REGION Network 39: Step[802] :
   RUNG wire#powerrail
      { S7_Templates := "SrcType := DInt" } EQ_Contact(in1 := "Unit1.Em2.ControlNodes".semiAutoSplice.sequence.status.currentStep, in2 := #JOB_8_STEP_02)
      Contact( "Unit1.Em2.ControlNodes".semiAutoSplice.sequence.status.seqActive )
      wire#w1
      Coil( "Unit1.Em2.ControlNodes".semiAutoSplice."step".action1[802] )
   END_RUNG
   RUNG wire#w1
      Coil( "Unit1.Em2.ControlNodes".semiAutoSplice."step".transition1[802] )
   END_RUNG
   RUNG wire#w1
      Contact( "Unit1.Em2.ControlNodes".semiAutoSplice."step".transition1[802] )
      { S7_Templates := "time_type := Time" } #statTonTimer[802].TON(pt := #SeqDelayTime, et =>)
      Move(in := #JOB_8_STEP_03, out1 => "Unit1.Em2.ControlNodes".semiAutoSplice.sequence.status.nextStep)
   END_RUNG
   // the same network as SCL:
   "Unit1.Em2.ControlNodes".semiAutoSplice."step".action1[802] := ("Unit1.Em2.ControlNodes".semiAutoSplice.sequence.status.currentStep = #JOB_8_STEP_02) AND "Unit1.Em2.ControlNodes".semiAutoSplice.sequence.status.seqActive;
   "Unit1.Em2.ControlNodes".semiAutoSplice."step".transition1[802] := ("Unit1.Em2.ControlNodes".semiAutoSplice.sequence.status.currentStep = #JOB_8_STEP_02) AND "Unit1.Em2.ControlNodes".semiAutoSplice.sequence.status.seqActive;
   #statTonTimer[802].TON(IN := ("Unit1.Em2.ControlNodes".semiAutoSplice.sequence.status.currentStep = #JOB_8_STEP_02) AND "Unit1.Em2.ControlNodes".semiAutoSplice.sequence.status.seqActive AND "Unit1.Em2.ControlNodes".semiAutoSplice."step".transition1[802],
                          PT := #SeqDelayTime);
   IF #statTonTimer[802].Q THEN
       "Unit1.Em2.ControlNodes".semiAutoSplice.sequence.status.nextStep := #JOB_8_STEP_03;
   END_IF;
END_REGION

REGION Network 40: Step[803] : cutter Home (Down)
   RUNG wire#powerrail
      { S7_Templates := "SrcType := DInt" } EQ_Contact(in1 := "Unit1.Em2.ControlNodes".semiAutoSplice.sequence.status.currentStep, in2 := #JOB_8_STEP_03)
      Contact( "Unit1.Em2.ControlNodes".semiAutoSplice.sequence.status.seqActive )
      wire#w1
      I_Contact( "Unit1.Em2.ControlNodes".cmCutterUpDown.monitoring.inHomePos )
      Coil( "Unit1.Em2.ControlNodes".semiAutoSplice."step".action1[803] )
   END_RUNG
   RUNG wire#w1
      Contact( "Unit1.Em2.ControlNodes".cmCutterUpDown.monitoring.inHomePos )
      Coil( "Unit1.Em2.ControlNodes".semiAutoSplice."step".transition1[803] )
   END_RUNG
   RUNG wire#w1
      Contact( "Unit1.Em2.ControlNodes".semiAutoSplice."step".transition1[803] )
      { S7_Templates := "time_type := Time" } #statTonTimer[803].TON(pt := #SeqDelayTime, et =>)
      Move(in := #JOB_8_STEP_04, out1 => "Unit1.Em2.ControlNodes".semiAutoSplice.sequence.status.nextStep)
      Add(in1 := #RetryCnt[0], in2 := 1, out => #RetryCnt[0])
   END_RUNG
   // the same network as SCL:
   #_w1 := ("Unit1.Em2.ControlNodes".semiAutoSplice.sequence.status.currentStep = #JOB_8_STEP_03) AND "Unit1.Em2.ControlNodes".semiAutoSplice.sequence.status.seqActive;
   "Unit1.Em2.ControlNodes".semiAutoSplice."step".action1[803] := #_w1 AND NOT "Unit1.Em2.ControlNodes".cmCutterUpDown.monitoring.inHomePos;
   "Unit1.Em2.ControlNodes".semiAutoSplice."step".transition1[803] := #_w1 AND "Unit1.Em2.ControlNodes".cmCutterUpDown.monitoring.inHomePos;
   #statTonTimer[803].TON(IN := #_w1 AND "Unit1.Em2.ControlNodes".semiAutoSplice."step".transition1[803],
                          PT := #SeqDelayTime);
   IF #statTonTimer[803].Q THEN
       "Unit1.Em2.ControlNodes".semiAutoSplice.sequence.status.nextStep := #JOB_8_STEP_04;
       #RetryCnt[0] := #RetryCnt[0] + 1;
   END_IF;
END_REGION

REGION Network 41: Step[804] : retry
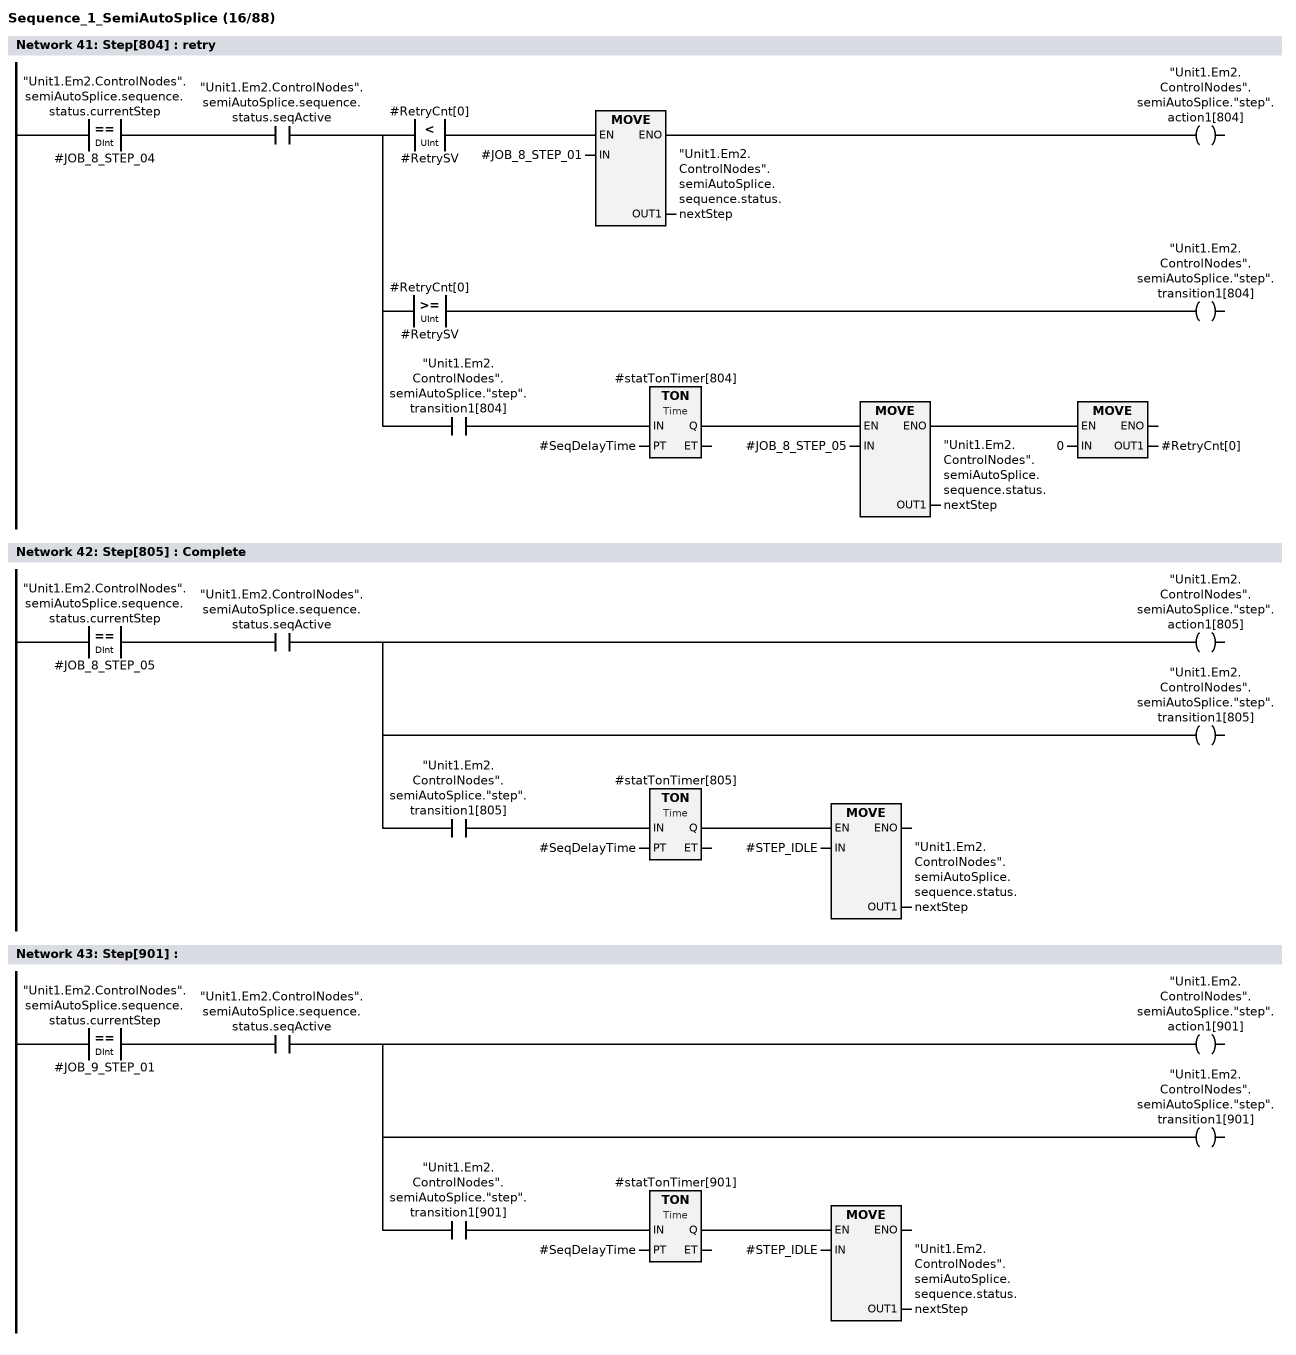
   RUNG wire#powerrail
      { S7_Templates := "SrcType := DInt" } EQ_Contact(in1 := "Unit1.Em2.ControlNodes".semiAutoSplice.sequence.status.currentStep, in2 := #JOB_8_STEP_04)
      Contact( "Unit1.Em2.ControlNodes".semiAutoSplice.sequence.status.seqActive )
      wire#w1
      { S7_Templates := "SrcType := UInt" } LT_Contact(in1 := #RetryCnt[0], in2 := #RetrySV)
      Move(in := #JOB_8_STEP_01, out1 => "Unit1.Em2.ControlNodes".semiAutoSplice.sequence.status.nextStep)
      Coil( "Unit1.Em2.ControlNodes".semiAutoSplice."step".action1[804] )
   END_RUNG
   RUNG wire#w1
      { S7_Templates := "SrcType := UInt" } GE_Contact(in1 := #RetryCnt[0], in2 := #RetrySV)
      Coil( "Unit1.Em2.ControlNodes".semiAutoSplice."step".transition1[804] )
   END_RUNG
   RUNG wire#w1
      Contact( "Unit1.Em2.ControlNodes".semiAutoSplice."step".transition1[804] )
      { S7_Templates := "time_type := Time" } #statTonTimer[804].TON(pt := #SeqDelayTime, et =>)
      Move(in := #JOB_8_STEP_05, out1 => "Unit1.Em2.ControlNodes".semiAutoSplice.sequence.status.nextStep)
      Move(in := 0, out1 => #RetryCnt[0])
   END_RUNG
   // the same network as SCL:
   #_w1 := ("Unit1.Em2.ControlNodes".semiAutoSplice.sequence.status.currentStep = #JOB_8_STEP_04) AND "Unit1.Em2.ControlNodes".semiAutoSplice.sequence.status.seqActive;
   #_w2 := #_w1 AND (#RetryCnt[0] < #RetrySV);
   IF #_w2 THEN "Unit1.Em2.ControlNodes".semiAutoSplice.sequence.status.nextStep := #JOB_8_STEP_01; END_IF;
   "Unit1.Em2.ControlNodes".semiAutoSplice."step".action1[804] := #_w2;
   "Unit1.Em2.ControlNodes".semiAutoSplice."step".transition1[804] := #_w1 AND (#RetryCnt[0] >= #RetrySV);
   #statTonTimer[804].TON(IN := #_w1 AND "Unit1.Em2.ControlNodes".semiAutoSplice."step".transition1[804],
                          PT := #SeqDelayTime);
   IF #statTonTimer[804].Q THEN
       "Unit1.Em2.ControlNodes".semiAutoSplice.sequence.status.nextStep := #JOB_8_STEP_05;
       #RetryCnt[0] := 0;
   END_IF;
END_REGION

REGION Network 42: Step[805] : Complete
   RUNG wire#powerrail
      { S7_Templates := "SrcType := DInt" } EQ_Contact(in1 := "Unit1.Em2.ControlNodes".semiAutoSplice.sequence.status.currentStep, in2 := #JOB_8_STEP_05)
      Contact( "Unit1.Em2.ControlNodes".semiAutoSplice.sequence.status.seqActive )
      wire#w1
      Coil( "Unit1.Em2.ControlNodes".semiAutoSplice."step".action1[805] )
   END_RUNG
   RUNG wire#w1
      Coil( "Unit1.Em2.ControlNodes".semiAutoSplice."step".transition1[805] )
   END_RUNG
   RUNG wire#w1
      Contact( "Unit1.Em2.ControlNodes".semiAutoSplice."step".transition1[805] )
      { S7_Templates := "time_type := Time" } #statTonTimer[805].TON(pt := #SeqDelayTime, et =>)
      Move(in := #STEP_IDLE, out1 => "Unit1.Em2.ControlNodes".semiAutoSplice.sequence.status.nextStep)
   END_RUNG
   // the same network as SCL:
   "Unit1.Em2.ControlNodes".semiAutoSplice."step".action1[805] := ("Unit1.Em2.ControlNodes".semiAutoSplice.sequence.status.currentStep = #JOB_8_STEP_05) AND "Unit1.Em2.ControlNodes".semiAutoSplice.sequence.status.seqActive;
   "Unit1.Em2.ControlNodes".semiAutoSplice."step".transition1[805] := ("Unit1.Em2.ControlNodes".semiAutoSplice.sequence.status.currentStep = #JOB_8_STEP_05) AND "Unit1.Em2.ControlNodes".semiAutoSplice.sequence.status.seqActive;
   #statTonTimer[805].TON(IN := ("Unit1.Em2.ControlNodes".semiAutoSplice.sequence.status.currentStep = #JOB_8_STEP_05) AND "Unit1.Em2.ControlNodes".semiAutoSplice.sequence.status.seqActive AND "Unit1.Em2.ControlNodes".semiAutoSplice."step".transition1[805],
                          PT := #SeqDelayTime);
   IF #statTonTimer[805].Q THEN
       "Unit1.Em2.ControlNodes".semiAutoSplice.sequence.status.nextStep := #STEP_IDLE;
   END_IF;
END_REGION

REGION Network 43: Step[901] :
   RUNG wire#powerrail
      { S7_Templates := "SrcType := DInt" } EQ_Contact(in1 := "Unit1.Em2.ControlNodes".semiAutoSplice.sequence.status.currentStep, in2 := #JOB_9_STEP_01)
      Contact( "Unit1.Em2.ControlNodes".semiAutoSplice.sequence.status.seqActive )
      wire#w1
      Coil( "Unit1.Em2.ControlNodes".semiAutoSplice."step".action1[901] )
   END_RUNG
   RUNG wire#w1
      Coil( "Unit1.Em2.ControlNodes".semiAutoSplice."step".transition1[901] )
   END_RUNG
   RUNG wire#w1
      Contact( "Unit1.Em2.ControlNodes".semiAutoSplice."step".transition1[901] )
      { S7_Templates := "time_type := Time" } #statTonTimer[901].TON(pt := #SeqDelayTime, et =>)
      Move(in := #STEP_IDLE, out1 => "Unit1.Em2.ControlNodes".semiAutoSplice.sequence.status.nextStep)
   END_RUNG
   // the same network as SCL:
   "Unit1.Em2.ControlNodes".semiAutoSplice."step".action1[901] := ("Unit1.Em2.ControlNodes".semiAutoSplice.sequence.status.currentStep = #JOB_9_STEP_01) AND "Unit1.Em2.ControlNodes".semiAutoSplice.sequence.status.seqActive;
   "Unit1.Em2.ControlNodes".semiAutoSplice."step".transition1[901] := ("Unit1.Em2.ControlNodes".semiAutoSplice.sequence.status.currentStep = #JOB_9_STEP_01) AND "Unit1.Em2.ControlNodes".semiAutoSplice.sequence.status.seqActive;
   #statTonTimer[901].TON(IN := ("Unit1.Em2.ControlNodes".semiAutoSplice.sequence.status.currentStep = #JOB_9_STEP_01) AND "Unit1.Em2.ControlNodes".semiAutoSplice.sequence.status.seqActive AND "Unit1.Em2.ControlNodes".semiAutoSplice."step".transition1[901],
                          PT := #SeqDelayTime);
   IF #statTonTimer[901].Q THEN
       "Unit1.Em2.ControlNodes".semiAutoSplice.sequence.status.nextStep := #STEP_IDLE;
   END_IF;
END_REGION

REGION Network 44: Step[1001] : Top Link Top Left/right Vacc Off (Btm Left/Right Vacc On)
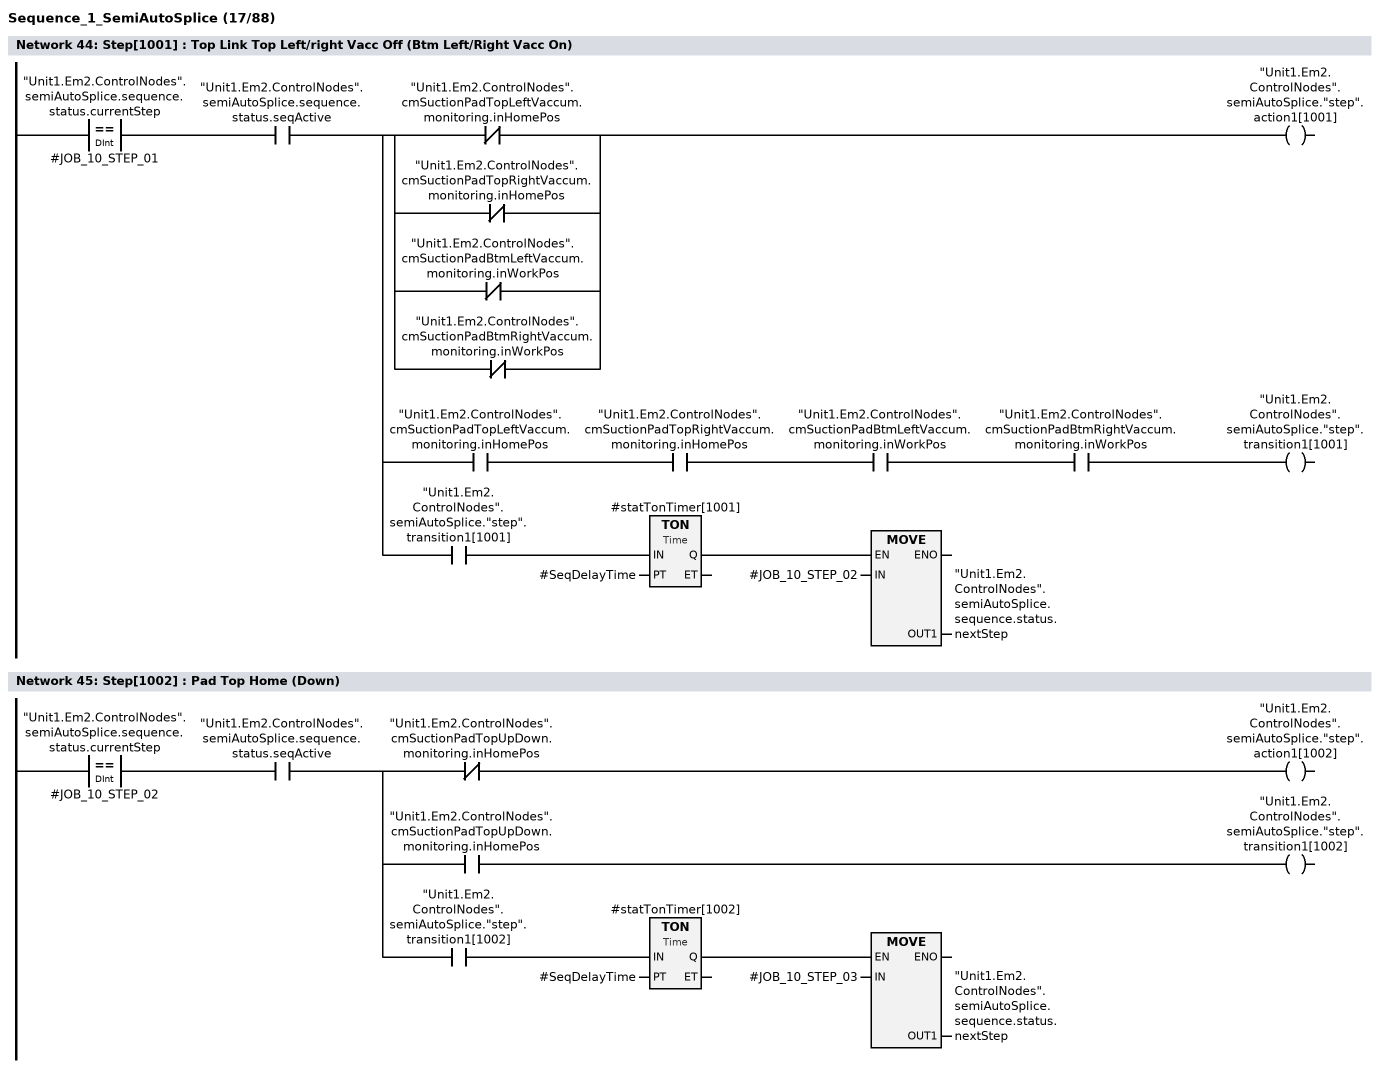
   RUNG wire#powerrail
      { S7_Templates := "SrcType := DInt" } EQ_Contact(in1 := "Unit1.Em2.ControlNodes".semiAutoSplice.sequence.status.currentStep, in2 := #JOB_10_STEP_01)
      Contact( "Unit1.Em2.ControlNodes".semiAutoSplice.sequence.status.seqActive )
      wire#w1
      I_Contact( "Unit1.Em2.ControlNodes".cmSuctionPadTopLeftVaccum.monitoring.inHomePos )
      wire#w2
      Coil( "Unit1.Em2.ControlNodes".semiAutoSplice."step".action1[1001] )
   END_RUNG
   RUNG wire#w1
      I_Contact( "Unit1.Em2.ControlNodes".cmSuctionPadTopRightVaccum.monitoring.inHomePos )
   END_RUNG wire#w2
   RUNG wire#w1
      I_Contact( "Unit1.Em2.ControlNodes".cmSuctionPadBtmLeftVaccum.monitoring.inWorkPos )
   END_RUNG wire#w2
   RUNG wire#w1
      I_Contact( "Unit1.Em2.ControlNodes".cmSuctionPadBtmRightVaccum.monitoring.inWorkPos )
   END_RUNG wire#w2
   RUNG wire#w1
      Contact( "Unit1.Em2.ControlNodes".cmSuctionPadTopLeftVaccum.monitoring.inHomePos )
      Contact( "Unit1.Em2.ControlNodes".cmSuctionPadTopRightVaccum.monitoring.inHomePos )
      Contact( "Unit1.Em2.ControlNodes".cmSuctionPadBtmLeftVaccum.monitoring.inWorkPos )
      Contact( "Unit1.Em2.ControlNodes".cmSuctionPadBtmRightVaccum.monitoring.inWorkPos )
      Coil( "Unit1.Em2.ControlNodes".semiAutoSplice."step".transition1[1001] )
   END_RUNG
   RUNG wire#w1
      Contact( "Unit1.Em2.ControlNodes".semiAutoSplice."step".transition1[1001] )
      { S7_Templates := "time_type := Time" } #statTonTimer[1001].TON(pt := #SeqDelayTime, et =>)
      Move(in := #JOB_10_STEP_02, out1 => "Unit1.Em2.ControlNodes".semiAutoSplice.sequence.status.nextStep)
   END_RUNG
   // the same network as SCL:
   #_w1 := ("Unit1.Em2.ControlNodes".semiAutoSplice.sequence.status.currentStep = #JOB_10_STEP_01) AND "Unit1.Em2.ControlNodes".semiAutoSplice.sequence.status.seqActive;
   "Unit1.Em2.ControlNodes".semiAutoSplice."step".action1[1001] := #_w1 AND (NOT "Unit1.Em2.ControlNodes".cmSuctionPadTopLeftVaccum.monitoring.inHomePos OR NOT "Unit1.Em2.ControlNodes".cmSuctionPadTopRightVaccum.monitoring.inHomePos OR NOT "Unit1.Em2.ControlNodes".cmSuctionPadBtmLeftVaccum.monitoring.inWorkPos OR NOT "Unit1.Em2.ControlNodes".cmSuctionPadBtmRightVaccum.monitoring.inWorkPos);
   "Unit1.Em2.ControlNodes".semiAutoSplice."step".transition1[1001] := #_w1 AND "Unit1.Em2.ControlNodes".cmSuctionPadTopLeftVaccum.monitoring.inHomePos AND "Unit1.Em2.ControlNodes".cmSuctionPadTopRightVaccum.monitoring.inHomePos AND "Unit1.Em2.ControlNodes".cmSuctionPadBtmLeftVaccum.monitoring.inWorkPos AND "Unit1.Em2.ControlNodes".cmSuctionPadBtmRightVaccum.monitoring.inWorkPos;
   #statTonTimer[1001].TON(IN := #_w1 AND "Unit1.Em2.ControlNodes".semiAutoSplice."step".transition1[1001],
                           PT := #SeqDelayTime);
   IF #statTonTimer[1001].Q THEN
       "Unit1.Em2.ControlNodes".semiAutoSplice.sequence.status.nextStep := #JOB_10_STEP_02;
   END_IF;
END_REGION

REGION Network 45: Step[1002] : Pad Top Home (Down)
   RUNG wire#powerrail
      { S7_Templates := "SrcType := DInt" } EQ_Contact(in1 := "Unit1.Em2.ControlNodes".semiAutoSplice.sequence.status.currentStep, in2 := #JOB_10_STEP_02)
      Contact( "Unit1.Em2.ControlNodes".semiAutoSplice.sequence.status.seqActive )
      wire#w1
      I_Contact( "Unit1.Em2.ControlNodes".cmSuctionPadTopUpDown.monitoring.inHomePos )
      Coil( "Unit1.Em2.ControlNodes".semiAutoSplice."step".action1[1002] )
   END_RUNG
   RUNG wire#w1
      Contact( "Unit1.Em2.ControlNodes".cmSuctionPadTopUpDown.monitoring.inHomePos )
      Coil( "Unit1.Em2.ControlNodes".semiAutoSplice."step".transition1[1002] )
   END_RUNG
   RUNG wire#w1
      Contact( "Unit1.Em2.ControlNodes".semiAutoSplice."step".transition1[1002] )
      { S7_Templates := "time_type := Time" } #statTonTimer[1002].TON(pt := #SeqDelayTime, et =>)
      Move(in := #JOB_10_STEP_03, out1 => "Unit1.Em2.ControlNodes".semiAutoSplice.sequence.status.nextStep)
   END_RUNG
   // the same network as SCL:
   #_w1 := ("Unit1.Em2.ControlNodes".semiAutoSplice.sequence.status.currentStep = #JOB_10_STEP_02) AND "Unit1.Em2.ControlNodes".semiAutoSplice.sequence.status.seqActive;
   "Unit1.Em2.ControlNodes".semiAutoSplice."step".action1[1002] := #_w1 AND NOT "Unit1.Em2.ControlNodes".cmSuctionPadTopUpDown.monitoring.inHomePos;
   "Unit1.Em2.ControlNodes".semiAutoSplice."step".transition1[1002] := #_w1 AND "Unit1.Em2.ControlNodes".cmSuctionPadTopUpDown.monitoring.inHomePos;
   #statTonTimer[1002].TON(IN := #_w1 AND "Unit1.Em2.ControlNodes".semiAutoSplice."step".transition1[1002],
                           PT := #SeqDelayTime);
   IF #statTonTimer[1002].Q THEN
       "Unit1.Em2.ControlNodes".semiAutoSplice.sequence.status.nextStep := #JOB_10_STEP_03;
   END_IF;
END_REGION

REGION Network 46: Step[1003] :
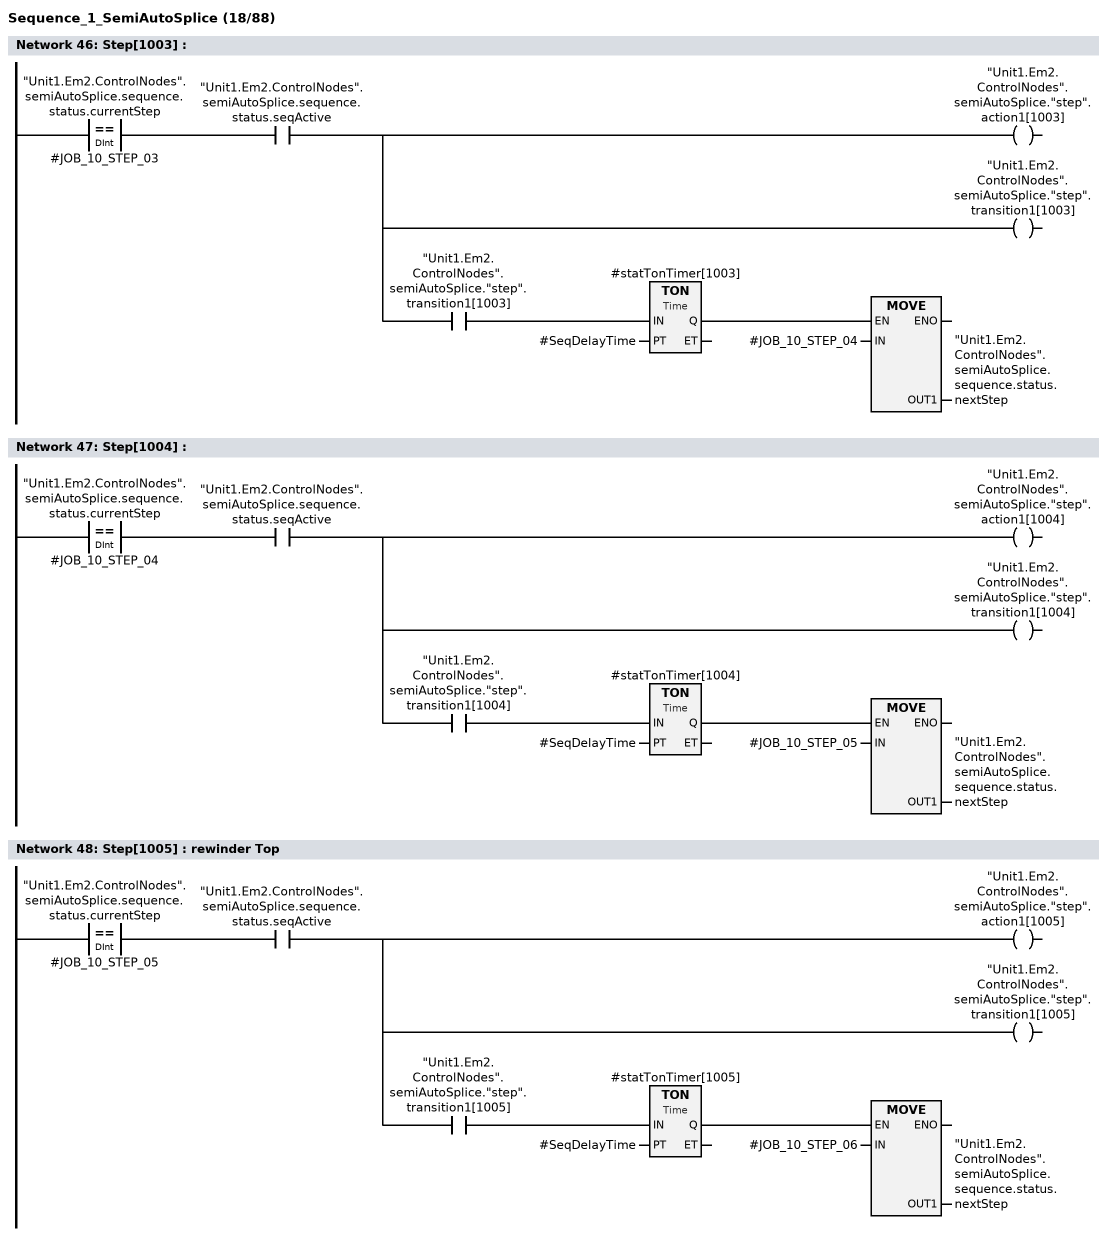
   RUNG wire#powerrail
      { S7_Templates := "SrcType := DInt" } EQ_Contact(in1 := "Unit1.Em2.ControlNodes".semiAutoSplice.sequence.status.currentStep, in2 := #JOB_10_STEP_03)
      Contact( "Unit1.Em2.ControlNodes".semiAutoSplice.sequence.status.seqActive )
      wire#w1
      Coil( "Unit1.Em2.ControlNodes".semiAutoSplice."step".action1[1003] )
   END_RUNG
   RUNG wire#w1
      Coil( "Unit1.Em2.ControlNodes".semiAutoSplice."step".transition1[1003] )
   END_RUNG
   RUNG wire#w1
      Contact( "Unit1.Em2.ControlNodes".semiAutoSplice."step".transition1[1003] )
      { S7_Templates := "time_type := Time" } #statTonTimer[1003].TON(pt := #SeqDelayTime, et =>)
      Move(in := #JOB_10_STEP_04, out1 => "Unit1.Em2.ControlNodes".semiAutoSplice.sequence.status.nextStep)
   END_RUNG
   // the same network as SCL:
   "Unit1.Em2.ControlNodes".semiAutoSplice."step".action1[1003] := ("Unit1.Em2.ControlNodes".semiAutoSplice.sequence.status.currentStep = #JOB_10_STEP_03) AND "Unit1.Em2.ControlNodes".semiAutoSplice.sequence.status.seqActive;
   "Unit1.Em2.ControlNodes".semiAutoSplice."step".transition1[1003] := ("Unit1.Em2.ControlNodes".semiAutoSplice.sequence.status.currentStep = #JOB_10_STEP_03) AND "Unit1.Em2.ControlNodes".semiAutoSplice.sequence.status.seqActive;
   #statTonTimer[1003].TON(IN := ("Unit1.Em2.ControlNodes".semiAutoSplice.sequence.status.currentStep = #JOB_10_STEP_03) AND "Unit1.Em2.ControlNodes".semiAutoSplice.sequence.status.seqActive AND "Unit1.Em2.ControlNodes".semiAutoSplice."step".transition1[1003],
                           PT := #SeqDelayTime);
   IF #statTonTimer[1003].Q THEN
       "Unit1.Em2.ControlNodes".semiAutoSplice.sequence.status.nextStep := #JOB_10_STEP_04;
   END_IF;
END_REGION

REGION Network 47: Step[1004] :
   RUNG wire#powerrail
      { S7_Templates := "SrcType := DInt" } EQ_Contact(in1 := "Unit1.Em2.ControlNodes".semiAutoSplice.sequence.status.currentStep, in2 := #JOB_10_STEP_04)
      Contact( "Unit1.Em2.ControlNodes".semiAutoSplice.sequence.status.seqActive )
      wire#w1
      Coil( "Unit1.Em2.ControlNodes".semiAutoSplice."step".action1[1004] )
   END_RUNG
   RUNG wire#w1
      Coil( "Unit1.Em2.ControlNodes".semiAutoSplice."step".transition1[1004] )
   END_RUNG
   RUNG wire#w1
      Contact( "Unit1.Em2.ControlNodes".semiAutoSplice."step".transition1[1004] )
      { S7_Templates := "time_type := Time" } #statTonTimer[1004].TON(pt := #SeqDelayTime, et =>)
      Move(in := #JOB_10_STEP_05, out1 => "Unit1.Em2.ControlNodes".semiAutoSplice.sequence.status.nextStep)
   END_RUNG
   // the same network as SCL:
   "Unit1.Em2.ControlNodes".semiAutoSplice."step".action1[1004] := ("Unit1.Em2.ControlNodes".semiAutoSplice.sequence.status.currentStep = #JOB_10_STEP_04) AND "Unit1.Em2.ControlNodes".semiAutoSplice.sequence.status.seqActive;
   "Unit1.Em2.ControlNodes".semiAutoSplice."step".transition1[1004] := ("Unit1.Em2.ControlNodes".semiAutoSplice.sequence.status.currentStep = #JOB_10_STEP_04) AND "Unit1.Em2.ControlNodes".semiAutoSplice.sequence.status.seqActive;
   #statTonTimer[1004].TON(IN := ("Unit1.Em2.ControlNodes".semiAutoSplice.sequence.status.currentStep = #JOB_10_STEP_04) AND "Unit1.Em2.ControlNodes".semiAutoSplice.sequence.status.seqActive AND "Unit1.Em2.ControlNodes".semiAutoSplice."step".transition1[1004],
                           PT := #SeqDelayTime);
   IF #statTonTimer[1004].Q THEN
       "Unit1.Em2.ControlNodes".semiAutoSplice.sequence.status.nextStep := #JOB_10_STEP_05;
   END_IF;
END_REGION

REGION Network 48: Step[1005] : rewinder Top
   RUNG wire#powerrail
      { S7_Templates := "SrcType := DInt" } EQ_Contact(in1 := "Unit1.Em2.ControlNodes".semiAutoSplice.sequence.status.currentStep, in2 := #JOB_10_STEP_05)
      Contact( "Unit1.Em2.ControlNodes".semiAutoSplice.sequence.status.seqActive )
      wire#w1
      Coil( "Unit1.Em2.ControlNodes".semiAutoSplice."step".action1[1005] )
   END_RUNG
   RUNG wire#w1
      Coil( "Unit1.Em2.ControlNodes".semiAutoSplice."step".transition1[1005] )
   END_RUNG
   RUNG wire#w1
      Contact( "Unit1.Em2.ControlNodes".semiAutoSplice."step".transition1[1005] )
      { S7_Templates := "time_type := Time" } #statTonTimer[1005].TON(pt := #SeqDelayTime, et =>)
      Move(in := #JOB_10_STEP_06, out1 => "Unit1.Em2.ControlNodes".semiAutoSplice.sequence.status.nextStep)
   END_RUNG
   // the same network as SCL:
   "Unit1.Em2.ControlNodes".semiAutoSplice."step".action1[1005] := ("Unit1.Em2.ControlNodes".semiAutoSplice.sequence.status.currentStep = #JOB_10_STEP_05) AND "Unit1.Em2.ControlNodes".semiAutoSplice.sequence.status.seqActive;
   "Unit1.Em2.ControlNodes".semiAutoSplice."step".transition1[1005] := ("Unit1.Em2.ControlNodes".semiAutoSplice.sequence.status.currentStep = #JOB_10_STEP_05) AND "Unit1.Em2.ControlNodes".semiAutoSplice.sequence.status.seqActive;
   #statTonTimer[1005].TON(IN := ("Unit1.Em2.ControlNodes".semiAutoSplice.sequence.status.currentStep = #JOB_10_STEP_05) AND "Unit1.Em2.ControlNodes".semiAutoSplice.sequence.status.seqActive AND "Unit1.Em2.ControlNodes".semiAutoSplice."step".transition1[1005],
                           PT := #SeqDelayTime);
   IF #statTonTimer[1005].Q THEN
       "Unit1.Em2.ControlNodes".semiAutoSplice.sequence.status.nextStep := #JOB_10_STEP_06;
   END_IF;
END_REGION

REGION Network 49: Step[1006] : Complete
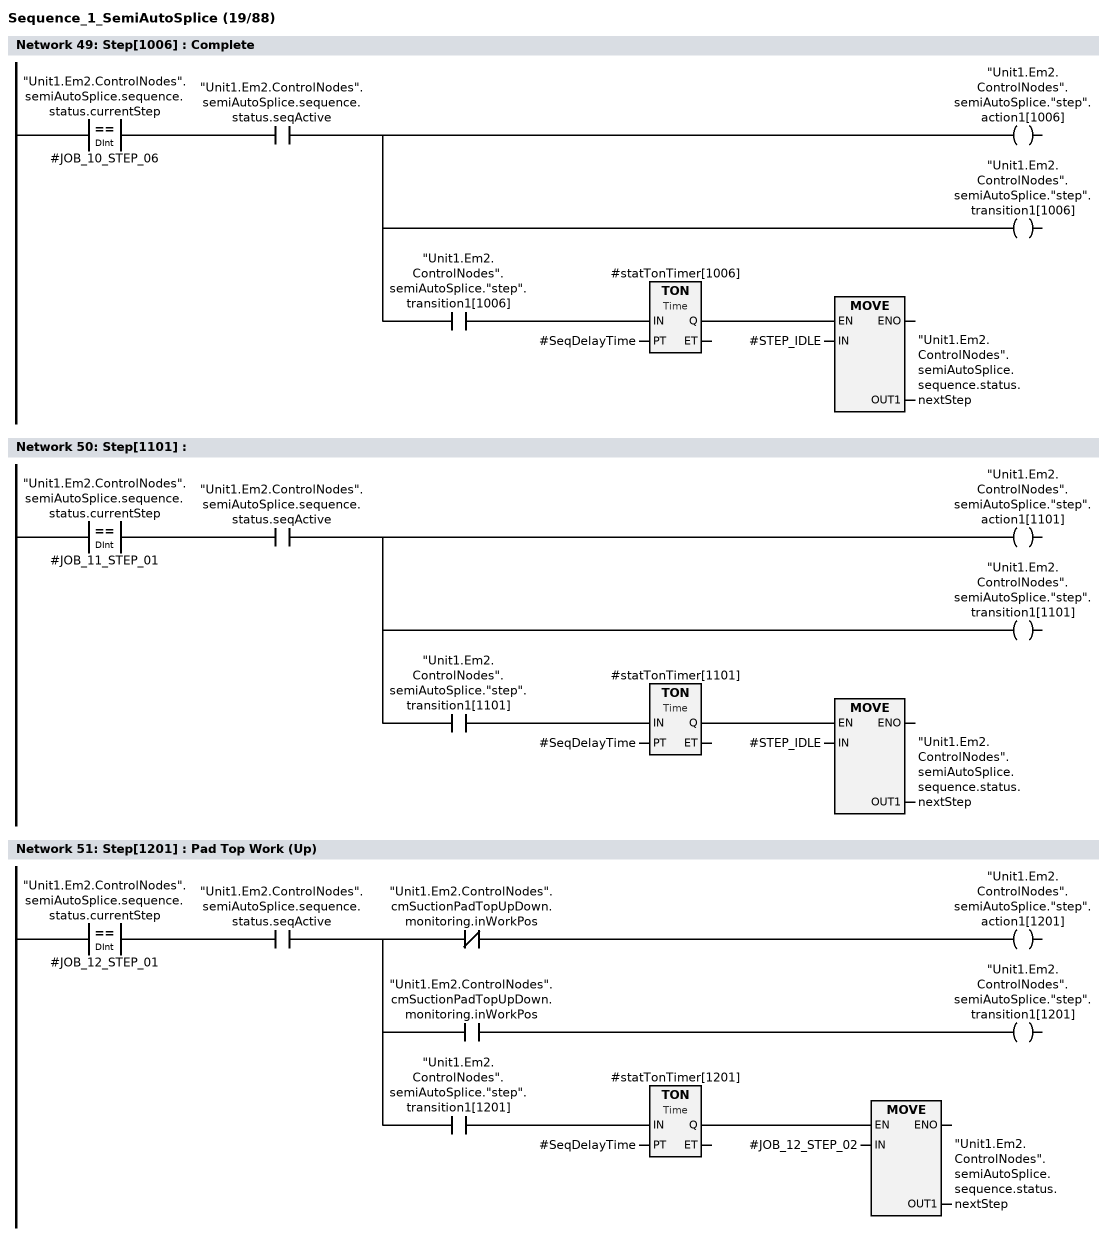
   RUNG wire#powerrail
      { S7_Templates := "SrcType := DInt" } EQ_Contact(in1 := "Unit1.Em2.ControlNodes".semiAutoSplice.sequence.status.currentStep, in2 := #JOB_10_STEP_06)
      Contact( "Unit1.Em2.ControlNodes".semiAutoSplice.sequence.status.seqActive )
      wire#w1
      Coil( "Unit1.Em2.ControlNodes".semiAutoSplice."step".action1[1006] )
   END_RUNG
   RUNG wire#w1
      Coil( "Unit1.Em2.ControlNodes".semiAutoSplice."step".transition1[1006] )
   END_RUNG
   RUNG wire#w1
      Contact( "Unit1.Em2.ControlNodes".semiAutoSplice."step".transition1[1006] )
      { S7_Templates := "time_type := Time" } #statTonTimer[1006].TON(pt := #SeqDelayTime, et =>)
      Move(in := #STEP_IDLE, out1 => "Unit1.Em2.ControlNodes".semiAutoSplice.sequence.status.nextStep)
   END_RUNG
   // the same network as SCL:
   "Unit1.Em2.ControlNodes".semiAutoSplice."step".action1[1006] := ("Unit1.Em2.ControlNodes".semiAutoSplice.sequence.status.currentStep = #JOB_10_STEP_06) AND "Unit1.Em2.ControlNodes".semiAutoSplice.sequence.status.seqActive;
   "Unit1.Em2.ControlNodes".semiAutoSplice."step".transition1[1006] := ("Unit1.Em2.ControlNodes".semiAutoSplice.sequence.status.currentStep = #JOB_10_STEP_06) AND "Unit1.Em2.ControlNodes".semiAutoSplice.sequence.status.seqActive;
   #statTonTimer[1006].TON(IN := ("Unit1.Em2.ControlNodes".semiAutoSplice.sequence.status.currentStep = #JOB_10_STEP_06) AND "Unit1.Em2.ControlNodes".semiAutoSplice.sequence.status.seqActive AND "Unit1.Em2.ControlNodes".semiAutoSplice."step".transition1[1006],
                           PT := #SeqDelayTime);
   IF #statTonTimer[1006].Q THEN
       "Unit1.Em2.ControlNodes".semiAutoSplice.sequence.status.nextStep := #STEP_IDLE;
   END_IF;
END_REGION

REGION Network 50: Step[1101] :
   RUNG wire#powerrail
      { S7_Templates := "SrcType := DInt" } EQ_Contact(in1 := "Unit1.Em2.ControlNodes".semiAutoSplice.sequence.status.currentStep, in2 := #JOB_11_STEP_01)
      Contact( "Unit1.Em2.ControlNodes".semiAutoSplice.sequence.status.seqActive )
      wire#w1
      Coil( "Unit1.Em2.ControlNodes".semiAutoSplice."step".action1[1101] )
   END_RUNG
   RUNG wire#w1
      Coil( "Unit1.Em2.ControlNodes".semiAutoSplice."step".transition1[1101] )
   END_RUNG
   RUNG wire#w1
      Contact( "Unit1.Em2.ControlNodes".semiAutoSplice."step".transition1[1101] )
      { S7_Templates := "time_type := Time" } #statTonTimer[1101].TON(pt := #SeqDelayTime, et =>)
      Move(in := #STEP_IDLE, out1 => "Unit1.Em2.ControlNodes".semiAutoSplice.sequence.status.nextStep)
   END_RUNG
   // the same network as SCL:
   "Unit1.Em2.ControlNodes".semiAutoSplice."step".action1[1101] := ("Unit1.Em2.ControlNodes".semiAutoSplice.sequence.status.currentStep = #JOB_11_STEP_01) AND "Unit1.Em2.ControlNodes".semiAutoSplice.sequence.status.seqActive;
   "Unit1.Em2.ControlNodes".semiAutoSplice."step".transition1[1101] := ("Unit1.Em2.ControlNodes".semiAutoSplice.sequence.status.currentStep = #JOB_11_STEP_01) AND "Unit1.Em2.ControlNodes".semiAutoSplice.sequence.status.seqActive;
   #statTonTimer[1101].TON(IN := ("Unit1.Em2.ControlNodes".semiAutoSplice.sequence.status.currentStep = #JOB_11_STEP_01) AND "Unit1.Em2.ControlNodes".semiAutoSplice.sequence.status.seqActive AND "Unit1.Em2.ControlNodes".semiAutoSplice."step".transition1[1101],
                           PT := #SeqDelayTime);
   IF #statTonTimer[1101].Q THEN
       "Unit1.Em2.ControlNodes".semiAutoSplice.sequence.status.nextStep := #STEP_IDLE;
   END_IF;
END_REGION

REGION Network 51: Step[1201] : Pad Top Work (Up)
   RUNG wire#powerrail
      { S7_Templates := "SrcType := DInt" } EQ_Contact(in1 := "Unit1.Em2.ControlNodes".semiAutoSplice.sequence.status.currentStep, in2 := #JOB_12_STEP_01)
      Contact( "Unit1.Em2.ControlNodes".semiAutoSplice.sequence.status.seqActive )
      wire#w1
      I_Contact( "Unit1.Em2.ControlNodes".cmSuctionPadTopUpDown.monitoring.inWorkPos )
      Coil( "Unit1.Em2.ControlNodes".semiAutoSplice."step".action1[1201] )
   END_RUNG
   RUNG wire#w1
      Contact( "Unit1.Em2.ControlNodes".cmSuctionPadTopUpDown.monitoring.inWorkPos )
      Coil( "Unit1.Em2.ControlNodes".semiAutoSplice."step".transition1[1201] )
   END_RUNG
   RUNG wire#w1
      Contact( "Unit1.Em2.ControlNodes".semiAutoSplice."step".transition1[1201] )
      { S7_Templates := "time_type := Time" } #statTonTimer[1201].TON(pt := #SeqDelayTime, et =>)
      Move(in := #JOB_12_STEP_02, out1 => "Unit1.Em2.ControlNodes".semiAutoSplice.sequence.status.nextStep)
   END_RUNG
   // the same network as SCL:
   #_w1 := ("Unit1.Em2.ControlNodes".semiAutoSplice.sequence.status.currentStep = #JOB_12_STEP_01) AND "Unit1.Em2.ControlNodes".semiAutoSplice.sequence.status.seqActive;
   "Unit1.Em2.ControlNodes".semiAutoSplice."step".action1[1201] := #_w1 AND NOT "Unit1.Em2.ControlNodes".cmSuctionPadTopUpDown.monitoring.inWorkPos;
   "Unit1.Em2.ControlNodes".semiAutoSplice."step".transition1[1201] := #_w1 AND "Unit1.Em2.ControlNodes".cmSuctionPadTopUpDown.monitoring.inWorkPos;
   #statTonTimer[1201].TON(IN := #_w1 AND "Unit1.Em2.ControlNodes".semiAutoSplice."step".transition1[1201],
                           PT := #SeqDelayTime);
   IF #statTonTimer[1201].Q THEN
       "Unit1.Em2.ControlNodes".semiAutoSplice.sequence.status.nextStep := #JOB_12_STEP_02;
   END_IF;
END_REGION

REGION Network 52: Step[1202] :
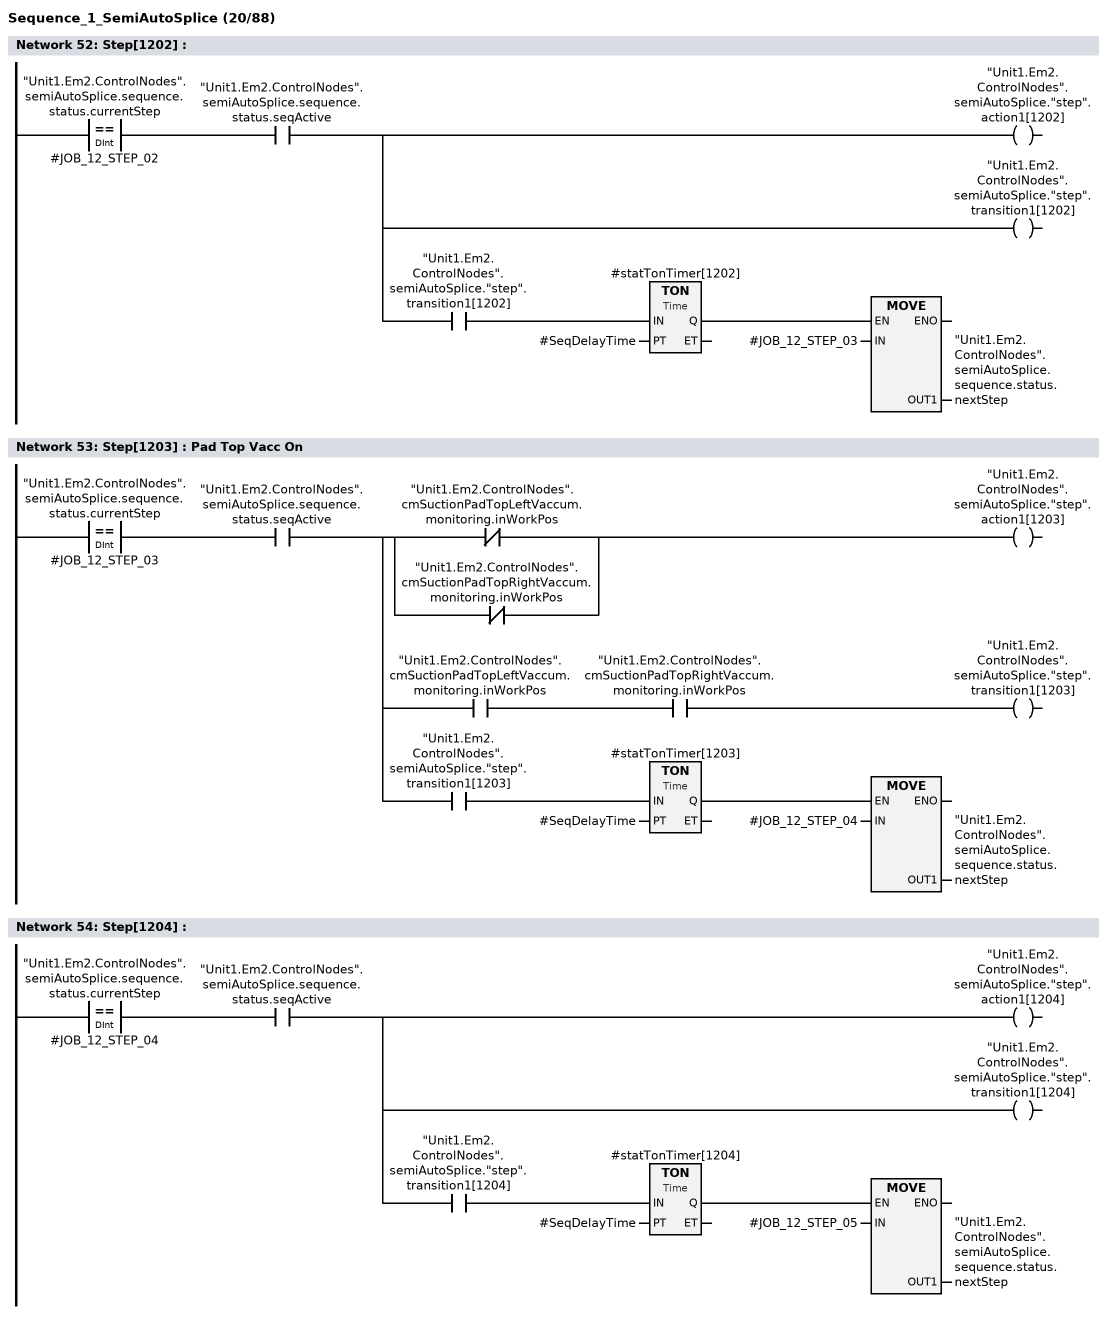
   RUNG wire#powerrail
      { S7_Templates := "SrcType := DInt" } EQ_Contact(in1 := "Unit1.Em2.ControlNodes".semiAutoSplice.sequence.status.currentStep, in2 := #JOB_12_STEP_02)
      Contact( "Unit1.Em2.ControlNodes".semiAutoSplice.sequence.status.seqActive )
      wire#w1
      Coil( "Unit1.Em2.ControlNodes".semiAutoSplice."step".action1[1202] )
   END_RUNG
   RUNG wire#w1
      Coil( "Unit1.Em2.ControlNodes".semiAutoSplice."step".transition1[1202] )
   END_RUNG
   RUNG wire#w1
      Contact( "Unit1.Em2.ControlNodes".semiAutoSplice."step".transition1[1202] )
      { S7_Templates := "time_type := Time" } #statTonTimer[1202].TON(pt := #SeqDelayTime, et =>)
      Move(in := #JOB_12_STEP_03, out1 => "Unit1.Em2.ControlNodes".semiAutoSplice.sequence.status.nextStep)
   END_RUNG
   // the same network as SCL:
   "Unit1.Em2.ControlNodes".semiAutoSplice."step".action1[1202] := ("Unit1.Em2.ControlNodes".semiAutoSplice.sequence.status.currentStep = #JOB_12_STEP_02) AND "Unit1.Em2.ControlNodes".semiAutoSplice.sequence.status.seqActive;
   "Unit1.Em2.ControlNodes".semiAutoSplice."step".transition1[1202] := ("Unit1.Em2.ControlNodes".semiAutoSplice.sequence.status.currentStep = #JOB_12_STEP_02) AND "Unit1.Em2.ControlNodes".semiAutoSplice.sequence.status.seqActive;
   #statTonTimer[1202].TON(IN := ("Unit1.Em2.ControlNodes".semiAutoSplice.sequence.status.currentStep = #JOB_12_STEP_02) AND "Unit1.Em2.ControlNodes".semiAutoSplice.sequence.status.seqActive AND "Unit1.Em2.ControlNodes".semiAutoSplice."step".transition1[1202],
                           PT := #SeqDelayTime);
   IF #statTonTimer[1202].Q THEN
       "Unit1.Em2.ControlNodes".semiAutoSplice.sequence.status.nextStep := #JOB_12_STEP_03;
   END_IF;
END_REGION

REGION Network 53: Step[1203] : Pad Top Vacc On
   RUNG wire#powerrail
      { S7_Templates := "SrcType := DInt" } EQ_Contact(in1 := "Unit1.Em2.ControlNodes".semiAutoSplice.sequence.status.currentStep, in2 := #JOB_12_STEP_03)
      Contact( "Unit1.Em2.ControlNodes".semiAutoSplice.sequence.status.seqActive )
      wire#w1
      I_Contact( "Unit1.Em2.ControlNodes".cmSuctionPadTopLeftVaccum.monitoring.inWorkPos )
      wire#w2
      Coil( "Unit1.Em2.ControlNodes".semiAutoSplice."step".action1[1203] )
   END_RUNG
   RUNG wire#w1
      I_Contact( "Unit1.Em2.ControlNodes".cmSuctionPadTopRightVaccum.monitoring.inWorkPos )
   END_RUNG wire#w2
   RUNG wire#w1
      Contact( "Unit1.Em2.ControlNodes".cmSuctionPadTopLeftVaccum.monitoring.inWorkPos )
      Contact( "Unit1.Em2.ControlNodes".cmSuctionPadTopRightVaccum.monitoring.inWorkPos )
      Coil( "Unit1.Em2.ControlNodes".semiAutoSplice."step".transition1[1203] )
   END_RUNG
   RUNG wire#w1
      Contact( "Unit1.Em2.ControlNodes".semiAutoSplice."step".transition1[1203] )
      { S7_Templates := "time_type := Time" } #statTonTimer[1203].TON(pt := #SeqDelayTime, et =>)
      Move(in := #JOB_12_STEP_04, out1 => "Unit1.Em2.ControlNodes".semiAutoSplice.sequence.status.nextStep)
   END_RUNG
   // the same network as SCL:
   #_w1 := ("Unit1.Em2.ControlNodes".semiAutoSplice.sequence.status.currentStep = #JOB_12_STEP_03) AND "Unit1.Em2.ControlNodes".semiAutoSplice.sequence.status.seqActive;
   "Unit1.Em2.ControlNodes".semiAutoSplice."step".action1[1203] := #_w1 AND (NOT "Unit1.Em2.ControlNodes".cmSuctionPadTopLeftVaccum.monitoring.inWorkPos OR NOT "Unit1.Em2.ControlNodes".cmSuctionPadTopRightVaccum.monitoring.inWorkPos);
   "Unit1.Em2.ControlNodes".semiAutoSplice."step".transition1[1203] := #_w1 AND "Unit1.Em2.ControlNodes".cmSuctionPadTopLeftVaccum.monitoring.inWorkPos AND "Unit1.Em2.ControlNodes".cmSuctionPadTopRightVaccum.monitoring.inWorkPos;
   #statTonTimer[1203].TON(IN := #_w1 AND "Unit1.Em2.ControlNodes".semiAutoSplice."step".transition1[1203],
                           PT := #SeqDelayTime);
   IF #statTonTimer[1203].Q THEN
       "Unit1.Em2.ControlNodes".semiAutoSplice.sequence.status.nextStep := #JOB_12_STEP_04;
   END_IF;
END_REGION

REGION Network 54: Step[1204] :
   RUNG wire#powerrail
      { S7_Templates := "SrcType := DInt" } EQ_Contact(in1 := "Unit1.Em2.ControlNodes".semiAutoSplice.sequence.status.currentStep, in2 := #JOB_12_STEP_04)
      Contact( "Unit1.Em2.ControlNodes".semiAutoSplice.sequence.status.seqActive )
      wire#w1
      Coil( "Unit1.Em2.ControlNodes".semiAutoSplice."step".action1[1204] )
   END_RUNG
   RUNG wire#w1
      Coil( "Unit1.Em2.ControlNodes".semiAutoSplice."step".transition1[1204] )
   END_RUNG
   RUNG wire#w1
      Contact( "Unit1.Em2.ControlNodes".semiAutoSplice."step".transition1[1204] )
      { S7_Templates := "time_type := Time" } #statTonTimer[1204].TON(pt := #SeqDelayTime, et =>)
      Move(in := #JOB_12_STEP_05, out1 => "Unit1.Em2.ControlNodes".semiAutoSplice.sequence.status.nextStep)
   END_RUNG
   // the same network as SCL:
   "Unit1.Em2.ControlNodes".semiAutoSplice."step".action1[1204] := ("Unit1.Em2.ControlNodes".semiAutoSplice.sequence.status.currentStep = #JOB_12_STEP_04) AND "Unit1.Em2.ControlNodes".semiAutoSplice.sequence.status.seqActive;
   "Unit1.Em2.ControlNodes".semiAutoSplice."step".transition1[1204] := ("Unit1.Em2.ControlNodes".semiAutoSplice.sequence.status.currentStep = #JOB_12_STEP_04) AND "Unit1.Em2.ControlNodes".semiAutoSplice.sequence.status.seqActive;
   #statTonTimer[1204].TON(IN := ("Unit1.Em2.ControlNodes".semiAutoSplice.sequence.status.currentStep = #JOB_12_STEP_04) AND "Unit1.Em2.ControlNodes".semiAutoSplice.sequence.status.seqActive AND "Unit1.Em2.ControlNodes".semiAutoSplice."step".transition1[1204],
                           PT := #SeqDelayTime);
   IF #statTonTimer[1204].Q THEN
       "Unit1.Em2.ControlNodes".semiAutoSplice.sequence.status.nextStep := #JOB_12_STEP_05;
   END_IF;
END_REGION

REGION Network 55: Step[1205] : Complete
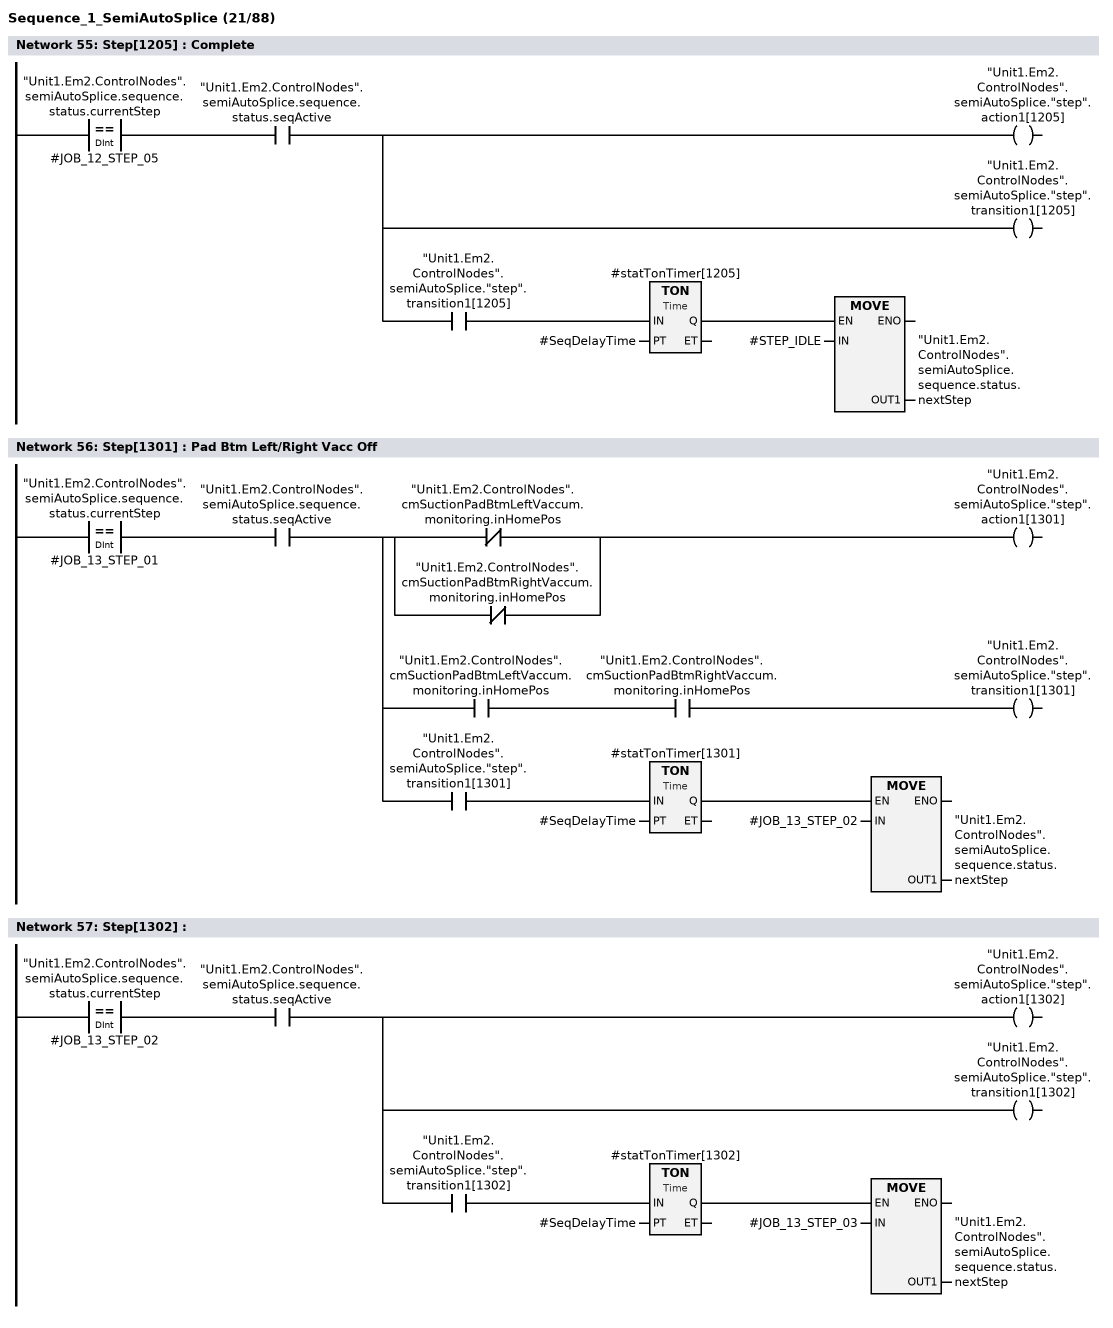
   RUNG wire#powerrail
      { S7_Templates := "SrcType := DInt" } EQ_Contact(in1 := "Unit1.Em2.ControlNodes".semiAutoSplice.sequence.status.currentStep, in2 := #JOB_12_STEP_05)
      Contact( "Unit1.Em2.ControlNodes".semiAutoSplice.sequence.status.seqActive )
      wire#w1
      Coil( "Unit1.Em2.ControlNodes".semiAutoSplice."step".action1[1205] )
   END_RUNG
   RUNG wire#w1
      Coil( "Unit1.Em2.ControlNodes".semiAutoSplice."step".transition1[1205] )
   END_RUNG
   RUNG wire#w1
      Contact( "Unit1.Em2.ControlNodes".semiAutoSplice."step".transition1[1205] )
      { S7_Templates := "time_type := Time" } #statTonTimer[1205].TON(pt := #SeqDelayTime, et =>)
      Move(in := #STEP_IDLE, out1 => "Unit1.Em2.ControlNodes".semiAutoSplice.sequence.status.nextStep)
   END_RUNG
   // the same network as SCL:
   "Unit1.Em2.ControlNodes".semiAutoSplice."step".action1[1205] := ("Unit1.Em2.ControlNodes".semiAutoSplice.sequence.status.currentStep = #JOB_12_STEP_05) AND "Unit1.Em2.ControlNodes".semiAutoSplice.sequence.status.seqActive;
   "Unit1.Em2.ControlNodes".semiAutoSplice."step".transition1[1205] := ("Unit1.Em2.ControlNodes".semiAutoSplice.sequence.status.currentStep = #JOB_12_STEP_05) AND "Unit1.Em2.ControlNodes".semiAutoSplice.sequence.status.seqActive;
   #statTonTimer[1205].TON(IN := ("Unit1.Em2.ControlNodes".semiAutoSplice.sequence.status.currentStep = #JOB_12_STEP_05) AND "Unit1.Em2.ControlNodes".semiAutoSplice.sequence.status.seqActive AND "Unit1.Em2.ControlNodes".semiAutoSplice."step".transition1[1205],
                           PT := #SeqDelayTime);
   IF #statTonTimer[1205].Q THEN
       "Unit1.Em2.ControlNodes".semiAutoSplice.sequence.status.nextStep := #STEP_IDLE;
   END_IF;
END_REGION

REGION Network 56: Step[1301] : Pad Btm Left/Right Vacc Off
   RUNG wire#powerrail
      { S7_Templates := "SrcType := DInt" } EQ_Contact(in1 := "Unit1.Em2.ControlNodes".semiAutoSplice.sequence.status.currentStep, in2 := #JOB_13_STEP_01)
      Contact( "Unit1.Em2.ControlNodes".semiAutoSplice.sequence.status.seqActive )
      wire#w1
      I_Contact( "Unit1.Em2.ControlNodes".cmSuctionPadBtmLeftVaccum.monitoring.inHomePos )
      wire#w2
      Coil( "Unit1.Em2.ControlNodes".semiAutoSplice."step".action1[1301] )
   END_RUNG
   RUNG wire#w1
      I_Contact( "Unit1.Em2.ControlNodes".cmSuctionPadBtmRightVaccum.monitoring.inHomePos )
   END_RUNG wire#w2
   RUNG wire#w1
      Contact( "Unit1.Em2.ControlNodes".cmSuctionPadBtmLeftVaccum.monitoring.inHomePos )
      Contact( "Unit1.Em2.ControlNodes".cmSuctionPadBtmRightVaccum.monitoring.inHomePos )
      Coil( "Unit1.Em2.ControlNodes".semiAutoSplice."step".transition1[1301] )
   END_RUNG
   RUNG wire#w1
      Contact( "Unit1.Em2.ControlNodes".semiAutoSplice."step".transition1[1301] )
      { S7_Templates := "time_type := Time" } #statTonTimer[1301].TON(pt := #SeqDelayTime, et =>)
      Move(in := #JOB_13_STEP_02, out1 => "Unit1.Em2.ControlNodes".semiAutoSplice.sequence.status.nextStep)
   END_RUNG
   // the same network as SCL:
   #_w1 := ("Unit1.Em2.ControlNodes".semiAutoSplice.sequence.status.currentStep = #JOB_13_STEP_01) AND "Unit1.Em2.ControlNodes".semiAutoSplice.sequence.status.seqActive;
   "Unit1.Em2.ControlNodes".semiAutoSplice."step".action1[1301] := #_w1 AND (NOT "Unit1.Em2.ControlNodes".cmSuctionPadBtmLeftVaccum.monitoring.inHomePos OR NOT "Unit1.Em2.ControlNodes".cmSuctionPadBtmRightVaccum.monitoring.inHomePos);
   "Unit1.Em2.ControlNodes".semiAutoSplice."step".transition1[1301] := #_w1 AND "Unit1.Em2.ControlNodes".cmSuctionPadBtmLeftVaccum.monitoring.inHomePos AND "Unit1.Em2.ControlNodes".cmSuctionPadBtmRightVaccum.monitoring.inHomePos;
   #statTonTimer[1301].TON(IN := #_w1 AND "Unit1.Em2.ControlNodes".semiAutoSplice."step".transition1[1301],
                           PT := #SeqDelayTime);
   IF #statTonTimer[1301].Q THEN
       "Unit1.Em2.ControlNodes".semiAutoSplice.sequence.status.nextStep := #JOB_13_STEP_02;
   END_IF;
END_REGION

REGION Network 57: Step[1302] :
   RUNG wire#powerrail
      { S7_Templates := "SrcType := DInt" } EQ_Contact(in1 := "Unit1.Em2.ControlNodes".semiAutoSplice.sequence.status.currentStep, in2 := #JOB_13_STEP_02)
      Contact( "Unit1.Em2.ControlNodes".semiAutoSplice.sequence.status.seqActive )
      wire#w1
      Coil( "Unit1.Em2.ControlNodes".semiAutoSplice."step".action1[1302] )
   END_RUNG
   RUNG wire#w1
      Coil( "Unit1.Em2.ControlNodes".semiAutoSplice."step".transition1[1302] )
   END_RUNG
   RUNG wire#w1
      Contact( "Unit1.Em2.ControlNodes".semiAutoSplice."step".transition1[1302] )
      { S7_Templates := "time_type := Time" } #statTonTimer[1302].TON(pt := #SeqDelayTime, et =>)
      Move(in := #JOB_13_STEP_03, out1 => "Unit1.Em2.ControlNodes".semiAutoSplice.sequence.status.nextStep)
   END_RUNG
   // the same network as SCL:
   "Unit1.Em2.ControlNodes".semiAutoSplice."step".action1[1302] := ("Unit1.Em2.ControlNodes".semiAutoSplice.sequence.status.currentStep = #JOB_13_STEP_02) AND "Unit1.Em2.ControlNodes".semiAutoSplice.sequence.status.seqActive;
   "Unit1.Em2.ControlNodes".semiAutoSplice."step".transition1[1302] := ("Unit1.Em2.ControlNodes".semiAutoSplice.sequence.status.currentStep = #JOB_13_STEP_02) AND "Unit1.Em2.ControlNodes".semiAutoSplice.sequence.status.seqActive;
   #statTonTimer[1302].TON(IN := ("Unit1.Em2.ControlNodes".semiAutoSplice.sequence.status.currentStep = #JOB_13_STEP_02) AND "Unit1.Em2.ControlNodes".semiAutoSplice.sequence.status.seqActive AND "Unit1.Em2.ControlNodes".semiAutoSplice."step".transition1[1302],
                           PT := #SeqDelayTime);
   IF #statTonTimer[1302].Q THEN
       "Unit1.Em2.ControlNodes".semiAutoSplice.sequence.status.nextStep := #JOB_13_STEP_03;
   END_IF;
END_REGION

REGION Network 58: Step[1303] : Pad Btm Home (Down)
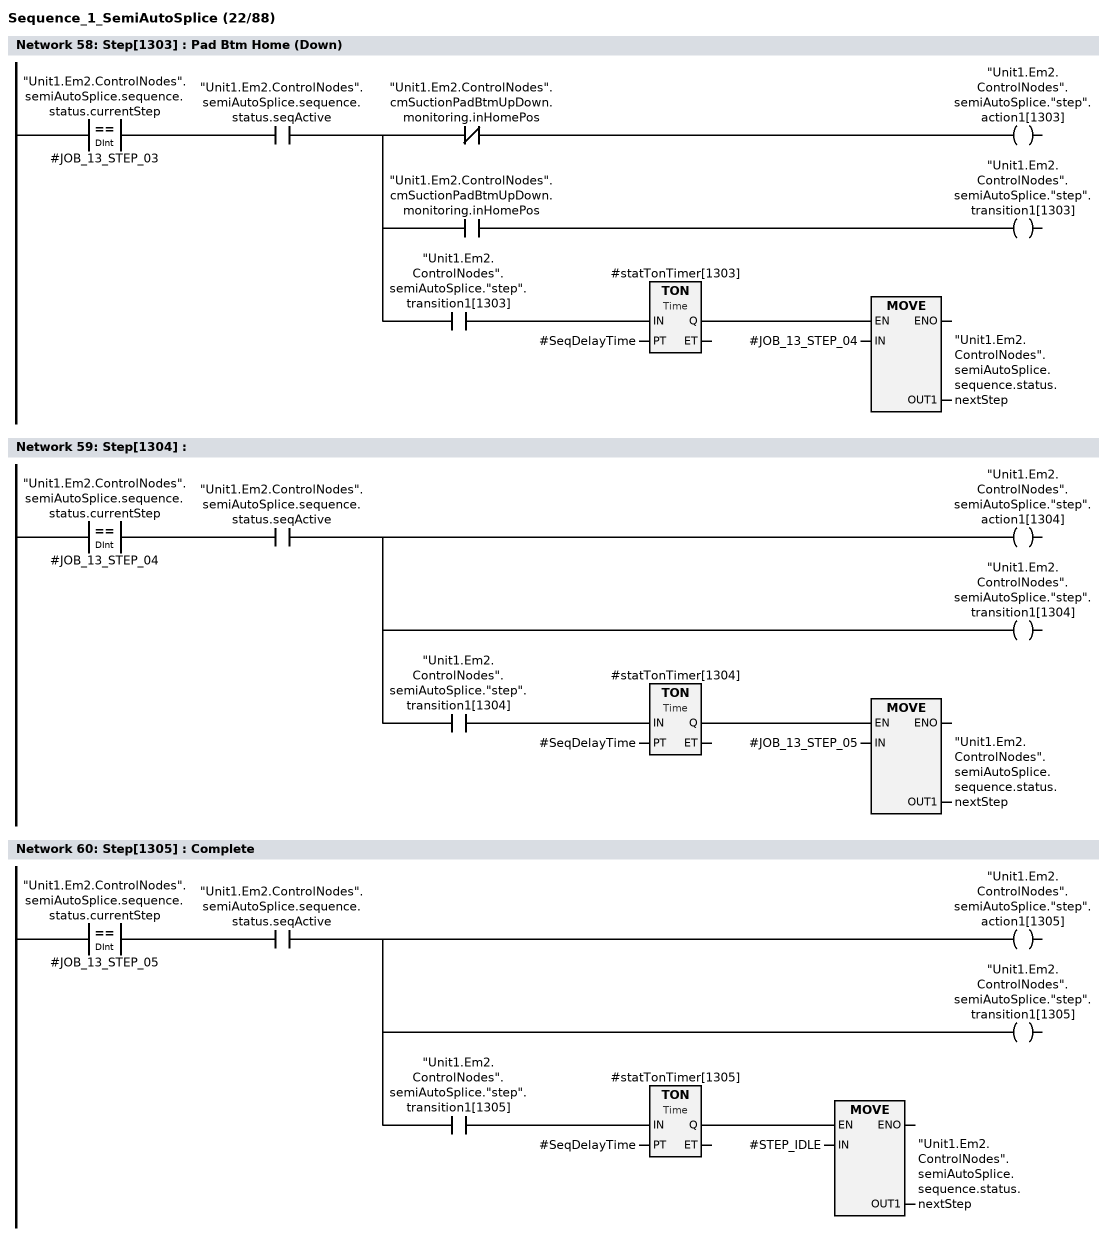
   RUNG wire#powerrail
      { S7_Templates := "SrcType := DInt" } EQ_Contact(in1 := "Unit1.Em2.ControlNodes".semiAutoSplice.sequence.status.currentStep, in2 := #JOB_13_STEP_03)
      Contact( "Unit1.Em2.ControlNodes".semiAutoSplice.sequence.status.seqActive )
      wire#w1
      I_Contact( "Unit1.Em2.ControlNodes".cmSuctionPadBtmUpDown.monitoring.inHomePos )
      Coil( "Unit1.Em2.ControlNodes".semiAutoSplice."step".action1[1303] )
   END_RUNG
   RUNG wire#w1
      Contact( "Unit1.Em2.ControlNodes".cmSuctionPadBtmUpDown.monitoring.inHomePos )
      Coil( "Unit1.Em2.ControlNodes".semiAutoSplice."step".transition1[1303] )
   END_RUNG
   RUNG wire#w1
      Contact( "Unit1.Em2.ControlNodes".semiAutoSplice."step".transition1[1303] )
      { S7_Templates := "time_type := Time" } #statTonTimer[1303].TON(pt := #SeqDelayTime, et =>)
      Move(in := #JOB_13_STEP_04, out1 => "Unit1.Em2.ControlNodes".semiAutoSplice.sequence.status.nextStep)
   END_RUNG
   // the same network as SCL:
   #_w1 := ("Unit1.Em2.ControlNodes".semiAutoSplice.sequence.status.currentStep = #JOB_13_STEP_03) AND "Unit1.Em2.ControlNodes".semiAutoSplice.sequence.status.seqActive;
   "Unit1.Em2.ControlNodes".semiAutoSplice."step".action1[1303] := #_w1 AND NOT "Unit1.Em2.ControlNodes".cmSuctionPadBtmUpDown.monitoring.inHomePos;
   "Unit1.Em2.ControlNodes".semiAutoSplice."step".transition1[1303] := #_w1 AND "Unit1.Em2.ControlNodes".cmSuctionPadBtmUpDown.monitoring.inHomePos;
   #statTonTimer[1303].TON(IN := #_w1 AND "Unit1.Em2.ControlNodes".semiAutoSplice."step".transition1[1303],
                           PT := #SeqDelayTime);
   IF #statTonTimer[1303].Q THEN
       "Unit1.Em2.ControlNodes".semiAutoSplice.sequence.status.nextStep := #JOB_13_STEP_04;
   END_IF;
END_REGION

REGION Network 59: Step[1304] :
   RUNG wire#powerrail
      { S7_Templates := "SrcType := DInt" } EQ_Contact(in1 := "Unit1.Em2.ControlNodes".semiAutoSplice.sequence.status.currentStep, in2 := #JOB_13_STEP_04)
      Contact( "Unit1.Em2.ControlNodes".semiAutoSplice.sequence.status.seqActive )
      wire#w1
      Coil( "Unit1.Em2.ControlNodes".semiAutoSplice."step".action1[1304] )
   END_RUNG
   RUNG wire#w1
      Coil( "Unit1.Em2.ControlNodes".semiAutoSplice."step".transition1[1304] )
   END_RUNG
   RUNG wire#w1
      Contact( "Unit1.Em2.ControlNodes".semiAutoSplice."step".transition1[1304] )
      { S7_Templates := "time_type := Time" } #statTonTimer[1304].TON(pt := #SeqDelayTime, et =>)
      Move(in := #JOB_13_STEP_05, out1 => "Unit1.Em2.ControlNodes".semiAutoSplice.sequence.status.nextStep)
   END_RUNG
   // the same network as SCL:
   "Unit1.Em2.ControlNodes".semiAutoSplice."step".action1[1304] := ("Unit1.Em2.ControlNodes".semiAutoSplice.sequence.status.currentStep = #JOB_13_STEP_04) AND "Unit1.Em2.ControlNodes".semiAutoSplice.sequence.status.seqActive;
   "Unit1.Em2.ControlNodes".semiAutoSplice."step".transition1[1304] := ("Unit1.Em2.ControlNodes".semiAutoSplice.sequence.status.currentStep = #JOB_13_STEP_04) AND "Unit1.Em2.ControlNodes".semiAutoSplice.sequence.status.seqActive;
   #statTonTimer[1304].TON(IN := ("Unit1.Em2.ControlNodes".semiAutoSplice.sequence.status.currentStep = #JOB_13_STEP_04) AND "Unit1.Em2.ControlNodes".semiAutoSplice.sequence.status.seqActive AND "Unit1.Em2.ControlNodes".semiAutoSplice."step".transition1[1304],
                           PT := #SeqDelayTime);
   IF #statTonTimer[1304].Q THEN
       "Unit1.Em2.ControlNodes".semiAutoSplice.sequence.status.nextStep := #JOB_13_STEP_05;
   END_IF;
END_REGION

REGION Network 60: Step[1305] : Complete
   RUNG wire#powerrail
      { S7_Templates := "SrcType := DInt" } EQ_Contact(in1 := "Unit1.Em2.ControlNodes".semiAutoSplice.sequence.status.currentStep, in2 := #JOB_13_STEP_05)
      Contact( "Unit1.Em2.ControlNodes".semiAutoSplice.sequence.status.seqActive )
      wire#w1
      Coil( "Unit1.Em2.ControlNodes".semiAutoSplice."step".action1[1305] )
   END_RUNG
   RUNG wire#w1
      Coil( "Unit1.Em2.ControlNodes".semiAutoSplice."step".transition1[1305] )
   END_RUNG
   RUNG wire#w1
      Contact( "Unit1.Em2.ControlNodes".semiAutoSplice."step".transition1[1305] )
      { S7_Templates := "time_type := Time" } #statTonTimer[1305].TON(pt := #SeqDelayTime, et =>)
      Move(in := #STEP_IDLE, out1 => "Unit1.Em2.ControlNodes".semiAutoSplice.sequence.status.nextStep)
   END_RUNG
   // the same network as SCL:
   "Unit1.Em2.ControlNodes".semiAutoSplice."step".action1[1305] := ("Unit1.Em2.ControlNodes".semiAutoSplice.sequence.status.currentStep = #JOB_13_STEP_05) AND "Unit1.Em2.ControlNodes".semiAutoSplice.sequence.status.seqActive;
   "Unit1.Em2.ControlNodes".semiAutoSplice."step".transition1[1305] := ("Unit1.Em2.ControlNodes".semiAutoSplice.sequence.status.currentStep = #JOB_13_STEP_05) AND "Unit1.Em2.ControlNodes".semiAutoSplice.sequence.status.seqActive;
   #statTonTimer[1305].TON(IN := ("Unit1.Em2.ControlNodes".semiAutoSplice.sequence.status.currentStep = #JOB_13_STEP_05) AND "Unit1.Em2.ControlNodes".semiAutoSplice.sequence.status.seqActive AND "Unit1.Em2.ControlNodes".semiAutoSplice."step".transition1[1305],
                           PT := #SeqDelayTime);
   IF #statTonTimer[1305].Q THEN
       "Unit1.Em2.ControlNodes".semiAutoSplice.sequence.status.nextStep := #STEP_IDLE;
   END_IF;
END_REGION

REGION Network 61: Step[1401] : Head rotate Btm work (FWD)
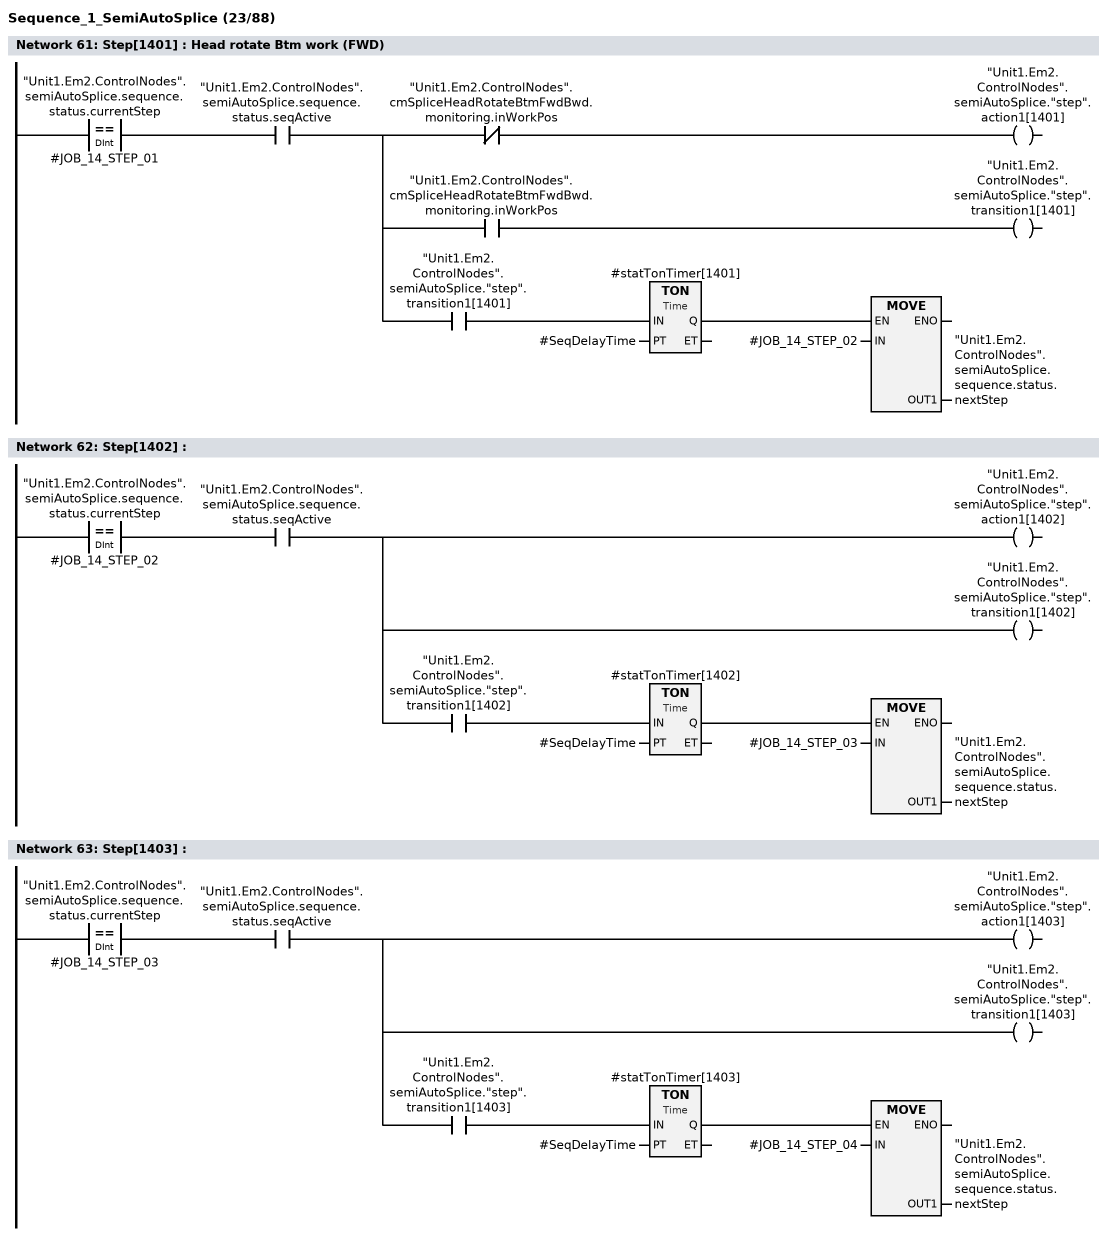
   RUNG wire#powerrail
      { S7_Templates := "SrcType := DInt" } EQ_Contact(in1 := "Unit1.Em2.ControlNodes".semiAutoSplice.sequence.status.currentStep, in2 := #JOB_14_STEP_01)
      Contact( "Unit1.Em2.ControlNodes".semiAutoSplice.sequence.status.seqActive )
      wire#w1
      I_Contact( "Unit1.Em2.ControlNodes".cmSpliceHeadRotateBtmFwdBwd.monitoring.inWorkPos )
      Coil( "Unit1.Em2.ControlNodes".semiAutoSplice."step".action1[1401] )
   END_RUNG
   RUNG wire#w1
      Contact( "Unit1.Em2.ControlNodes".cmSpliceHeadRotateBtmFwdBwd.monitoring.inWorkPos )
      Coil( "Unit1.Em2.ControlNodes".semiAutoSplice."step".transition1[1401] )
   END_RUNG
   RUNG wire#w1
      Contact( "Unit1.Em2.ControlNodes".semiAutoSplice."step".transition1[1401] )
      { S7_Templates := "time_type := Time" } #statTonTimer[1401].TON(pt := #SeqDelayTime, et =>)
      Move(in := #JOB_14_STEP_02, out1 => "Unit1.Em2.ControlNodes".semiAutoSplice.sequence.status.nextStep)
   END_RUNG
   // the same network as SCL:
   #_w1 := ("Unit1.Em2.ControlNodes".semiAutoSplice.sequence.status.currentStep = #JOB_14_STEP_01) AND "Unit1.Em2.ControlNodes".semiAutoSplice.sequence.status.seqActive;
   "Unit1.Em2.ControlNodes".semiAutoSplice."step".action1[1401] := #_w1 AND NOT "Unit1.Em2.ControlNodes".cmSpliceHeadRotateBtmFwdBwd.monitoring.inWorkPos;
   "Unit1.Em2.ControlNodes".semiAutoSplice."step".transition1[1401] := #_w1 AND "Unit1.Em2.ControlNodes".cmSpliceHeadRotateBtmFwdBwd.monitoring.inWorkPos;
   #statTonTimer[1401].TON(IN := #_w1 AND "Unit1.Em2.ControlNodes".semiAutoSplice."step".transition1[1401],
                           PT := #SeqDelayTime);
   IF #statTonTimer[1401].Q THEN
       "Unit1.Em2.ControlNodes".semiAutoSplice.sequence.status.nextStep := #JOB_14_STEP_02;
   END_IF;
END_REGION

REGION Network 62: Step[1402] :
   RUNG wire#powerrail
      { S7_Templates := "SrcType := DInt" } EQ_Contact(in1 := "Unit1.Em2.ControlNodes".semiAutoSplice.sequence.status.currentStep, in2 := #JOB_14_STEP_02)
      Contact( "Unit1.Em2.ControlNodes".semiAutoSplice.sequence.status.seqActive )
      wire#w1
      Coil( "Unit1.Em2.ControlNodes".semiAutoSplice."step".action1[1402] )
   END_RUNG
   RUNG wire#w1
      Coil( "Unit1.Em2.ControlNodes".semiAutoSplice."step".transition1[1402] )
   END_RUNG
   RUNG wire#w1
      Contact( "Unit1.Em2.ControlNodes".semiAutoSplice."step".transition1[1402] )
      { S7_Templates := "time_type := Time" } #statTonTimer[1402].TON(pt := #SeqDelayTime, et =>)
      Move(in := #JOB_14_STEP_03, out1 => "Unit1.Em2.ControlNodes".semiAutoSplice.sequence.status.nextStep)
   END_RUNG
   // the same network as SCL:
   "Unit1.Em2.ControlNodes".semiAutoSplice."step".action1[1402] := ("Unit1.Em2.ControlNodes".semiAutoSplice.sequence.status.currentStep = #JOB_14_STEP_02) AND "Unit1.Em2.ControlNodes".semiAutoSplice.sequence.status.seqActive;
   "Unit1.Em2.ControlNodes".semiAutoSplice."step".transition1[1402] := ("Unit1.Em2.ControlNodes".semiAutoSplice.sequence.status.currentStep = #JOB_14_STEP_02) AND "Unit1.Em2.ControlNodes".semiAutoSplice.sequence.status.seqActive;
   #statTonTimer[1402].TON(IN := ("Unit1.Em2.ControlNodes".semiAutoSplice.sequence.status.currentStep = #JOB_14_STEP_02) AND "Unit1.Em2.ControlNodes".semiAutoSplice.sequence.status.seqActive AND "Unit1.Em2.ControlNodes".semiAutoSplice."step".transition1[1402],
                           PT := #SeqDelayTime);
   IF #statTonTimer[1402].Q THEN
       "Unit1.Em2.ControlNodes".semiAutoSplice.sequence.status.nextStep := #JOB_14_STEP_03;
   END_IF;
END_REGION

REGION Network 63: Step[1403] :
   RUNG wire#powerrail
      { S7_Templates := "SrcType := DInt" } EQ_Contact(in1 := "Unit1.Em2.ControlNodes".semiAutoSplice.sequence.status.currentStep, in2 := #JOB_14_STEP_03)
      Contact( "Unit1.Em2.ControlNodes".semiAutoSplice.sequence.status.seqActive )
      wire#w1
      Coil( "Unit1.Em2.ControlNodes".semiAutoSplice."step".action1[1403] )
   END_RUNG
   RUNG wire#w1
      Coil( "Unit1.Em2.ControlNodes".semiAutoSplice."step".transition1[1403] )
   END_RUNG
   RUNG wire#w1
      Contact( "Unit1.Em2.ControlNodes".semiAutoSplice."step".transition1[1403] )
      { S7_Templates := "time_type := Time" } #statTonTimer[1403].TON(pt := #SeqDelayTime, et =>)
      Move(in := #JOB_14_STEP_04, out1 => "Unit1.Em2.ControlNodes".semiAutoSplice.sequence.status.nextStep)
   END_RUNG
   // the same network as SCL:
   "Unit1.Em2.ControlNodes".semiAutoSplice."step".action1[1403] := ("Unit1.Em2.ControlNodes".semiAutoSplice.sequence.status.currentStep = #JOB_14_STEP_03) AND "Unit1.Em2.ControlNodes".semiAutoSplice.sequence.status.seqActive;
   "Unit1.Em2.ControlNodes".semiAutoSplice."step".transition1[1403] := ("Unit1.Em2.ControlNodes".semiAutoSplice.sequence.status.currentStep = #JOB_14_STEP_03) AND "Unit1.Em2.ControlNodes".semiAutoSplice.sequence.status.seqActive;
   #statTonTimer[1403].TON(IN := ("Unit1.Em2.ControlNodes".semiAutoSplice.sequence.status.currentStep = #JOB_14_STEP_03) AND "Unit1.Em2.ControlNodes".semiAutoSplice.sequence.status.seqActive AND "Unit1.Em2.ControlNodes".semiAutoSplice."step".transition1[1403],
                           PT := #SeqDelayTime);
   IF #statTonTimer[1403].Q THEN
       "Unit1.Em2.ControlNodes".semiAutoSplice.sequence.status.nextStep := #JOB_14_STEP_04;
   END_IF;
END_REGION

REGION Network 64: Step[1404] :
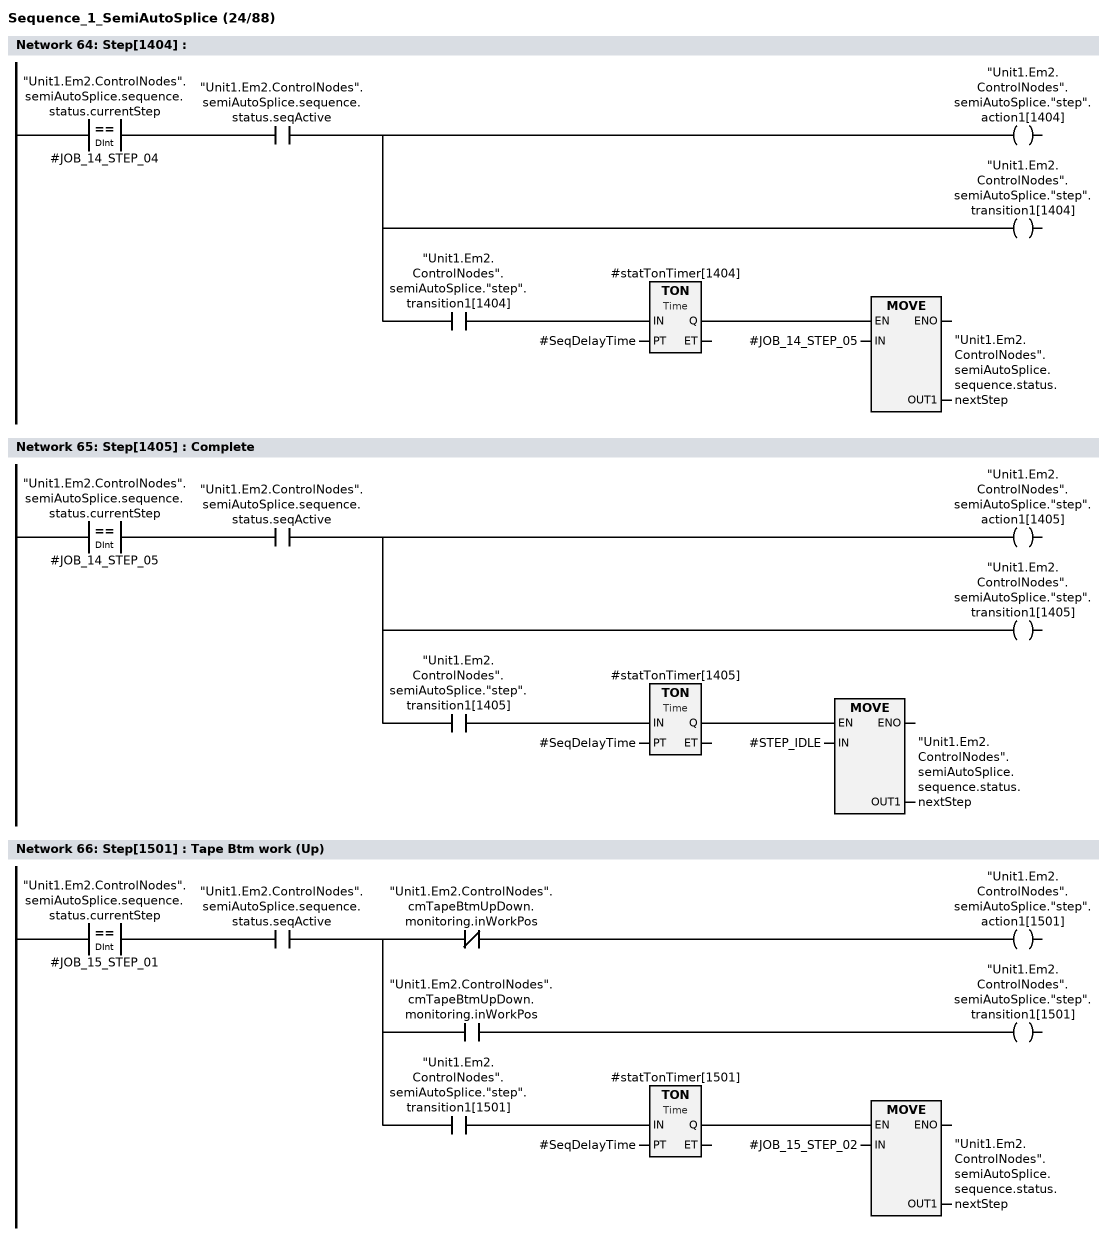
   RUNG wire#powerrail
      { S7_Templates := "SrcType := DInt" } EQ_Contact(in1 := "Unit1.Em2.ControlNodes".semiAutoSplice.sequence.status.currentStep, in2 := #JOB_14_STEP_04)
      Contact( "Unit1.Em2.ControlNodes".semiAutoSplice.sequence.status.seqActive )
      wire#w1
      Coil( "Unit1.Em2.ControlNodes".semiAutoSplice."step".action1[1404] )
   END_RUNG
   RUNG wire#w1
      Coil( "Unit1.Em2.ControlNodes".semiAutoSplice."step".transition1[1404] )
   END_RUNG
   RUNG wire#w1
      Contact( "Unit1.Em2.ControlNodes".semiAutoSplice."step".transition1[1404] )
      { S7_Templates := "time_type := Time" } #statTonTimer[1404].TON(pt := #SeqDelayTime, et =>)
      Move(in := #JOB_14_STEP_05, out1 => "Unit1.Em2.ControlNodes".semiAutoSplice.sequence.status.nextStep)
   END_RUNG
   // the same network as SCL:
   "Unit1.Em2.ControlNodes".semiAutoSplice."step".action1[1404] := ("Unit1.Em2.ControlNodes".semiAutoSplice.sequence.status.currentStep = #JOB_14_STEP_04) AND "Unit1.Em2.ControlNodes".semiAutoSplice.sequence.status.seqActive;
   "Unit1.Em2.ControlNodes".semiAutoSplice."step".transition1[1404] := ("Unit1.Em2.ControlNodes".semiAutoSplice.sequence.status.currentStep = #JOB_14_STEP_04) AND "Unit1.Em2.ControlNodes".semiAutoSplice.sequence.status.seqActive;
   #statTonTimer[1404].TON(IN := ("Unit1.Em2.ControlNodes".semiAutoSplice.sequence.status.currentStep = #JOB_14_STEP_04) AND "Unit1.Em2.ControlNodes".semiAutoSplice.sequence.status.seqActive AND "Unit1.Em2.ControlNodes".semiAutoSplice."step".transition1[1404],
                           PT := #SeqDelayTime);
   IF #statTonTimer[1404].Q THEN
       "Unit1.Em2.ControlNodes".semiAutoSplice.sequence.status.nextStep := #JOB_14_STEP_05;
   END_IF;
END_REGION

REGION Network 65: Step[1405] : Complete
   RUNG wire#powerrail
      { S7_Templates := "SrcType := DInt" } EQ_Contact(in1 := "Unit1.Em2.ControlNodes".semiAutoSplice.sequence.status.currentStep, in2 := #JOB_14_STEP_05)
      Contact( "Unit1.Em2.ControlNodes".semiAutoSplice.sequence.status.seqActive )
      wire#w1
      Coil( "Unit1.Em2.ControlNodes".semiAutoSplice."step".action1[1405] )
   END_RUNG
   RUNG wire#w1
      Coil( "Unit1.Em2.ControlNodes".semiAutoSplice."step".transition1[1405] )
   END_RUNG
   RUNG wire#w1
      Contact( "Unit1.Em2.ControlNodes".semiAutoSplice."step".transition1[1405] )
      { S7_Templates := "time_type := Time" } #statTonTimer[1405].TON(pt := #SeqDelayTime, et =>)
      Move(in := #STEP_IDLE, out1 => "Unit1.Em2.ControlNodes".semiAutoSplice.sequence.status.nextStep)
   END_RUNG
   // the same network as SCL:
   "Unit1.Em2.ControlNodes".semiAutoSplice."step".action1[1405] := ("Unit1.Em2.ControlNodes".semiAutoSplice.sequence.status.currentStep = #JOB_14_STEP_05) AND "Unit1.Em2.ControlNodes".semiAutoSplice.sequence.status.seqActive;
   "Unit1.Em2.ControlNodes".semiAutoSplice."step".transition1[1405] := ("Unit1.Em2.ControlNodes".semiAutoSplice.sequence.status.currentStep = #JOB_14_STEP_05) AND "Unit1.Em2.ControlNodes".semiAutoSplice.sequence.status.seqActive;
   #statTonTimer[1405].TON(IN := ("Unit1.Em2.ControlNodes".semiAutoSplice.sequence.status.currentStep = #JOB_14_STEP_05) AND "Unit1.Em2.ControlNodes".semiAutoSplice.sequence.status.seqActive AND "Unit1.Em2.ControlNodes".semiAutoSplice."step".transition1[1405],
                           PT := #SeqDelayTime);
   IF #statTonTimer[1405].Q THEN
       "Unit1.Em2.ControlNodes".semiAutoSplice.sequence.status.nextStep := #STEP_IDLE;
   END_IF;
END_REGION

REGION Network 66: Step[1501] : Tape Btm work (Up)
   RUNG wire#powerrail
      { S7_Templates := "SrcType := DInt" } EQ_Contact(in1 := "Unit1.Em2.ControlNodes".semiAutoSplice.sequence.status.currentStep, in2 := #JOB_15_STEP_01)
      Contact( "Unit1.Em2.ControlNodes".semiAutoSplice.sequence.status.seqActive )
      wire#w1
      I_Contact( "Unit1.Em2.ControlNodes".cmTapeBtmUpDown.monitoring.inWorkPos )
      Coil( "Unit1.Em2.ControlNodes".semiAutoSplice."step".action1[1501] )
   END_RUNG
   RUNG wire#w1
      Contact( "Unit1.Em2.ControlNodes".cmTapeBtmUpDown.monitoring.inWorkPos )
      Coil( "Unit1.Em2.ControlNodes".semiAutoSplice."step".transition1[1501] )
   END_RUNG
   RUNG wire#w1
      Contact( "Unit1.Em2.ControlNodes".semiAutoSplice."step".transition1[1501] )
      { S7_Templates := "time_type := Time" } #statTonTimer[1501].TON(pt := #SeqDelayTime, et =>)
      Move(in := #JOB_15_STEP_02, out1 => "Unit1.Em2.ControlNodes".semiAutoSplice.sequence.status.nextStep)
   END_RUNG
   // the same network as SCL:
   #_w1 := ("Unit1.Em2.ControlNodes".semiAutoSplice.sequence.status.currentStep = #JOB_15_STEP_01) AND "Unit1.Em2.ControlNodes".semiAutoSplice.sequence.status.seqActive;
   "Unit1.Em2.ControlNodes".semiAutoSplice."step".action1[1501] := #_w1 AND NOT "Unit1.Em2.ControlNodes".cmTapeBtmUpDown.monitoring.inWorkPos;
   "Unit1.Em2.ControlNodes".semiAutoSplice."step".transition1[1501] := #_w1 AND "Unit1.Em2.ControlNodes".cmTapeBtmUpDown.monitoring.inWorkPos;
   #statTonTimer[1501].TON(IN := #_w1 AND "Unit1.Em2.ControlNodes".semiAutoSplice."step".transition1[1501],
                           PT := #SeqDelayTime);
   IF #statTonTimer[1501].Q THEN
       "Unit1.Em2.ControlNodes".semiAutoSplice.sequence.status.nextStep := #JOB_15_STEP_02;
   END_IF;
END_REGION

REGION Network 67: Step[1502] :
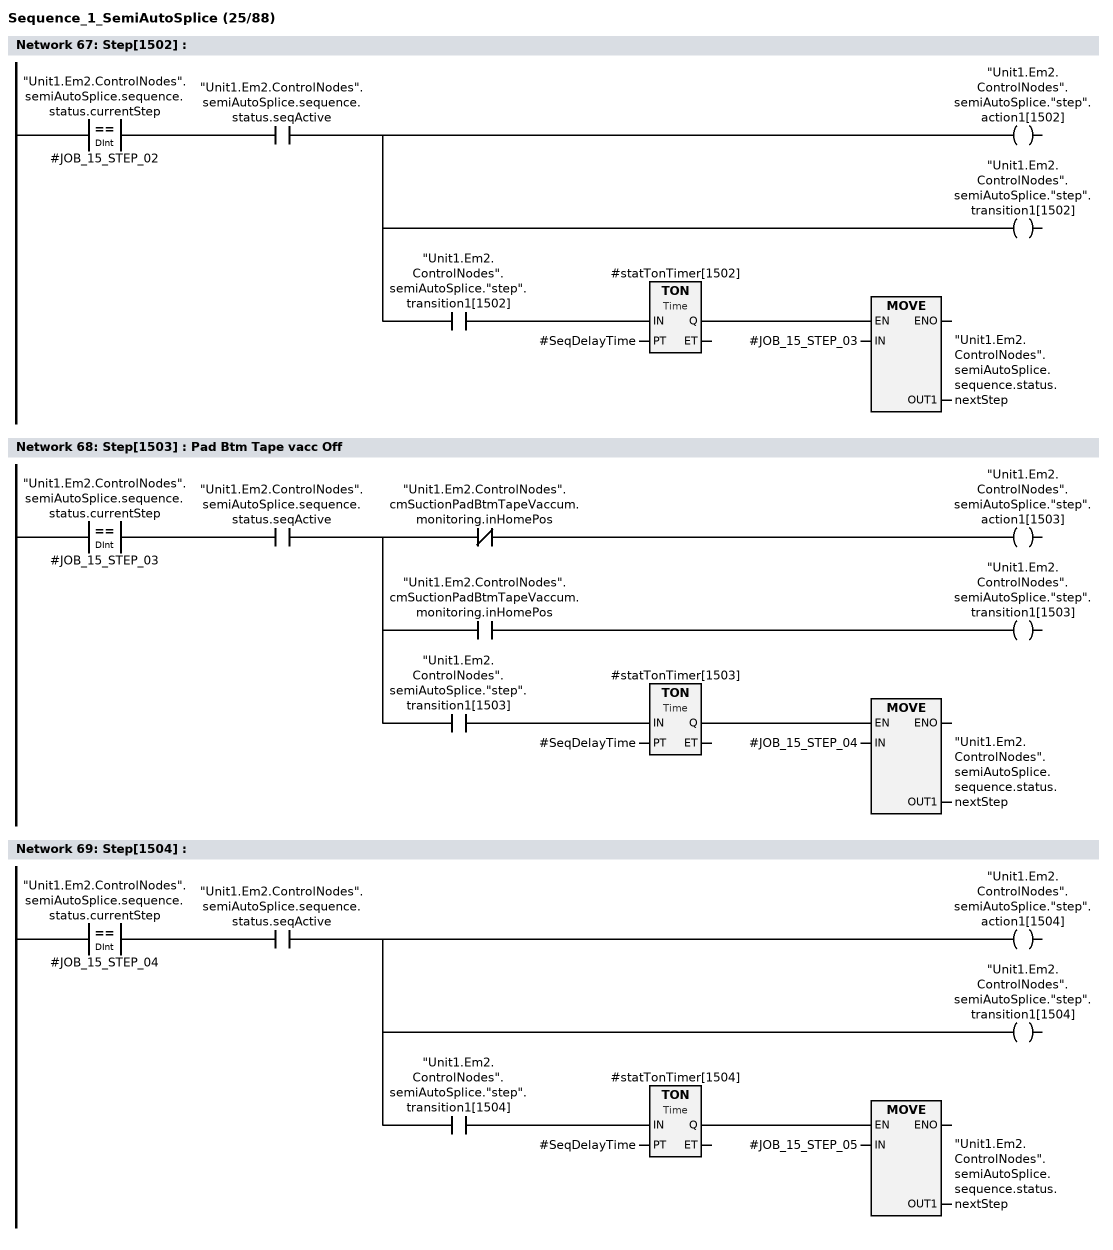
   RUNG wire#powerrail
      { S7_Templates := "SrcType := DInt" } EQ_Contact(in1 := "Unit1.Em2.ControlNodes".semiAutoSplice.sequence.status.currentStep, in2 := #JOB_15_STEP_02)
      Contact( "Unit1.Em2.ControlNodes".semiAutoSplice.sequence.status.seqActive )
      wire#w1
      Coil( "Unit1.Em2.ControlNodes".semiAutoSplice."step".action1[1502] )
   END_RUNG
   RUNG wire#w1
      Coil( "Unit1.Em2.ControlNodes".semiAutoSplice."step".transition1[1502] )
   END_RUNG
   RUNG wire#w1
      Contact( "Unit1.Em2.ControlNodes".semiAutoSplice."step".transition1[1502] )
      { S7_Templates := "time_type := Time" } #statTonTimer[1502].TON(pt := #SeqDelayTime, et =>)
      Move(in := #JOB_15_STEP_03, out1 => "Unit1.Em2.ControlNodes".semiAutoSplice.sequence.status.nextStep)
   END_RUNG
   // the same network as SCL:
   "Unit1.Em2.ControlNodes".semiAutoSplice."step".action1[1502] := ("Unit1.Em2.ControlNodes".semiAutoSplice.sequence.status.currentStep = #JOB_15_STEP_02) AND "Unit1.Em2.ControlNodes".semiAutoSplice.sequence.status.seqActive;
   "Unit1.Em2.ControlNodes".semiAutoSplice."step".transition1[1502] := ("Unit1.Em2.ControlNodes".semiAutoSplice.sequence.status.currentStep = #JOB_15_STEP_02) AND "Unit1.Em2.ControlNodes".semiAutoSplice.sequence.status.seqActive;
   #statTonTimer[1502].TON(IN := ("Unit1.Em2.ControlNodes".semiAutoSplice.sequence.status.currentStep = #JOB_15_STEP_02) AND "Unit1.Em2.ControlNodes".semiAutoSplice.sequence.status.seqActive AND "Unit1.Em2.ControlNodes".semiAutoSplice."step".transition1[1502],
                           PT := #SeqDelayTime);
   IF #statTonTimer[1502].Q THEN
       "Unit1.Em2.ControlNodes".semiAutoSplice.sequence.status.nextStep := #JOB_15_STEP_03;
   END_IF;
END_REGION

REGION Network 68: Step[1503] : Pad Btm Tape vacc Off
   RUNG wire#powerrail
      { S7_Templates := "SrcType := DInt" } EQ_Contact(in1 := "Unit1.Em2.ControlNodes".semiAutoSplice.sequence.status.currentStep, in2 := #JOB_15_STEP_03)
      Contact( "Unit1.Em2.ControlNodes".semiAutoSplice.sequence.status.seqActive )
      wire#w1
      I_Contact( "Unit1.Em2.ControlNodes".cmSuctionPadBtmTapeVaccum.monitoring.inHomePos )
      Coil( "Unit1.Em2.ControlNodes".semiAutoSplice."step".action1[1503] )
   END_RUNG
   RUNG wire#w1
      Contact( "Unit1.Em2.ControlNodes".cmSuctionPadBtmTapeVaccum.monitoring.inHomePos )
      Coil( "Unit1.Em2.ControlNodes".semiAutoSplice."step".transition1[1503] )
   END_RUNG
   RUNG wire#w1
      Contact( "Unit1.Em2.ControlNodes".semiAutoSplice."step".transition1[1503] )
      { S7_Templates := "time_type := Time" } #statTonTimer[1503].TON(pt := #SeqDelayTime, et =>)
      Move(in := #JOB_15_STEP_04, out1 => "Unit1.Em2.ControlNodes".semiAutoSplice.sequence.status.nextStep)
   END_RUNG
   // the same network as SCL:
   #_w1 := ("Unit1.Em2.ControlNodes".semiAutoSplice.sequence.status.currentStep = #JOB_15_STEP_03) AND "Unit1.Em2.ControlNodes".semiAutoSplice.sequence.status.seqActive;
   "Unit1.Em2.ControlNodes".semiAutoSplice."step".action1[1503] := #_w1 AND NOT "Unit1.Em2.ControlNodes".cmSuctionPadBtmTapeVaccum.monitoring.inHomePos;
   "Unit1.Em2.ControlNodes".semiAutoSplice."step".transition1[1503] := #_w1 AND "Unit1.Em2.ControlNodes".cmSuctionPadBtmTapeVaccum.monitoring.inHomePos;
   #statTonTimer[1503].TON(IN := #_w1 AND "Unit1.Em2.ControlNodes".semiAutoSplice."step".transition1[1503],
                           PT := #SeqDelayTime);
   IF #statTonTimer[1503].Q THEN
       "Unit1.Em2.ControlNodes".semiAutoSplice.sequence.status.nextStep := #JOB_15_STEP_04;
   END_IF;
END_REGION

REGION Network 69: Step[1504] :
   RUNG wire#powerrail
      { S7_Templates := "SrcType := DInt" } EQ_Contact(in1 := "Unit1.Em2.ControlNodes".semiAutoSplice.sequence.status.currentStep, in2 := #JOB_15_STEP_04)
      Contact( "Unit1.Em2.ControlNodes".semiAutoSplice.sequence.status.seqActive )
      wire#w1
      Coil( "Unit1.Em2.ControlNodes".semiAutoSplice."step".action1[1504] )
   END_RUNG
   RUNG wire#w1
      Coil( "Unit1.Em2.ControlNodes".semiAutoSplice."step".transition1[1504] )
   END_RUNG
   RUNG wire#w1
      Contact( "Unit1.Em2.ControlNodes".semiAutoSplice."step".transition1[1504] )
      { S7_Templates := "time_type := Time" } #statTonTimer[1504].TON(pt := #SeqDelayTime, et =>)
      Move(in := #JOB_15_STEP_05, out1 => "Unit1.Em2.ControlNodes".semiAutoSplice.sequence.status.nextStep)
   END_RUNG
   // the same network as SCL:
   "Unit1.Em2.ControlNodes".semiAutoSplice."step".action1[1504] := ("Unit1.Em2.ControlNodes".semiAutoSplice.sequence.status.currentStep = #JOB_15_STEP_04) AND "Unit1.Em2.ControlNodes".semiAutoSplice.sequence.status.seqActive;
   "Unit1.Em2.ControlNodes".semiAutoSplice."step".transition1[1504] := ("Unit1.Em2.ControlNodes".semiAutoSplice.sequence.status.currentStep = #JOB_15_STEP_04) AND "Unit1.Em2.ControlNodes".semiAutoSplice.sequence.status.seqActive;
   #statTonTimer[1504].TON(IN := ("Unit1.Em2.ControlNodes".semiAutoSplice.sequence.status.currentStep = #JOB_15_STEP_04) AND "Unit1.Em2.ControlNodes".semiAutoSplice.sequence.status.seqActive AND "Unit1.Em2.ControlNodes".semiAutoSplice."step".transition1[1504],
                           PT := #SeqDelayTime);
   IF #statTonTimer[1504].Q THEN
       "Unit1.Em2.ControlNodes".semiAutoSplice.sequence.status.nextStep := #JOB_15_STEP_05;
   END_IF;
END_REGION

REGION Network 70: Step[1505] : Tape Btm home (Down)
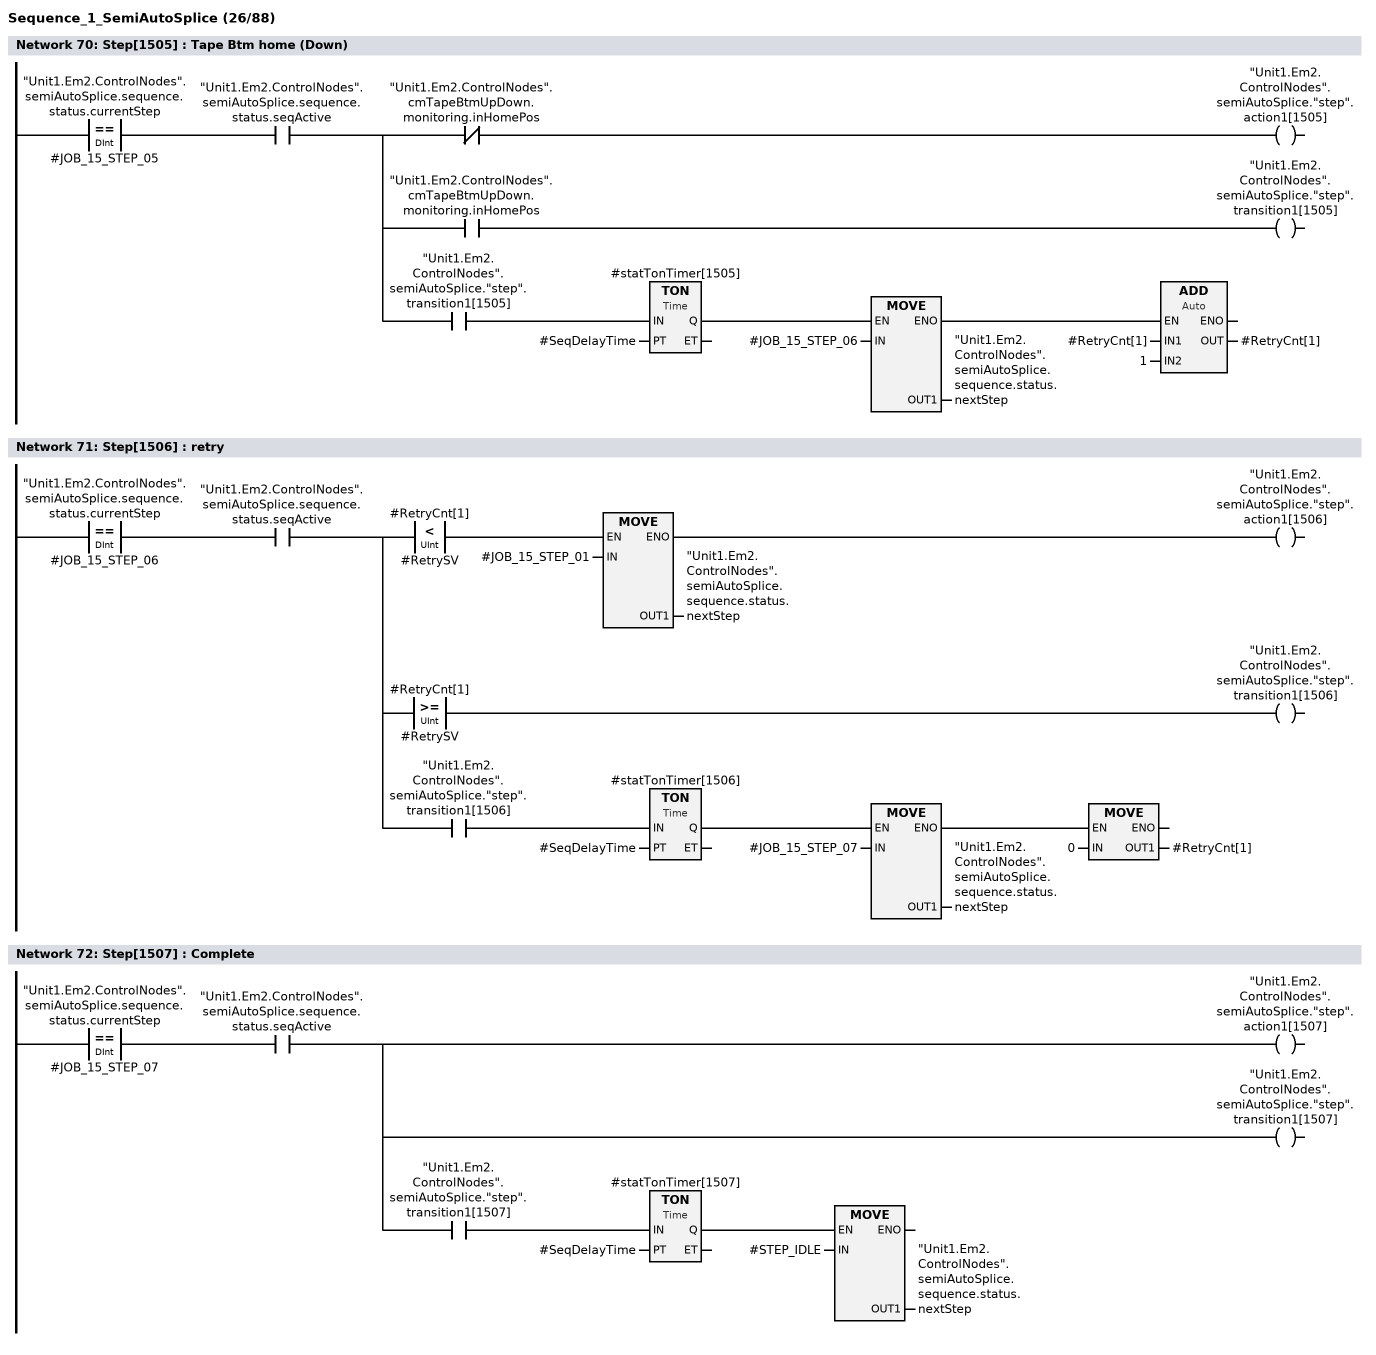
   RUNG wire#powerrail
      { S7_Templates := "SrcType := DInt" } EQ_Contact(in1 := "Unit1.Em2.ControlNodes".semiAutoSplice.sequence.status.currentStep, in2 := #JOB_15_STEP_05)
      Contact( "Unit1.Em2.ControlNodes".semiAutoSplice.sequence.status.seqActive )
      wire#w1
      I_Contact( "Unit1.Em2.ControlNodes".cmTapeBtmUpDown.monitoring.inHomePos )
      Coil( "Unit1.Em2.ControlNodes".semiAutoSplice."step".action1[1505] )
   END_RUNG
   RUNG wire#w1
      Contact( "Unit1.Em2.ControlNodes".cmTapeBtmUpDown.monitoring.inHomePos )
      Coil( "Unit1.Em2.ControlNodes".semiAutoSplice."step".transition1[1505] )
   END_RUNG
   RUNG wire#w1
      Contact( "Unit1.Em2.ControlNodes".semiAutoSplice."step".transition1[1505] )
      { S7_Templates := "time_type := Time" } #statTonTimer[1505].TON(pt := #SeqDelayTime, et =>)
      Move(in := #JOB_15_STEP_06, out1 => "Unit1.Em2.ControlNodes".semiAutoSplice.sequence.status.nextStep)
      Add(in1 := #RetryCnt[1], in2 := 1, out => #RetryCnt[1])
   END_RUNG
   // the same network as SCL:
   #_w1 := ("Unit1.Em2.ControlNodes".semiAutoSplice.sequence.status.currentStep = #JOB_15_STEP_05) AND "Unit1.Em2.ControlNodes".semiAutoSplice.sequence.status.seqActive;
   "Unit1.Em2.ControlNodes".semiAutoSplice."step".action1[1505] := #_w1 AND NOT "Unit1.Em2.ControlNodes".cmTapeBtmUpDown.monitoring.inHomePos;
   "Unit1.Em2.ControlNodes".semiAutoSplice."step".transition1[1505] := #_w1 AND "Unit1.Em2.ControlNodes".cmTapeBtmUpDown.monitoring.inHomePos;
   #statTonTimer[1505].TON(IN := #_w1 AND "Unit1.Em2.ControlNodes".semiAutoSplice."step".transition1[1505],
                           PT := #SeqDelayTime);
   IF #statTonTimer[1505].Q THEN
       "Unit1.Em2.ControlNodes".semiAutoSplice.sequence.status.nextStep := #JOB_15_STEP_06;
       #RetryCnt[1] := #RetryCnt[1] + 1;
   END_IF;
END_REGION

REGION Network 71: Step[1506] : retry
   RUNG wire#powerrail
      { S7_Templates := "SrcType := DInt" } EQ_Contact(in1 := "Unit1.Em2.ControlNodes".semiAutoSplice.sequence.status.currentStep, in2 := #JOB_15_STEP_06)
      Contact( "Unit1.Em2.ControlNodes".semiAutoSplice.sequence.status.seqActive )
      wire#w1
      { S7_Templates := "SrcType := UInt" } LT_Contact(in1 := #RetryCnt[1], in2 := #RetrySV)
      Move(in := #JOB_15_STEP_01, out1 => "Unit1.Em2.ControlNodes".semiAutoSplice.sequence.status.nextStep)
      Coil( "Unit1.Em2.ControlNodes".semiAutoSplice."step".action1[1506] )
   END_RUNG
   RUNG wire#w1
      { S7_Templates := "SrcType := UInt" } GE_Contact(in1 := #RetryCnt[1], in2 := #RetrySV)
      Coil( "Unit1.Em2.ControlNodes".semiAutoSplice."step".transition1[1506] )
   END_RUNG
   RUNG wire#w1
      Contact( "Unit1.Em2.ControlNodes".semiAutoSplice."step".transition1[1506] )
      { S7_Templates := "time_type := Time" } #statTonTimer[1506].TON(pt := #SeqDelayTime, et =>)
      Move(in := #JOB_15_STEP_07, out1 => "Unit1.Em2.ControlNodes".semiAutoSplice.sequence.status.nextStep)
      Move(in := 0, out1 => #RetryCnt[1])
   END_RUNG
   // the same network as SCL:
   #_w1 := ("Unit1.Em2.ControlNodes".semiAutoSplice.sequence.status.currentStep = #JOB_15_STEP_06) AND "Unit1.Em2.ControlNodes".semiAutoSplice.sequence.status.seqActive;
   #_w2 := #_w1 AND (#RetryCnt[1] < #RetrySV);
   IF #_w2 THEN "Unit1.Em2.ControlNodes".semiAutoSplice.sequence.status.nextStep := #JOB_15_STEP_01; END_IF;
   "Unit1.Em2.ControlNodes".semiAutoSplice."step".action1[1506] := #_w2;
   "Unit1.Em2.ControlNodes".semiAutoSplice."step".transition1[1506] := #_w1 AND (#RetryCnt[1] >= #RetrySV);
   #statTonTimer[1506].TON(IN := #_w1 AND "Unit1.Em2.ControlNodes".semiAutoSplice."step".transition1[1506],
                           PT := #SeqDelayTime);
   IF #statTonTimer[1506].Q THEN
       "Unit1.Em2.ControlNodes".semiAutoSplice.sequence.status.nextStep := #JOB_15_STEP_07;
       #RetryCnt[1] := 0;
   END_IF;
END_REGION

REGION Network 72: Step[1507] : Complete
   RUNG wire#powerrail
      { S7_Templates := "SrcType := DInt" } EQ_Contact(in1 := "Unit1.Em2.ControlNodes".semiAutoSplice.sequence.status.currentStep, in2 := #JOB_15_STEP_07)
      Contact( "Unit1.Em2.ControlNodes".semiAutoSplice.sequence.status.seqActive )
      wire#w1
      Coil( "Unit1.Em2.ControlNodes".semiAutoSplice."step".action1[1507] )
   END_RUNG
   RUNG wire#w1
      Coil( "Unit1.Em2.ControlNodes".semiAutoSplice."step".transition1[1507] )
   END_RUNG
   RUNG wire#w1
      Contact( "Unit1.Em2.ControlNodes".semiAutoSplice."step".transition1[1507] )
      { S7_Templates := "time_type := Time" } #statTonTimer[1507].TON(pt := #SeqDelayTime, et =>)
      Move(in := #STEP_IDLE, out1 => "Unit1.Em2.ControlNodes".semiAutoSplice.sequence.status.nextStep)
   END_RUNG
   // the same network as SCL:
   "Unit1.Em2.ControlNodes".semiAutoSplice."step".action1[1507] := ("Unit1.Em2.ControlNodes".semiAutoSplice.sequence.status.currentStep = #JOB_15_STEP_07) AND "Unit1.Em2.ControlNodes".semiAutoSplice.sequence.status.seqActive;
   "Unit1.Em2.ControlNodes".semiAutoSplice."step".transition1[1507] := ("Unit1.Em2.ControlNodes".semiAutoSplice.sequence.status.currentStep = #JOB_15_STEP_07) AND "Unit1.Em2.ControlNodes".semiAutoSplice.sequence.status.seqActive;
   #statTonTimer[1507].TON(IN := ("Unit1.Em2.ControlNodes".semiAutoSplice.sequence.status.currentStep = #JOB_15_STEP_07) AND "Unit1.Em2.ControlNodes".semiAutoSplice.sequence.status.seqActive AND "Unit1.Em2.ControlNodes".semiAutoSplice."step".transition1[1507],
                           PT := #SeqDelayTime);
   IF #statTonTimer[1507].Q THEN
       "Unit1.Em2.ControlNodes".semiAutoSplice.sequence.status.nextStep := #STEP_IDLE;
   END_IF;
END_REGION

REGION Network 73: Step[1601] : Head rotate Btm home (BWD)
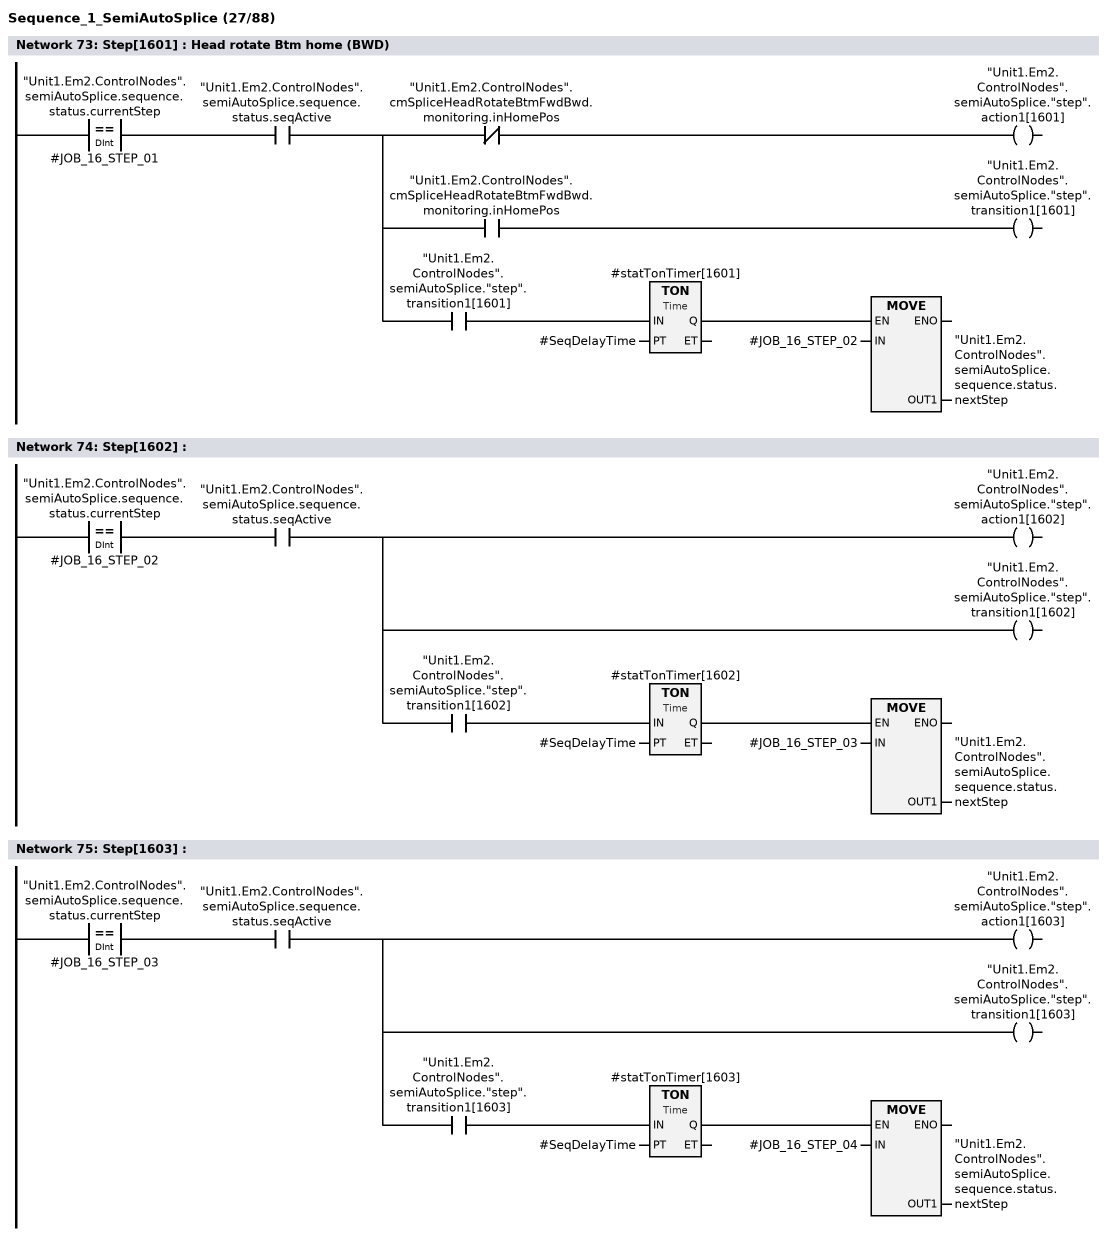
   RUNG wire#powerrail
      { S7_Templates := "SrcType := DInt" } EQ_Contact(in1 := "Unit1.Em2.ControlNodes".semiAutoSplice.sequence.status.currentStep, in2 := #JOB_16_STEP_01)
      Contact( "Unit1.Em2.ControlNodes".semiAutoSplice.sequence.status.seqActive )
      wire#w1
      I_Contact( "Unit1.Em2.ControlNodes".cmSpliceHeadRotateBtmFwdBwd.monitoring.inHomePos )
      Coil( "Unit1.Em2.ControlNodes".semiAutoSplice."step".action1[1601] )
   END_RUNG
   RUNG wire#w1
      Contact( "Unit1.Em2.ControlNodes".cmSpliceHeadRotateBtmFwdBwd.monitoring.inHomePos )
      Coil( "Unit1.Em2.ControlNodes".semiAutoSplice."step".transition1[1601] )
   END_RUNG
   RUNG wire#w1
      Contact( "Unit1.Em2.ControlNodes".semiAutoSplice."step".transition1[1601] )
      { S7_Templates := "time_type := Time" } #statTonTimer[1601].TON(pt := #SeqDelayTime, et =>)
      Move(in := #JOB_16_STEP_02, out1 => "Unit1.Em2.ControlNodes".semiAutoSplice.sequence.status.nextStep)
   END_RUNG
   // the same network as SCL:
   #_w1 := ("Unit1.Em2.ControlNodes".semiAutoSplice.sequence.status.currentStep = #JOB_16_STEP_01) AND "Unit1.Em2.ControlNodes".semiAutoSplice.sequence.status.seqActive;
   "Unit1.Em2.ControlNodes".semiAutoSplice."step".action1[1601] := #_w1 AND NOT "Unit1.Em2.ControlNodes".cmSpliceHeadRotateBtmFwdBwd.monitoring.inHomePos;
   "Unit1.Em2.ControlNodes".semiAutoSplice."step".transition1[1601] := #_w1 AND "Unit1.Em2.ControlNodes".cmSpliceHeadRotateBtmFwdBwd.monitoring.inHomePos;
   #statTonTimer[1601].TON(IN := #_w1 AND "Unit1.Em2.ControlNodes".semiAutoSplice."step".transition1[1601],
                           PT := #SeqDelayTime);
   IF #statTonTimer[1601].Q THEN
       "Unit1.Em2.ControlNodes".semiAutoSplice.sequence.status.nextStep := #JOB_16_STEP_02;
   END_IF;
END_REGION

REGION Network 74: Step[1602] :
   RUNG wire#powerrail
      { S7_Templates := "SrcType := DInt" } EQ_Contact(in1 := "Unit1.Em2.ControlNodes".semiAutoSplice.sequence.status.currentStep, in2 := #JOB_16_STEP_02)
      Contact( "Unit1.Em2.ControlNodes".semiAutoSplice.sequence.status.seqActive )
      wire#w1
      Coil( "Unit1.Em2.ControlNodes".semiAutoSplice."step".action1[1602] )
   END_RUNG
   RUNG wire#w1
      Coil( "Unit1.Em2.ControlNodes".semiAutoSplice."step".transition1[1602] )
   END_RUNG
   RUNG wire#w1
      Contact( "Unit1.Em2.ControlNodes".semiAutoSplice."step".transition1[1602] )
      { S7_Templates := "time_type := Time" } #statTonTimer[1602].TON(pt := #SeqDelayTime, et =>)
      Move(in := #JOB_16_STEP_03, out1 => "Unit1.Em2.ControlNodes".semiAutoSplice.sequence.status.nextStep)
   END_RUNG
   // the same network as SCL:
   "Unit1.Em2.ControlNodes".semiAutoSplice."step".action1[1602] := ("Unit1.Em2.ControlNodes".semiAutoSplice.sequence.status.currentStep = #JOB_16_STEP_02) AND "Unit1.Em2.ControlNodes".semiAutoSplice.sequence.status.seqActive;
   "Unit1.Em2.ControlNodes".semiAutoSplice."step".transition1[1602] := ("Unit1.Em2.ControlNodes".semiAutoSplice.sequence.status.currentStep = #JOB_16_STEP_02) AND "Unit1.Em2.ControlNodes".semiAutoSplice.sequence.status.seqActive;
   #statTonTimer[1602].TON(IN := ("Unit1.Em2.ControlNodes".semiAutoSplice.sequence.status.currentStep = #JOB_16_STEP_02) AND "Unit1.Em2.ControlNodes".semiAutoSplice.sequence.status.seqActive AND "Unit1.Em2.ControlNodes".semiAutoSplice."step".transition1[1602],
                           PT := #SeqDelayTime);
   IF #statTonTimer[1602].Q THEN
       "Unit1.Em2.ControlNodes".semiAutoSplice.sequence.status.nextStep := #JOB_16_STEP_03;
   END_IF;
END_REGION

REGION Network 75: Step[1603] :
   RUNG wire#powerrail
      { S7_Templates := "SrcType := DInt" } EQ_Contact(in1 := "Unit1.Em2.ControlNodes".semiAutoSplice.sequence.status.currentStep, in2 := #JOB_16_STEP_03)
      Contact( "Unit1.Em2.ControlNodes".semiAutoSplice.sequence.status.seqActive )
      wire#w1
      Coil( "Unit1.Em2.ControlNodes".semiAutoSplice."step".action1[1603] )
   END_RUNG
   RUNG wire#w1
      Coil( "Unit1.Em2.ControlNodes".semiAutoSplice."step".transition1[1603] )
   END_RUNG
   RUNG wire#w1
      Contact( "Unit1.Em2.ControlNodes".semiAutoSplice."step".transition1[1603] )
      { S7_Templates := "time_type := Time" } #statTonTimer[1603].TON(pt := #SeqDelayTime, et =>)
      Move(in := #JOB_16_STEP_04, out1 => "Unit1.Em2.ControlNodes".semiAutoSplice.sequence.status.nextStep)
   END_RUNG
   // the same network as SCL:
   "Unit1.Em2.ControlNodes".semiAutoSplice."step".action1[1603] := ("Unit1.Em2.ControlNodes".semiAutoSplice.sequence.status.currentStep = #JOB_16_STEP_03) AND "Unit1.Em2.ControlNodes".semiAutoSplice.sequence.status.seqActive;
   "Unit1.Em2.ControlNodes".semiAutoSplice."step".transition1[1603] := ("Unit1.Em2.ControlNodes".semiAutoSplice.sequence.status.currentStep = #JOB_16_STEP_03) AND "Unit1.Em2.ControlNodes".semiAutoSplice.sequence.status.seqActive;
   #statTonTimer[1603].TON(IN := ("Unit1.Em2.ControlNodes".semiAutoSplice.sequence.status.currentStep = #JOB_16_STEP_03) AND "Unit1.Em2.ControlNodes".semiAutoSplice.sequence.status.seqActive AND "Unit1.Em2.ControlNodes".semiAutoSplice."step".transition1[1603],
                           PT := #SeqDelayTime);
   IF #statTonTimer[1603].Q THEN
       "Unit1.Em2.ControlNodes".semiAutoSplice.sequence.status.nextStep := #JOB_16_STEP_04;
   END_IF;
END_REGION

REGION Network 76: Step[1604] :
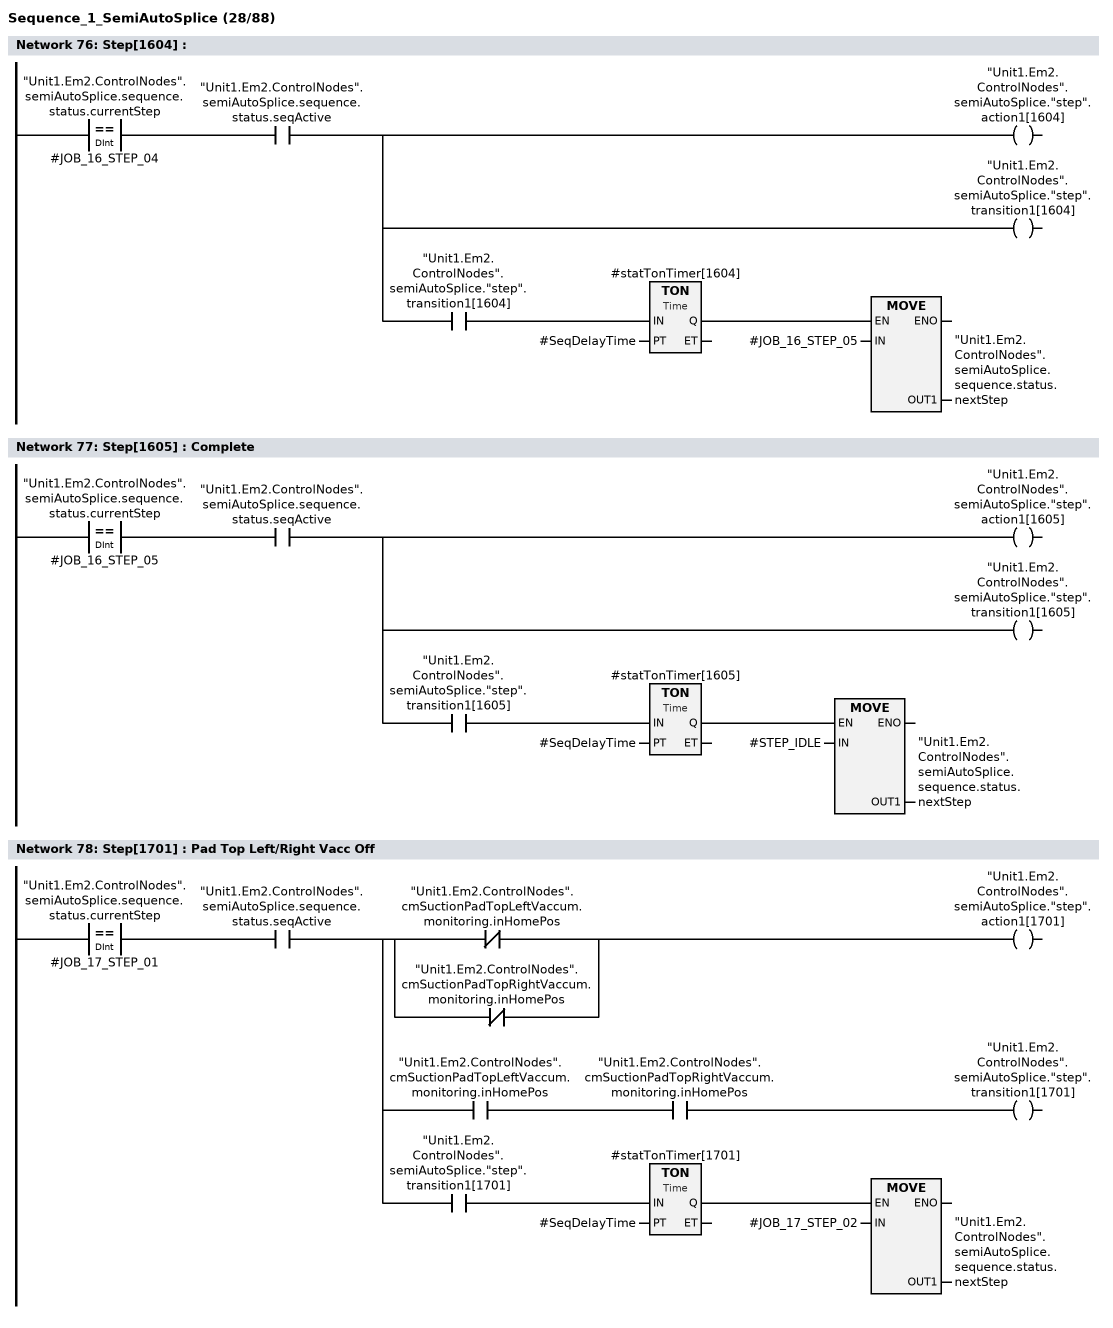
   RUNG wire#powerrail
      { S7_Templates := "SrcType := DInt" } EQ_Contact(in1 := "Unit1.Em2.ControlNodes".semiAutoSplice.sequence.status.currentStep, in2 := #JOB_16_STEP_04)
      Contact( "Unit1.Em2.ControlNodes".semiAutoSplice.sequence.status.seqActive )
      wire#w1
      Coil( "Unit1.Em2.ControlNodes".semiAutoSplice."step".action1[1604] )
   END_RUNG
   RUNG wire#w1
      Coil( "Unit1.Em2.ControlNodes".semiAutoSplice."step".transition1[1604] )
   END_RUNG
   RUNG wire#w1
      Contact( "Unit1.Em2.ControlNodes".semiAutoSplice."step".transition1[1604] )
      { S7_Templates := "time_type := Time" } #statTonTimer[1604].TON(pt := #SeqDelayTime, et =>)
      Move(in := #JOB_16_STEP_05, out1 => "Unit1.Em2.ControlNodes".semiAutoSplice.sequence.status.nextStep)
   END_RUNG
   // the same network as SCL:
   "Unit1.Em2.ControlNodes".semiAutoSplice."step".action1[1604] := ("Unit1.Em2.ControlNodes".semiAutoSplice.sequence.status.currentStep = #JOB_16_STEP_04) AND "Unit1.Em2.ControlNodes".semiAutoSplice.sequence.status.seqActive;
   "Unit1.Em2.ControlNodes".semiAutoSplice."step".transition1[1604] := ("Unit1.Em2.ControlNodes".semiAutoSplice.sequence.status.currentStep = #JOB_16_STEP_04) AND "Unit1.Em2.ControlNodes".semiAutoSplice.sequence.status.seqActive;
   #statTonTimer[1604].TON(IN := ("Unit1.Em2.ControlNodes".semiAutoSplice.sequence.status.currentStep = #JOB_16_STEP_04) AND "Unit1.Em2.ControlNodes".semiAutoSplice.sequence.status.seqActive AND "Unit1.Em2.ControlNodes".semiAutoSplice."step".transition1[1604],
                           PT := #SeqDelayTime);
   IF #statTonTimer[1604].Q THEN
       "Unit1.Em2.ControlNodes".semiAutoSplice.sequence.status.nextStep := #JOB_16_STEP_05;
   END_IF;
END_REGION

REGION Network 77: Step[1605] : Complete
   RUNG wire#powerrail
      { S7_Templates := "SrcType := DInt" } EQ_Contact(in1 := "Unit1.Em2.ControlNodes".semiAutoSplice.sequence.status.currentStep, in2 := #JOB_16_STEP_05)
      Contact( "Unit1.Em2.ControlNodes".semiAutoSplice.sequence.status.seqActive )
      wire#w1
      Coil( "Unit1.Em2.ControlNodes".semiAutoSplice."step".action1[1605] )
   END_RUNG
   RUNG wire#w1
      Coil( "Unit1.Em2.ControlNodes".semiAutoSplice."step".transition1[1605] )
   END_RUNG
   RUNG wire#w1
      Contact( "Unit1.Em2.ControlNodes".semiAutoSplice."step".transition1[1605] )
      { S7_Templates := "time_type := Time" } #statTonTimer[1605].TON(pt := #SeqDelayTime, et =>)
      Move(in := #STEP_IDLE, out1 => "Unit1.Em2.ControlNodes".semiAutoSplice.sequence.status.nextStep)
   END_RUNG
   // the same network as SCL:
   "Unit1.Em2.ControlNodes".semiAutoSplice."step".action1[1605] := ("Unit1.Em2.ControlNodes".semiAutoSplice.sequence.status.currentStep = #JOB_16_STEP_05) AND "Unit1.Em2.ControlNodes".semiAutoSplice.sequence.status.seqActive;
   "Unit1.Em2.ControlNodes".semiAutoSplice."step".transition1[1605] := ("Unit1.Em2.ControlNodes".semiAutoSplice.sequence.status.currentStep = #JOB_16_STEP_05) AND "Unit1.Em2.ControlNodes".semiAutoSplice.sequence.status.seqActive;
   #statTonTimer[1605].TON(IN := ("Unit1.Em2.ControlNodes".semiAutoSplice.sequence.status.currentStep = #JOB_16_STEP_05) AND "Unit1.Em2.ControlNodes".semiAutoSplice.sequence.status.seqActive AND "Unit1.Em2.ControlNodes".semiAutoSplice."step".transition1[1605],
                           PT := #SeqDelayTime);
   IF #statTonTimer[1605].Q THEN
       "Unit1.Em2.ControlNodes".semiAutoSplice.sequence.status.nextStep := #STEP_IDLE;
   END_IF;
END_REGION

REGION Network 78: Step[1701] : Pad Top Left/Right Vacc Off
   RUNG wire#powerrail
      { S7_Templates := "SrcType := DInt" } EQ_Contact(in1 := "Unit1.Em2.ControlNodes".semiAutoSplice.sequence.status.currentStep, in2 := #JOB_17_STEP_01)
      Contact( "Unit1.Em2.ControlNodes".semiAutoSplice.sequence.status.seqActive )
      wire#w1
      I_Contact( "Unit1.Em2.ControlNodes".cmSuctionPadTopLeftVaccum.monitoring.inHomePos )
      wire#w2
      Coil( "Unit1.Em2.ControlNodes".semiAutoSplice."step".action1[1701] )
   END_RUNG
   RUNG wire#w1
      I_Contact( "Unit1.Em2.ControlNodes".cmSuctionPadTopRightVaccum.monitoring.inHomePos )
   END_RUNG wire#w2
   RUNG wire#w1
      Contact( "Unit1.Em2.ControlNodes".cmSuctionPadTopLeftVaccum.monitoring.inHomePos )
      Contact( "Unit1.Em2.ControlNodes".cmSuctionPadTopRightVaccum.monitoring.inHomePos )
      Coil( "Unit1.Em2.ControlNodes".semiAutoSplice."step".transition1[1701] )
   END_RUNG
   RUNG wire#w1
      Contact( "Unit1.Em2.ControlNodes".semiAutoSplice."step".transition1[1701] )
      { S7_Templates := "time_type := Time" } #statTonTimer[1701].TON(pt := #SeqDelayTime, et =>)
      Move(in := #JOB_17_STEP_02, out1 => "Unit1.Em2.ControlNodes".semiAutoSplice.sequence.status.nextStep)
   END_RUNG
   // the same network as SCL:
   #_w1 := ("Unit1.Em2.ControlNodes".semiAutoSplice.sequence.status.currentStep = #JOB_17_STEP_01) AND "Unit1.Em2.ControlNodes".semiAutoSplice.sequence.status.seqActive;
   "Unit1.Em2.ControlNodes".semiAutoSplice."step".action1[1701] := #_w1 AND (NOT "Unit1.Em2.ControlNodes".cmSuctionPadTopLeftVaccum.monitoring.inHomePos OR NOT "Unit1.Em2.ControlNodes".cmSuctionPadTopRightVaccum.monitoring.inHomePos);
   "Unit1.Em2.ControlNodes".semiAutoSplice."step".transition1[1701] := #_w1 AND "Unit1.Em2.ControlNodes".cmSuctionPadTopLeftVaccum.monitoring.inHomePos AND "Unit1.Em2.ControlNodes".cmSuctionPadTopRightVaccum.monitoring.inHomePos;
   #statTonTimer[1701].TON(IN := #_w1 AND "Unit1.Em2.ControlNodes".semiAutoSplice."step".transition1[1701],
                           PT := #SeqDelayTime);
   IF #statTonTimer[1701].Q THEN
       "Unit1.Em2.ControlNodes".semiAutoSplice.sequence.status.nextStep := #JOB_17_STEP_02;
   END_IF;
END_REGION

REGION Network 79: Step[1702] :
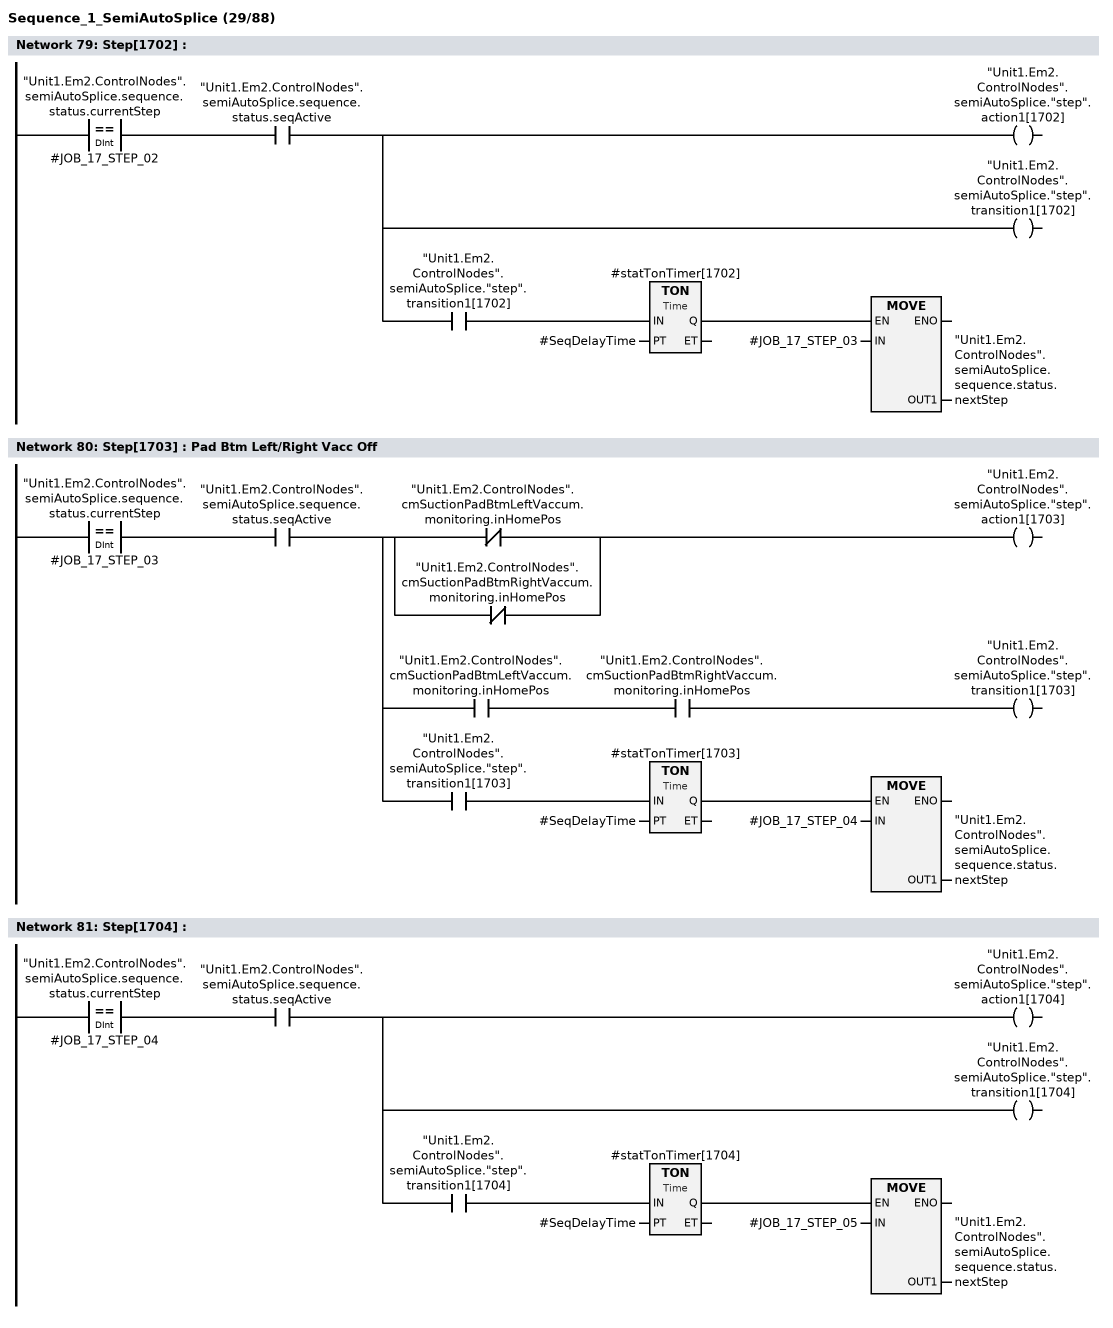
   RUNG wire#powerrail
      { S7_Templates := "SrcType := DInt" } EQ_Contact(in1 := "Unit1.Em2.ControlNodes".semiAutoSplice.sequence.status.currentStep, in2 := #JOB_17_STEP_02)
      Contact( "Unit1.Em2.ControlNodes".semiAutoSplice.sequence.status.seqActive )
      wire#w1
      Coil( "Unit1.Em2.ControlNodes".semiAutoSplice."step".action1[1702] )
   END_RUNG
   RUNG wire#w1
      Coil( "Unit1.Em2.ControlNodes".semiAutoSplice."step".transition1[1702] )
   END_RUNG
   RUNG wire#w1
      Contact( "Unit1.Em2.ControlNodes".semiAutoSplice."step".transition1[1702] )
      { S7_Templates := "time_type := Time" } #statTonTimer[1702].TON(pt := #SeqDelayTime, et =>)
      Move(in := #JOB_17_STEP_03, out1 => "Unit1.Em2.ControlNodes".semiAutoSplice.sequence.status.nextStep)
   END_RUNG
   // the same network as SCL:
   "Unit1.Em2.ControlNodes".semiAutoSplice."step".action1[1702] := ("Unit1.Em2.ControlNodes".semiAutoSplice.sequence.status.currentStep = #JOB_17_STEP_02) AND "Unit1.Em2.ControlNodes".semiAutoSplice.sequence.status.seqActive;
   "Unit1.Em2.ControlNodes".semiAutoSplice."step".transition1[1702] := ("Unit1.Em2.ControlNodes".semiAutoSplice.sequence.status.currentStep = #JOB_17_STEP_02) AND "Unit1.Em2.ControlNodes".semiAutoSplice.sequence.status.seqActive;
   #statTonTimer[1702].TON(IN := ("Unit1.Em2.ControlNodes".semiAutoSplice.sequence.status.currentStep = #JOB_17_STEP_02) AND "Unit1.Em2.ControlNodes".semiAutoSplice.sequence.status.seqActive AND "Unit1.Em2.ControlNodes".semiAutoSplice."step".transition1[1702],
                           PT := #SeqDelayTime);
   IF #statTonTimer[1702].Q THEN
       "Unit1.Em2.ControlNodes".semiAutoSplice.sequence.status.nextStep := #JOB_17_STEP_03;
   END_IF;
END_REGION

REGION Network 80: Step[1703] : Pad Btm Left/Right Vacc Off
   RUNG wire#powerrail
      { S7_Templates := "SrcType := DInt" } EQ_Contact(in1 := "Unit1.Em2.ControlNodes".semiAutoSplice.sequence.status.currentStep, in2 := #JOB_17_STEP_03)
      Contact( "Unit1.Em2.ControlNodes".semiAutoSplice.sequence.status.seqActive )
      wire#w1
      I_Contact( "Unit1.Em2.ControlNodes".cmSuctionPadBtmLeftVaccum.monitoring.inHomePos )
      wire#w2
      Coil( "Unit1.Em2.ControlNodes".semiAutoSplice."step".action1[1703] )
   END_RUNG
   RUNG wire#w1
      I_Contact( "Unit1.Em2.ControlNodes".cmSuctionPadBtmRightVaccum.monitoring.inHomePos )
   END_RUNG wire#w2
   RUNG wire#w1
      Contact( "Unit1.Em2.ControlNodes".cmSuctionPadBtmLeftVaccum.monitoring.inHomePos )
      Contact( "Unit1.Em2.ControlNodes".cmSuctionPadBtmRightVaccum.monitoring.inHomePos )
      Coil( "Unit1.Em2.ControlNodes".semiAutoSplice."step".transition1[1703] )
   END_RUNG
   RUNG wire#w1
      Contact( "Unit1.Em2.ControlNodes".semiAutoSplice."step".transition1[1703] )
      { S7_Templates := "time_type := Time" } #statTonTimer[1703].TON(pt := #SeqDelayTime, et =>)
      Move(in := #JOB_17_STEP_04, out1 => "Unit1.Em2.ControlNodes".semiAutoSplice.sequence.status.nextStep)
   END_RUNG
   // the same network as SCL:
   #_w1 := ("Unit1.Em2.ControlNodes".semiAutoSplice.sequence.status.currentStep = #JOB_17_STEP_03) AND "Unit1.Em2.ControlNodes".semiAutoSplice.sequence.status.seqActive;
   "Unit1.Em2.ControlNodes".semiAutoSplice."step".action1[1703] := #_w1 AND (NOT "Unit1.Em2.ControlNodes".cmSuctionPadBtmLeftVaccum.monitoring.inHomePos OR NOT "Unit1.Em2.ControlNodes".cmSuctionPadBtmRightVaccum.monitoring.inHomePos);
   "Unit1.Em2.ControlNodes".semiAutoSplice."step".transition1[1703] := #_w1 AND "Unit1.Em2.ControlNodes".cmSuctionPadBtmLeftVaccum.monitoring.inHomePos AND "Unit1.Em2.ControlNodes".cmSuctionPadBtmRightVaccum.monitoring.inHomePos;
   #statTonTimer[1703].TON(IN := #_w1 AND "Unit1.Em2.ControlNodes".semiAutoSplice."step".transition1[1703],
                           PT := #SeqDelayTime);
   IF #statTonTimer[1703].Q THEN
       "Unit1.Em2.ControlNodes".semiAutoSplice.sequence.status.nextStep := #JOB_17_STEP_04;
   END_IF;
END_REGION

REGION Network 81: Step[1704] :
   RUNG wire#powerrail
      { S7_Templates := "SrcType := DInt" } EQ_Contact(in1 := "Unit1.Em2.ControlNodes".semiAutoSplice.sequence.status.currentStep, in2 := #JOB_17_STEP_04)
      Contact( "Unit1.Em2.ControlNodes".semiAutoSplice.sequence.status.seqActive )
      wire#w1
      Coil( "Unit1.Em2.ControlNodes".semiAutoSplice."step".action1[1704] )
   END_RUNG
   RUNG wire#w1
      Coil( "Unit1.Em2.ControlNodes".semiAutoSplice."step".transition1[1704] )
   END_RUNG
   RUNG wire#w1
      Contact( "Unit1.Em2.ControlNodes".semiAutoSplice."step".transition1[1704] )
      { S7_Templates := "time_type := Time" } #statTonTimer[1704].TON(pt := #SeqDelayTime, et =>)
      Move(in := #JOB_17_STEP_05, out1 => "Unit1.Em2.ControlNodes".semiAutoSplice.sequence.status.nextStep)
   END_RUNG
   // the same network as SCL:
   "Unit1.Em2.ControlNodes".semiAutoSplice."step".action1[1704] := ("Unit1.Em2.ControlNodes".semiAutoSplice.sequence.status.currentStep = #JOB_17_STEP_04) AND "Unit1.Em2.ControlNodes".semiAutoSplice.sequence.status.seqActive;
   "Unit1.Em2.ControlNodes".semiAutoSplice."step".transition1[1704] := ("Unit1.Em2.ControlNodes".semiAutoSplice.sequence.status.currentStep = #JOB_17_STEP_04) AND "Unit1.Em2.ControlNodes".semiAutoSplice.sequence.status.seqActive;
   #statTonTimer[1704].TON(IN := ("Unit1.Em2.ControlNodes".semiAutoSplice.sequence.status.currentStep = #JOB_17_STEP_04) AND "Unit1.Em2.ControlNodes".semiAutoSplice.sequence.status.seqActive AND "Unit1.Em2.ControlNodes".semiAutoSplice."step".transition1[1704],
                           PT := #SeqDelayTime);
   IF #statTonTimer[1704].Q THEN
       "Unit1.Em2.ControlNodes".semiAutoSplice.sequence.status.nextStep := #JOB_17_STEP_05;
   END_IF;
END_REGION

REGION Network 82: Step[1705] :
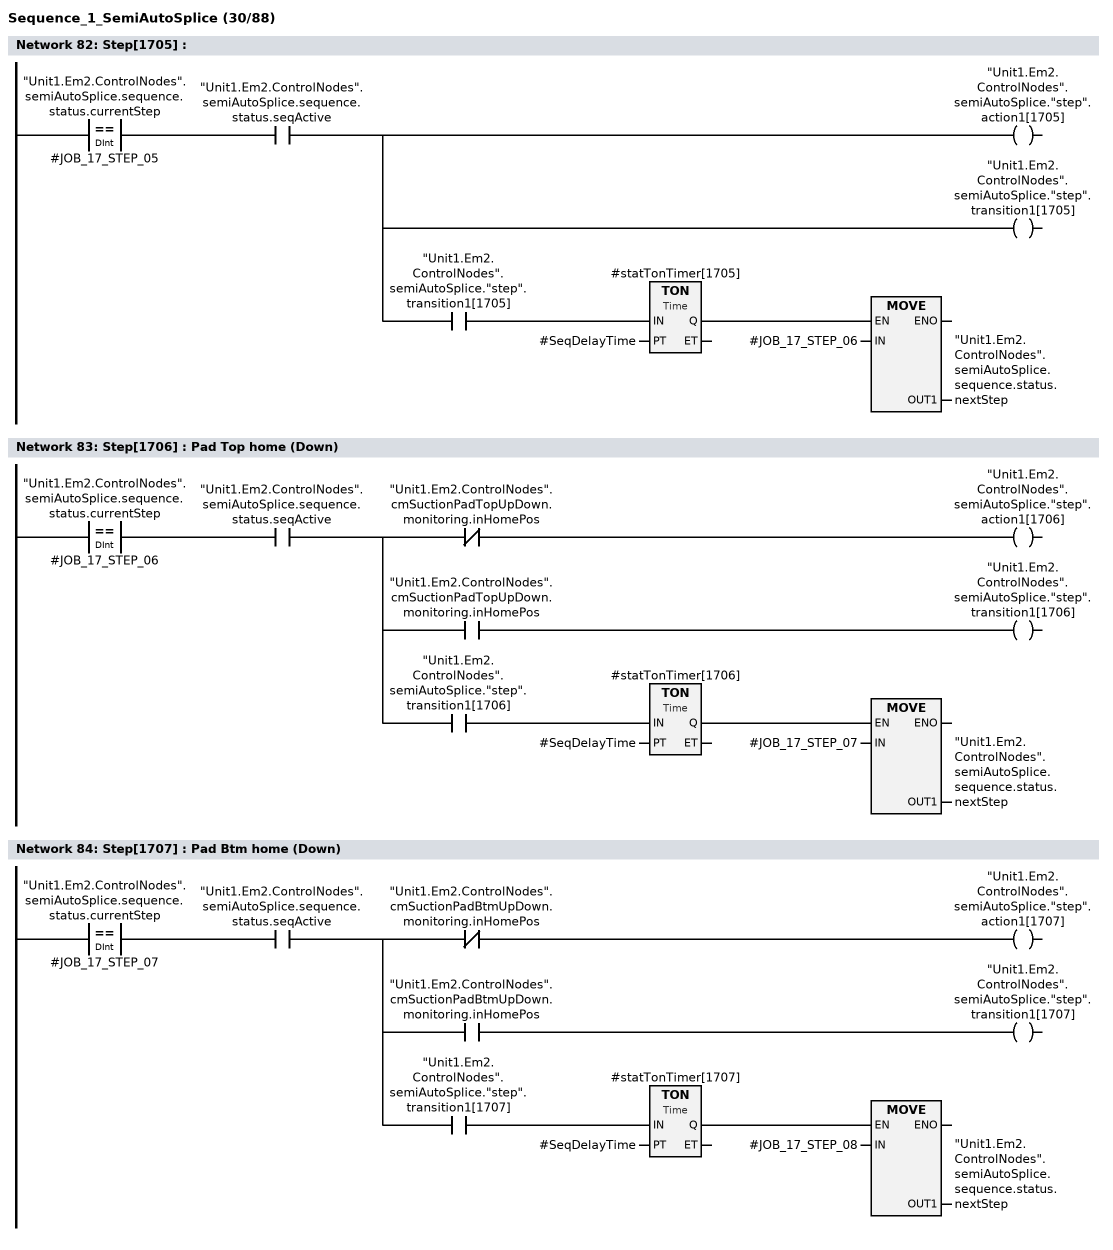
   RUNG wire#powerrail
      { S7_Templates := "SrcType := DInt" } EQ_Contact(in1 := "Unit1.Em2.ControlNodes".semiAutoSplice.sequence.status.currentStep, in2 := #JOB_17_STEP_05)
      Contact( "Unit1.Em2.ControlNodes".semiAutoSplice.sequence.status.seqActive )
      wire#w1
      Coil( "Unit1.Em2.ControlNodes".semiAutoSplice."step".action1[1705] )
   END_RUNG
   RUNG wire#w1
      Coil( "Unit1.Em2.ControlNodes".semiAutoSplice."step".transition1[1705] )
   END_RUNG
   RUNG wire#w1
      Contact( "Unit1.Em2.ControlNodes".semiAutoSplice."step".transition1[1705] )
      { S7_Templates := "time_type := Time" } #statTonTimer[1705].TON(pt := #SeqDelayTime, et =>)
      Move(in := #JOB_17_STEP_06, out1 => "Unit1.Em2.ControlNodes".semiAutoSplice.sequence.status.nextStep)
   END_RUNG
   // the same network as SCL:
   "Unit1.Em2.ControlNodes".semiAutoSplice."step".action1[1705] := ("Unit1.Em2.ControlNodes".semiAutoSplice.sequence.status.currentStep = #JOB_17_STEP_05) AND "Unit1.Em2.ControlNodes".semiAutoSplice.sequence.status.seqActive;
   "Unit1.Em2.ControlNodes".semiAutoSplice."step".transition1[1705] := ("Unit1.Em2.ControlNodes".semiAutoSplice.sequence.status.currentStep = #JOB_17_STEP_05) AND "Unit1.Em2.ControlNodes".semiAutoSplice.sequence.status.seqActive;
   #statTonTimer[1705].TON(IN := ("Unit1.Em2.ControlNodes".semiAutoSplice.sequence.status.currentStep = #JOB_17_STEP_05) AND "Unit1.Em2.ControlNodes".semiAutoSplice.sequence.status.seqActive AND "Unit1.Em2.ControlNodes".semiAutoSplice."step".transition1[1705],
                           PT := #SeqDelayTime);
   IF #statTonTimer[1705].Q THEN
       "Unit1.Em2.ControlNodes".semiAutoSplice.sequence.status.nextStep := #JOB_17_STEP_06;
   END_IF;
END_REGION

REGION Network 83: Step[1706] : Pad Top home (Down)
   RUNG wire#powerrail
      { S7_Templates := "SrcType := DInt" } EQ_Contact(in1 := "Unit1.Em2.ControlNodes".semiAutoSplice.sequence.status.currentStep, in2 := #JOB_17_STEP_06)
      Contact( "Unit1.Em2.ControlNodes".semiAutoSplice.sequence.status.seqActive )
      wire#w1
      I_Contact( "Unit1.Em2.ControlNodes".cmSuctionPadTopUpDown.monitoring.inHomePos )
      Coil( "Unit1.Em2.ControlNodes".semiAutoSplice."step".action1[1706] )
   END_RUNG
   RUNG wire#w1
      Contact( "Unit1.Em2.ControlNodes".cmSuctionPadTopUpDown.monitoring.inHomePos )
      Coil( "Unit1.Em2.ControlNodes".semiAutoSplice."step".transition1[1706] )
   END_RUNG
   RUNG wire#w1
      Contact( "Unit1.Em2.ControlNodes".semiAutoSplice."step".transition1[1706] )
      { S7_Templates := "time_type := Time" } #statTonTimer[1706].TON(pt := #SeqDelayTime, et =>)
      Move(in := #JOB_17_STEP_07, out1 => "Unit1.Em2.ControlNodes".semiAutoSplice.sequence.status.nextStep)
   END_RUNG
   // the same network as SCL:
   #_w1 := ("Unit1.Em2.ControlNodes".semiAutoSplice.sequence.status.currentStep = #JOB_17_STEP_06) AND "Unit1.Em2.ControlNodes".semiAutoSplice.sequence.status.seqActive;
   "Unit1.Em2.ControlNodes".semiAutoSplice."step".action1[1706] := #_w1 AND NOT "Unit1.Em2.ControlNodes".cmSuctionPadTopUpDown.monitoring.inHomePos;
   "Unit1.Em2.ControlNodes".semiAutoSplice."step".transition1[1706] := #_w1 AND "Unit1.Em2.ControlNodes".cmSuctionPadTopUpDown.monitoring.inHomePos;
   #statTonTimer[1706].TON(IN := #_w1 AND "Unit1.Em2.ControlNodes".semiAutoSplice."step".transition1[1706],
                           PT := #SeqDelayTime);
   IF #statTonTimer[1706].Q THEN
       "Unit1.Em2.ControlNodes".semiAutoSplice.sequence.status.nextStep := #JOB_17_STEP_07;
   END_IF;
END_REGION

REGION Network 84: Step[1707] : Pad Btm home (Down)
   RUNG wire#powerrail
      { S7_Templates := "SrcType := DInt" } EQ_Contact(in1 := "Unit1.Em2.ControlNodes".semiAutoSplice.sequence.status.currentStep, in2 := #JOB_17_STEP_07)
      Contact( "Unit1.Em2.ControlNodes".semiAutoSplice.sequence.status.seqActive )
      wire#w1
      I_Contact( "Unit1.Em2.ControlNodes".cmSuctionPadBtmUpDown.monitoring.inHomePos )
      Coil( "Unit1.Em2.ControlNodes".semiAutoSplice."step".action1[1707] )
   END_RUNG
   RUNG wire#w1
      Contact( "Unit1.Em2.ControlNodes".cmSuctionPadBtmUpDown.monitoring.inHomePos )
      Coil( "Unit1.Em2.ControlNodes".semiAutoSplice."step".transition1[1707] )
   END_RUNG
   RUNG wire#w1
      Contact( "Unit1.Em2.ControlNodes".semiAutoSplice."step".transition1[1707] )
      { S7_Templates := "time_type := Time" } #statTonTimer[1707].TON(pt := #SeqDelayTime, et =>)
      Move(in := #JOB_17_STEP_08, out1 => "Unit1.Em2.ControlNodes".semiAutoSplice.sequence.status.nextStep)
   END_RUNG
   // the same network as SCL:
   #_w1 := ("Unit1.Em2.ControlNodes".semiAutoSplice.sequence.status.currentStep = #JOB_17_STEP_07) AND "Unit1.Em2.ControlNodes".semiAutoSplice.sequence.status.seqActive;
   "Unit1.Em2.ControlNodes".semiAutoSplice."step".action1[1707] := #_w1 AND NOT "Unit1.Em2.ControlNodes".cmSuctionPadBtmUpDown.monitoring.inHomePos;
   "Unit1.Em2.ControlNodes".semiAutoSplice."step".transition1[1707] := #_w1 AND "Unit1.Em2.ControlNodes".cmSuctionPadBtmUpDown.monitoring.inHomePos;
   #statTonTimer[1707].TON(IN := #_w1 AND "Unit1.Em2.ControlNodes".semiAutoSplice."step".transition1[1707],
                           PT := #SeqDelayTime);
   IF #statTonTimer[1707].Q THEN
       "Unit1.Em2.ControlNodes".semiAutoSplice.sequence.status.nextStep := #JOB_17_STEP_08;
   END_IF;
END_REGION

REGION Network 85: Step[1708] : Complete
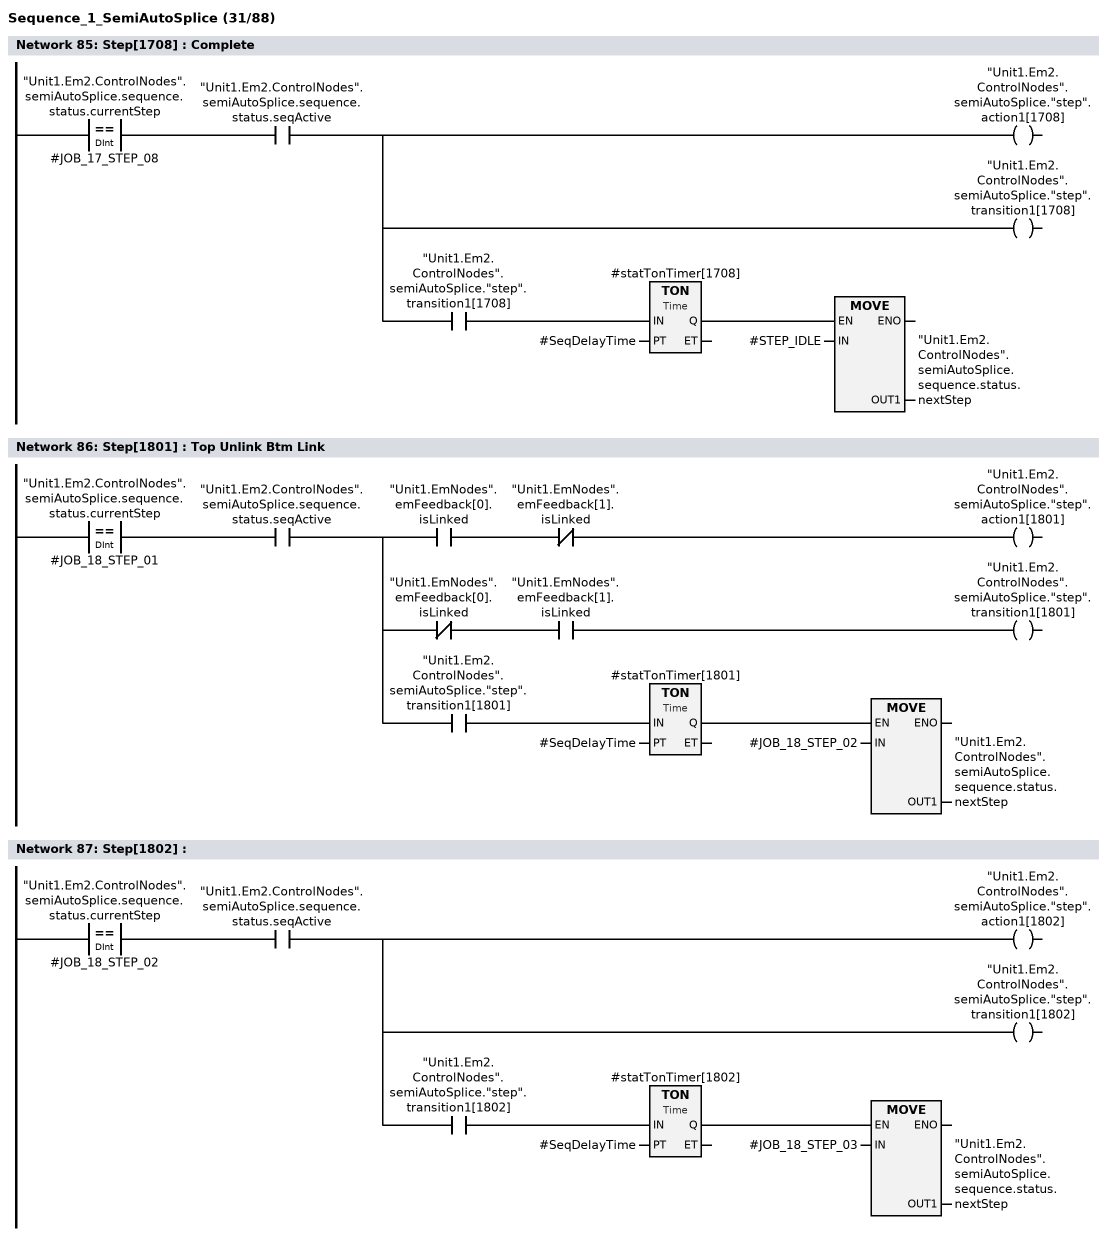
   RUNG wire#powerrail
      { S7_Templates := "SrcType := DInt" } EQ_Contact(in1 := "Unit1.Em2.ControlNodes".semiAutoSplice.sequence.status.currentStep, in2 := #JOB_17_STEP_08)
      Contact( "Unit1.Em2.ControlNodes".semiAutoSplice.sequence.status.seqActive )
      wire#w1
      Coil( "Unit1.Em2.ControlNodes".semiAutoSplice."step".action1[1708] )
   END_RUNG
   RUNG wire#w1
      Coil( "Unit1.Em2.ControlNodes".semiAutoSplice."step".transition1[1708] )
   END_RUNG
   RUNG wire#w1
      Contact( "Unit1.Em2.ControlNodes".semiAutoSplice."step".transition1[1708] )
      { S7_Templates := "time_type := Time" } #statTonTimer[1708].TON(pt := #SeqDelayTime, et =>)
      Move(in := #STEP_IDLE, out1 => "Unit1.Em2.ControlNodes".semiAutoSplice.sequence.status.nextStep)
   END_RUNG
   // the same network as SCL:
   "Unit1.Em2.ControlNodes".semiAutoSplice."step".action1[1708] := ("Unit1.Em2.ControlNodes".semiAutoSplice.sequence.status.currentStep = #JOB_17_STEP_08) AND "Unit1.Em2.ControlNodes".semiAutoSplice.sequence.status.seqActive;
   "Unit1.Em2.ControlNodes".semiAutoSplice."step".transition1[1708] := ("Unit1.Em2.ControlNodes".semiAutoSplice.sequence.status.currentStep = #JOB_17_STEP_08) AND "Unit1.Em2.ControlNodes".semiAutoSplice.sequence.status.seqActive;
   #statTonTimer[1708].TON(IN := ("Unit1.Em2.ControlNodes".semiAutoSplice.sequence.status.currentStep = #JOB_17_STEP_08) AND "Unit1.Em2.ControlNodes".semiAutoSplice.sequence.status.seqActive AND "Unit1.Em2.ControlNodes".semiAutoSplice."step".transition1[1708],
                           PT := #SeqDelayTime);
   IF #statTonTimer[1708].Q THEN
       "Unit1.Em2.ControlNodes".semiAutoSplice.sequence.status.nextStep := #STEP_IDLE;
   END_IF;
END_REGION

REGION Network 86: Step[1801] : Top Unlink Btm Link
   RUNG wire#powerrail
      { S7_Templates := "SrcType := DInt" } EQ_Contact(in1 := "Unit1.Em2.ControlNodes".semiAutoSplice.sequence.status.currentStep, in2 := #JOB_18_STEP_01)
      Contact( "Unit1.Em2.ControlNodes".semiAutoSplice.sequence.status.seqActive )
      wire#w1
      Contact( "Unit1.EmNodes".emFeedback[0].isLinked )
      I_Contact( "Unit1.EmNodes".emFeedback[1].isLinked )
      Coil( "Unit1.Em2.ControlNodes".semiAutoSplice."step".action1[1801] )
   END_RUNG
   RUNG wire#w1
      I_Contact( "Unit1.EmNodes".emFeedback[0].isLinked )
      Contact( "Unit1.EmNodes".emFeedback[1].isLinked )
      Coil( "Unit1.Em2.ControlNodes".semiAutoSplice."step".transition1[1801] )
   END_RUNG
   RUNG wire#w1
      Contact( "Unit1.Em2.ControlNodes".semiAutoSplice."step".transition1[1801] )
      { S7_Templates := "time_type := Time" } #statTonTimer[1801].TON(pt := #SeqDelayTime, et =>)
      Move(in := #JOB_18_STEP_02, out1 => "Unit1.Em2.ControlNodes".semiAutoSplice.sequence.status.nextStep)
   END_RUNG
   // the same network as SCL:
   #_w1 := ("Unit1.Em2.ControlNodes".semiAutoSplice.sequence.status.currentStep = #JOB_18_STEP_01) AND "Unit1.Em2.ControlNodes".semiAutoSplice.sequence.status.seqActive;
   "Unit1.Em2.ControlNodes".semiAutoSplice."step".action1[1801] := #_w1 AND "Unit1.EmNodes".emFeedback[0].isLinked AND NOT "Unit1.EmNodes".emFeedback[1].isLinked;
   "Unit1.Em2.ControlNodes".semiAutoSplice."step".transition1[1801] := #_w1 AND NOT "Unit1.EmNodes".emFeedback[0].isLinked AND "Unit1.EmNodes".emFeedback[1].isLinked;
   #statTonTimer[1801].TON(IN := #_w1 AND "Unit1.Em2.ControlNodes".semiAutoSplice."step".transition1[1801],
                           PT := #SeqDelayTime);
   IF #statTonTimer[1801].Q THEN
       "Unit1.Em2.ControlNodes".semiAutoSplice.sequence.status.nextStep := #JOB_18_STEP_02;
   END_IF;
END_REGION

REGION Network 87: Step[1802] :
   RUNG wire#powerrail
      { S7_Templates := "SrcType := DInt" } EQ_Contact(in1 := "Unit1.Em2.ControlNodes".semiAutoSplice.sequence.status.currentStep, in2 := #JOB_18_STEP_02)
      Contact( "Unit1.Em2.ControlNodes".semiAutoSplice.sequence.status.seqActive )
      wire#w1
      Coil( "Unit1.Em2.ControlNodes".semiAutoSplice."step".action1[1802] )
   END_RUNG
   RUNG wire#w1
      Coil( "Unit1.Em2.ControlNodes".semiAutoSplice."step".transition1[1802] )
   END_RUNG
   RUNG wire#w1
      Contact( "Unit1.Em2.ControlNodes".semiAutoSplice."step".transition1[1802] )
      { S7_Templates := "time_type := Time" } #statTonTimer[1802].TON(pt := #SeqDelayTime, et =>)
      Move(in := #JOB_18_STEP_03, out1 => "Unit1.Em2.ControlNodes".semiAutoSplice.sequence.status.nextStep)
   END_RUNG
   // the same network as SCL:
   "Unit1.Em2.ControlNodes".semiAutoSplice."step".action1[1802] := ("Unit1.Em2.ControlNodes".semiAutoSplice.sequence.status.currentStep = #JOB_18_STEP_02) AND "Unit1.Em2.ControlNodes".semiAutoSplice.sequence.status.seqActive;
   "Unit1.Em2.ControlNodes".semiAutoSplice."step".transition1[1802] := ("Unit1.Em2.ControlNodes".semiAutoSplice.sequence.status.currentStep = #JOB_18_STEP_02) AND "Unit1.Em2.ControlNodes".semiAutoSplice.sequence.status.seqActive;
   #statTonTimer[1802].TON(IN := ("Unit1.Em2.ControlNodes".semiAutoSplice.sequence.status.currentStep = #JOB_18_STEP_02) AND "Unit1.Em2.ControlNodes".semiAutoSplice.sequence.status.seqActive AND "Unit1.Em2.ControlNodes".semiAutoSplice."step".transition1[1802],
                           PT := #SeqDelayTime);
   IF #statTonTimer[1802].Q THEN
       "Unit1.Em2.ControlNodes".semiAutoSplice.sequence.status.nextStep := #JOB_18_STEP_03;
   END_IF;
END_REGION

REGION Network 88: Step[1803] :
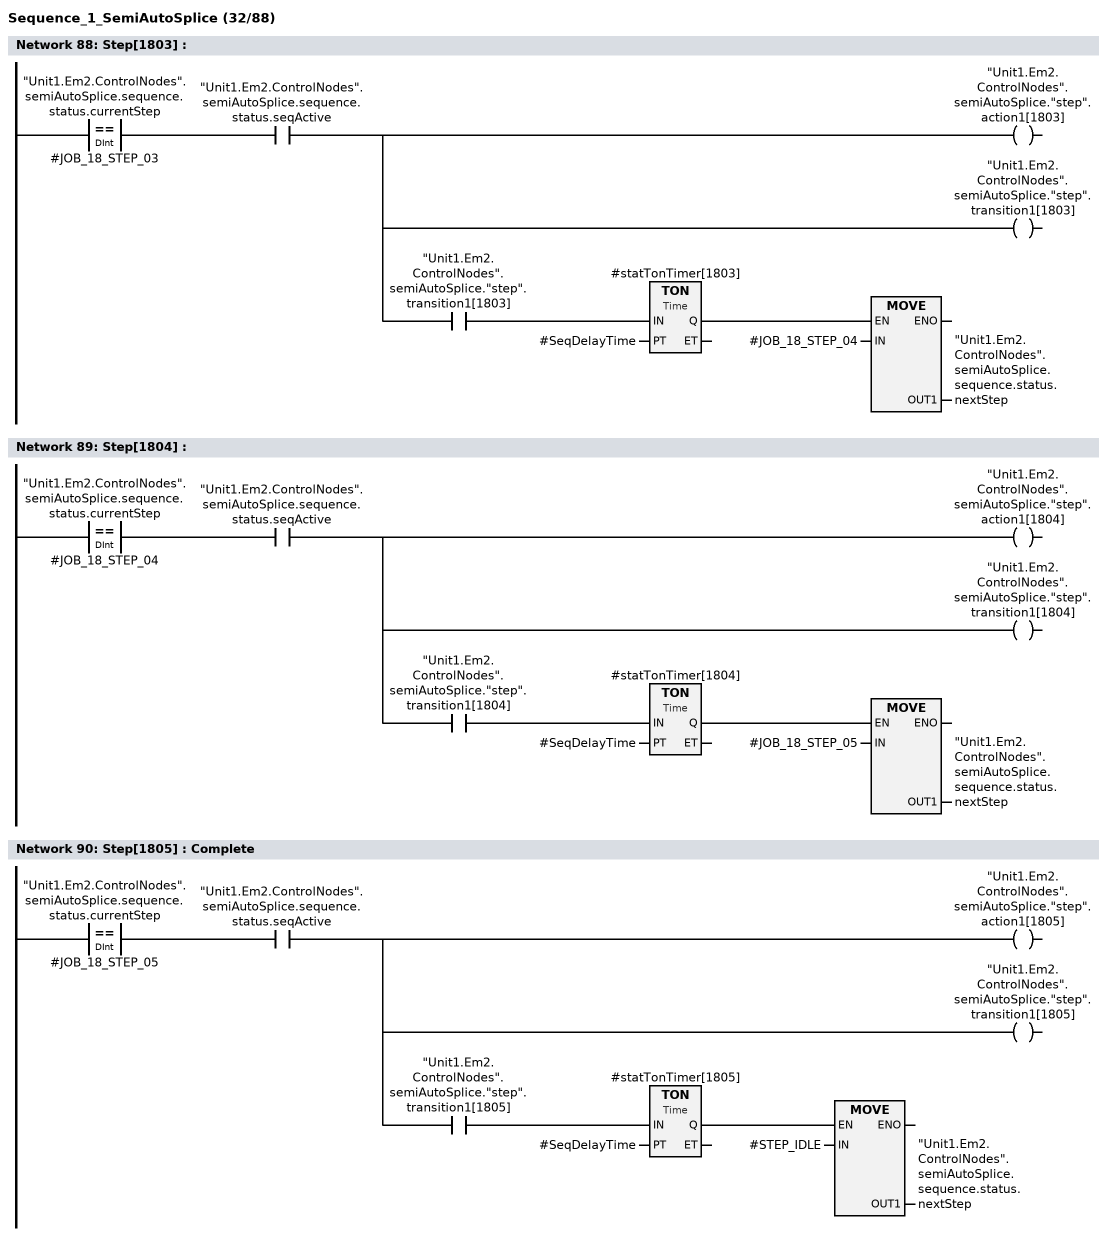
   RUNG wire#powerrail
      { S7_Templates := "SrcType := DInt" } EQ_Contact(in1 := "Unit1.Em2.ControlNodes".semiAutoSplice.sequence.status.currentStep, in2 := #JOB_18_STEP_03)
      Contact( "Unit1.Em2.ControlNodes".semiAutoSplice.sequence.status.seqActive )
      wire#w1
      Coil( "Unit1.Em2.ControlNodes".semiAutoSplice."step".action1[1803] )
   END_RUNG
   RUNG wire#w1
      Coil( "Unit1.Em2.ControlNodes".semiAutoSplice."step".transition1[1803] )
   END_RUNG
   RUNG wire#w1
      Contact( "Unit1.Em2.ControlNodes".semiAutoSplice."step".transition1[1803] )
      { S7_Templates := "time_type := Time" } #statTonTimer[1803].TON(pt := #SeqDelayTime, et =>)
      Move(in := #JOB_18_STEP_04, out1 => "Unit1.Em2.ControlNodes".semiAutoSplice.sequence.status.nextStep)
   END_RUNG
   // the same network as SCL:
   "Unit1.Em2.ControlNodes".semiAutoSplice."step".action1[1803] := ("Unit1.Em2.ControlNodes".semiAutoSplice.sequence.status.currentStep = #JOB_18_STEP_03) AND "Unit1.Em2.ControlNodes".semiAutoSplice.sequence.status.seqActive;
   "Unit1.Em2.ControlNodes".semiAutoSplice."step".transition1[1803] := ("Unit1.Em2.ControlNodes".semiAutoSplice.sequence.status.currentStep = #JOB_18_STEP_03) AND "Unit1.Em2.ControlNodes".semiAutoSplice.sequence.status.seqActive;
   #statTonTimer[1803].TON(IN := ("Unit1.Em2.ControlNodes".semiAutoSplice.sequence.status.currentStep = #JOB_18_STEP_03) AND "Unit1.Em2.ControlNodes".semiAutoSplice.sequence.status.seqActive AND "Unit1.Em2.ControlNodes".semiAutoSplice."step".transition1[1803],
                           PT := #SeqDelayTime);
   IF #statTonTimer[1803].Q THEN
       "Unit1.Em2.ControlNodes".semiAutoSplice.sequence.status.nextStep := #JOB_18_STEP_04;
   END_IF;
END_REGION

REGION Network 89: Step[1804] :
   RUNG wire#powerrail
      { S7_Templates := "SrcType := DInt" } EQ_Contact(in1 := "Unit1.Em2.ControlNodes".semiAutoSplice.sequence.status.currentStep, in2 := #JOB_18_STEP_04)
      Contact( "Unit1.Em2.ControlNodes".semiAutoSplice.sequence.status.seqActive )
      wire#w1
      Coil( "Unit1.Em2.ControlNodes".semiAutoSplice."step".action1[1804] )
   END_RUNG
   RUNG wire#w1
      Coil( "Unit1.Em2.ControlNodes".semiAutoSplice."step".transition1[1804] )
   END_RUNG
   RUNG wire#w1
      Contact( "Unit1.Em2.ControlNodes".semiAutoSplice."step".transition1[1804] )
      { S7_Templates := "time_type := Time" } #statTonTimer[1804].TON(pt := #SeqDelayTime, et =>)
      Move(in := #JOB_18_STEP_05, out1 => "Unit1.Em2.ControlNodes".semiAutoSplice.sequence.status.nextStep)
   END_RUNG
   // the same network as SCL:
   "Unit1.Em2.ControlNodes".semiAutoSplice."step".action1[1804] := ("Unit1.Em2.ControlNodes".semiAutoSplice.sequence.status.currentStep = #JOB_18_STEP_04) AND "Unit1.Em2.ControlNodes".semiAutoSplice.sequence.status.seqActive;
   "Unit1.Em2.ControlNodes".semiAutoSplice."step".transition1[1804] := ("Unit1.Em2.ControlNodes".semiAutoSplice.sequence.status.currentStep = #JOB_18_STEP_04) AND "Unit1.Em2.ControlNodes".semiAutoSplice.sequence.status.seqActive;
   #statTonTimer[1804].TON(IN := ("Unit1.Em2.ControlNodes".semiAutoSplice.sequence.status.currentStep = #JOB_18_STEP_04) AND "Unit1.Em2.ControlNodes".semiAutoSplice.sequence.status.seqActive AND "Unit1.Em2.ControlNodes".semiAutoSplice."step".transition1[1804],
                           PT := #SeqDelayTime);
   IF #statTonTimer[1804].Q THEN
       "Unit1.Em2.ControlNodes".semiAutoSplice.sequence.status.nextStep := #JOB_18_STEP_05;
   END_IF;
END_REGION

REGION Network 90: Step[1805] : Complete
   RUNG wire#powerrail
      { S7_Templates := "SrcType := DInt" } EQ_Contact(in1 := "Unit1.Em2.ControlNodes".semiAutoSplice.sequence.status.currentStep, in2 := #JOB_18_STEP_05)
      Contact( "Unit1.Em2.ControlNodes".semiAutoSplice.sequence.status.seqActive )
      wire#w1
      Coil( "Unit1.Em2.ControlNodes".semiAutoSplice."step".action1[1805] )
   END_RUNG
   RUNG wire#w1
      Coil( "Unit1.Em2.ControlNodes".semiAutoSplice."step".transition1[1805] )
   END_RUNG
   RUNG wire#w1
      Contact( "Unit1.Em2.ControlNodes".semiAutoSplice."step".transition1[1805] )
      { S7_Templates := "time_type := Time" } #statTonTimer[1805].TON(pt := #SeqDelayTime, et =>)
      Move(in := #STEP_IDLE, out1 => "Unit1.Em2.ControlNodes".semiAutoSplice.sequence.status.nextStep)
   END_RUNG
   // the same network as SCL:
   "Unit1.Em2.ControlNodes".semiAutoSplice."step".action1[1805] := ("Unit1.Em2.ControlNodes".semiAutoSplice.sequence.status.currentStep = #JOB_18_STEP_05) AND "Unit1.Em2.ControlNodes".semiAutoSplice.sequence.status.seqActive;
   "Unit1.Em2.ControlNodes".semiAutoSplice."step".transition1[1805] := ("Unit1.Em2.ControlNodes".semiAutoSplice.sequence.status.currentStep = #JOB_18_STEP_05) AND "Unit1.Em2.ControlNodes".semiAutoSplice.sequence.status.seqActive;
   #statTonTimer[1805].TON(IN := ("Unit1.Em2.ControlNodes".semiAutoSplice.sequence.status.currentStep = #JOB_18_STEP_05) AND "Unit1.Em2.ControlNodes".semiAutoSplice.sequence.status.seqActive AND "Unit1.Em2.ControlNodes".semiAutoSplice."step".transition1[1805],
                           PT := #SeqDelayTime);
   IF #statTonTimer[1805].Q THEN
       "Unit1.Em2.ControlNodes".semiAutoSplice.sequence.status.nextStep := #STEP_IDLE;
   END_IF;
END_REGION

REGION Network 91: Step[1901] :
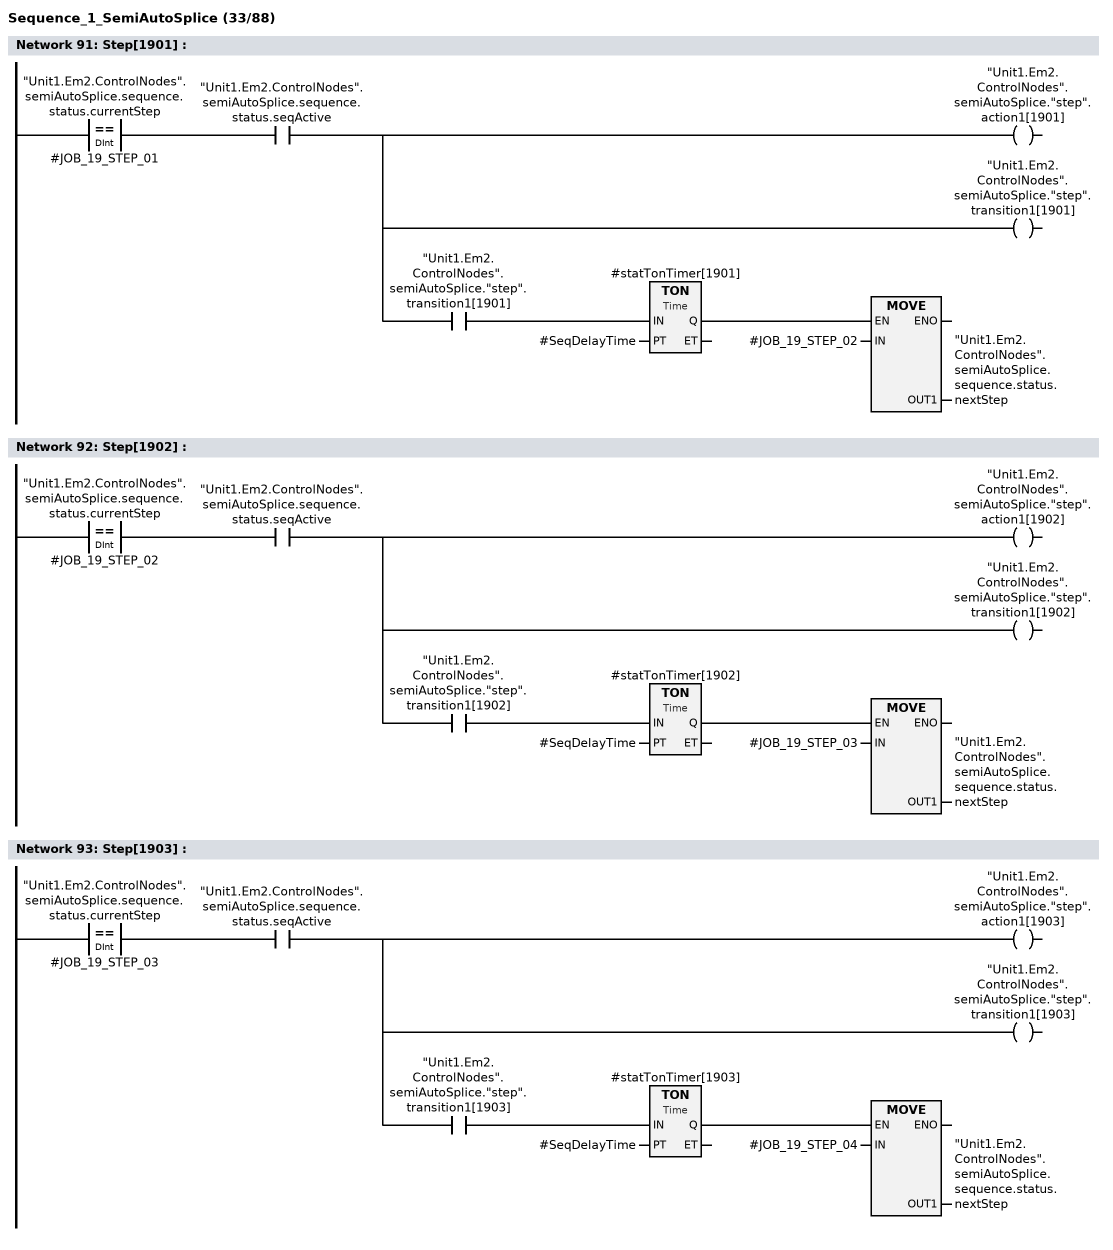
   RUNG wire#powerrail
      { S7_Templates := "SrcType := DInt" } EQ_Contact(in1 := "Unit1.Em2.ControlNodes".semiAutoSplice.sequence.status.currentStep, in2 := #JOB_19_STEP_01)
      Contact( "Unit1.Em2.ControlNodes".semiAutoSplice.sequence.status.seqActive )
      wire#w1
      Coil( "Unit1.Em2.ControlNodes".semiAutoSplice."step".action1[1901] )
   END_RUNG
   RUNG wire#w1
      Coil( "Unit1.Em2.ControlNodes".semiAutoSplice."step".transition1[1901] )
   END_RUNG
   RUNG wire#w1
      Contact( "Unit1.Em2.ControlNodes".semiAutoSplice."step".transition1[1901] )
      { S7_Templates := "time_type := Time" } #statTonTimer[1901].TON(pt := #SeqDelayTime, et =>)
      Move(in := #JOB_19_STEP_02, out1 => "Unit1.Em2.ControlNodes".semiAutoSplice.sequence.status.nextStep)
   END_RUNG
   // the same network as SCL:
   "Unit1.Em2.ControlNodes".semiAutoSplice."step".action1[1901] := ("Unit1.Em2.ControlNodes".semiAutoSplice.sequence.status.currentStep = #JOB_19_STEP_01) AND "Unit1.Em2.ControlNodes".semiAutoSplice.sequence.status.seqActive;
   "Unit1.Em2.ControlNodes".semiAutoSplice."step".transition1[1901] := ("Unit1.Em2.ControlNodes".semiAutoSplice.sequence.status.currentStep = #JOB_19_STEP_01) AND "Unit1.Em2.ControlNodes".semiAutoSplice.sequence.status.seqActive;
   #statTonTimer[1901].TON(IN := ("Unit1.Em2.ControlNodes".semiAutoSplice.sequence.status.currentStep = #JOB_19_STEP_01) AND "Unit1.Em2.ControlNodes".semiAutoSplice.sequence.status.seqActive AND "Unit1.Em2.ControlNodes".semiAutoSplice."step".transition1[1901],
                           PT := #SeqDelayTime);
   IF #statTonTimer[1901].Q THEN
       "Unit1.Em2.ControlNodes".semiAutoSplice.sequence.status.nextStep := #JOB_19_STEP_02;
   END_IF;
END_REGION

